// TIA Portal V17 export
// export: Created 2025-03-14T10:45:43.7128547Z, ExportSetting WithDefaults, DisplayName Totally Integrated Automation Portal, DisplayVersion V17 Update 8, DisplayName TIA Portal Openness, DisplayVersion V17 Update 8, DisplayName TIA Portal Version Control Interface, DisplayVersion V17, DisplayName SINAMICS Startdrive Advanced, DisplayVersion V17 SP2, DisplayName SINAMICS Startdrive G110M, G120, G120C, G120D, G120P, G115D, DisplayVersion V17 SP2, DisplayName SINAMICS Startdrive G130, G150, S120, S150, SINAMICS MV, S210, DisplayVersion V17 SP2, DisplayName STEP 7 Professional, DisplayVersion V17 Update 8, DisplayName SINUMERIK ONE STEP 7 Toolbox, DisplayVersion V17 Update 12, DisplayName SINUMERIK 840D sl STEP 7 Toolbox, DisplayVersion V17 Update 12, DisplayName STEP 7 Safety, DisplayVersion V17 Update 6, DisplayName WinCC Advanced, DisplayVersion V17 Update 8
FUNCTION "FC2036_MANUAL_LOAD_CYCLE" : Void   // FC2036, LAD
{ S7_Optimized_Access := 'FALSE' }
AUTHOR : ETXETAR
VERSION : 1.0
// stored: AutoNumber false, IsIECCheckEnabled false, SetENOAutomatically false, UDAEnableTagReadback false
   VAR_TEMP
      O_BYTE_0 : Struct   // OPTIONS BYTE 0
         MANUAL_LOAD_SELECTOR : Bool;   // MANUAL LOAD SELECTOR OPTION
      END_STRUCT;
   END_VAR
   VAR CONSTANT
      FC_NUMBER : Int := 2036;
      ZERO : Char := '0';
   END_VAR
   VAR_TEMP   // added for the SCL form of the ladder/FBD networks
      _w1 : Bool;
      _w2 : Bool;
      _w3 : Bool;
      _w4 : Bool;
      _w5 : Bool;
      _w6 : Bool;
      _w7 : Bool;
      _w8 : Bool;
      _w9 : Bool;
      _w10 : Bool;
      _w11 : Bool;
      _w12 : Bool;
      _w13 : Bool;
      _w14 : Bool;
      _w15 : Bool;
      _w16 : Bool;
      _w17 : Bool;
      _w18 : Bool;
      _w19 : Bool;
      _w20 : Bool;
      _w21 : Bool;
      _w22 : Bool;
      _w23 : Bool;
      _w24 : Bool;
      _w25 : Bool;
      _w26 : Bool;
   END_VAR
BEGIN

REGION Network 1: MANUAL LOAD SELECTOR OPTION
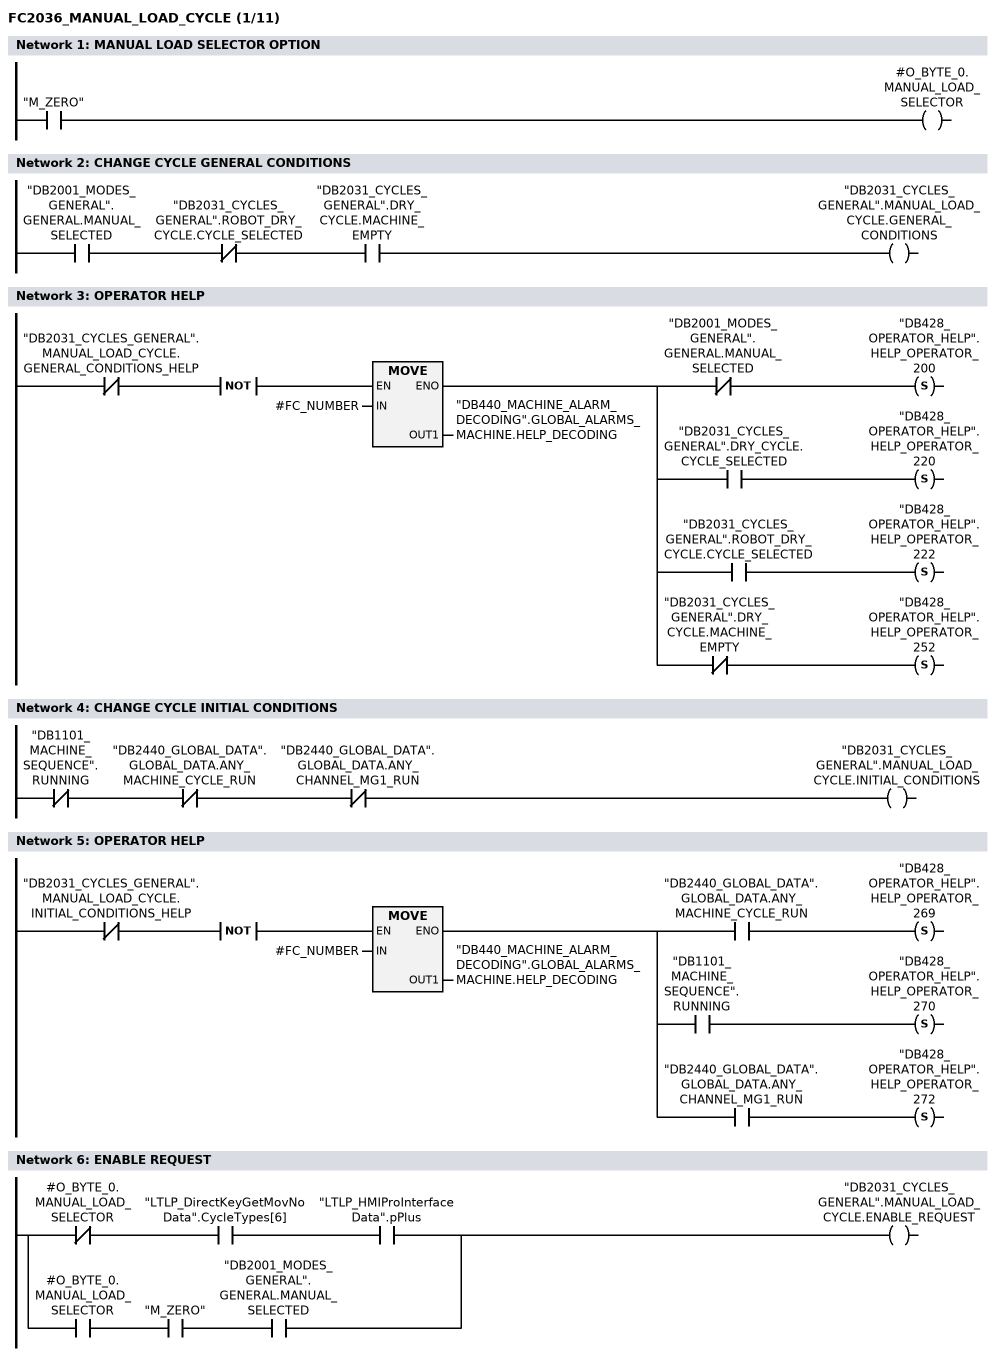
   RUNG wire#powerrail
      Contact( "M_ZERO" )
      Coil( #O_BYTE_0.MANUAL_LOAD_SELECTOR )
   END_RUNG
   // the same network as SCL:
   #O_BYTE_0.MANUAL_LOAD_SELECTOR := "M_ZERO";
END_REGION

REGION Network 2: CHANGE CYCLE GENERAL CONDITIONS
   RUNG wire#powerrail
      Contact( "DB2001_MODES_GENERAL".GENERAL.MANUAL_SELECTED )
      I_Contact( "DB2031_CYCLES_GENERAL".ROBOT_DRY_CYCLE.CYCLE_SELECTED )
      Contact( "DB2031_CYCLES_GENERAL".DRY_CYCLE.MACHINE_EMPTY )
      Coil( "DB2031_CYCLES_GENERAL".MANUAL_LOAD_CYCLE.GENERAL_CONDITIONS )
   END_RUNG
   // the same network as SCL:
   "DB2031_CYCLES_GENERAL".MANUAL_LOAD_CYCLE.GENERAL_CONDITIONS := "DB2001_MODES_GENERAL".GENERAL.MANUAL_SELECTED AND NOT "DB2031_CYCLES_GENERAL".ROBOT_DRY_CYCLE.CYCLE_SELECTED AND "DB2031_CYCLES_GENERAL".DRY_CYCLE.MACHINE_EMPTY;
END_REGION

REGION Network 3: OPERATOR HELP
   RUNG wire#powerrail
      I_Contact( "DB2031_CYCLES_GENERAL".MANUAL_LOAD_CYCLE.GENERAL_CONDITIONS_HELP )
      Not()
      { S7_GenerateENO := "TRUE" } Move(in := #FC_NUMBER, out1 => "DB440_MACHINE_ALARM_DECODING".GLOBAL_ALARMS_MACHINE.HELP_DECODING)
      wire#w1
      I_Contact( "DB2001_MODES_GENERAL".GENERAL.MANUAL_SELECTED )
      S_Coil( "DB428_OPERATOR_HELP".HELP_OPERATOR_200 )
   END_RUNG
   RUNG wire#w1
      Contact( "DB2031_CYCLES_GENERAL".DRY_CYCLE.CYCLE_SELECTED )
      S_Coil( "DB428_OPERATOR_HELP".HELP_OPERATOR_220 )
   END_RUNG
   RUNG wire#w1
      Contact( "DB2031_CYCLES_GENERAL".ROBOT_DRY_CYCLE.CYCLE_SELECTED )
      S_Coil( "DB428_OPERATOR_HELP".HELP_OPERATOR_222 )
   END_RUNG
   RUNG wire#w1
      I_Contact( "DB2031_CYCLES_GENERAL".DRY_CYCLE.MACHINE_EMPTY )
      S_Coil( "DB428_OPERATOR_HELP".HELP_OPERATOR_252 )
   END_RUNG
   // the same network as SCL:
   // ENO of a box is taken as its EN; it also drops when the box reports an error
   #_w1 := NOT (NOT "DB2031_CYCLES_GENERAL".MANUAL_LOAD_CYCLE.GENERAL_CONDITIONS_HELP);
   IF #_w1 THEN "DB440_MACHINE_ALARM_DECODING".GLOBAL_ALARMS_MACHINE.HELP_DECODING := #FC_NUMBER; END_IF;
   IF #_w1 AND NOT "DB2001_MODES_GENERAL".GENERAL.MANUAL_SELECTED THEN
       "DB428_OPERATOR_HELP".HELP_OPERATOR_200 := TRUE;
   END_IF;
   IF #_w1 AND "DB2031_CYCLES_GENERAL".DRY_CYCLE.CYCLE_SELECTED THEN
       "DB428_OPERATOR_HELP".HELP_OPERATOR_220 := TRUE;
   END_IF;
   IF #_w1 AND "DB2031_CYCLES_GENERAL".ROBOT_DRY_CYCLE.CYCLE_SELECTED THEN
       "DB428_OPERATOR_HELP".HELP_OPERATOR_222 := TRUE;
   END_IF;
   IF #_w1 AND NOT "DB2031_CYCLES_GENERAL".DRY_CYCLE.MACHINE_EMPTY THEN
       "DB428_OPERATOR_HELP".HELP_OPERATOR_252 := TRUE;
   END_IF;
END_REGION

REGION Network 4: CHANGE CYCLE INITIAL CONDITIONS
   RUNG wire#powerrail
      I_Contact( "DB1101_MACHINE_SEQUENCE".RUNNING )
      I_Contact( "DB2440_GLOBAL_DATA".GLOBAL_DATA.ANY_MACHINE_CYCLE_RUN )
      I_Contact( "DB2440_GLOBAL_DATA".GLOBAL_DATA.ANY_CHANNEL_MG1_RUN )
      Coil( "DB2031_CYCLES_GENERAL".MANUAL_LOAD_CYCLE.INITIAL_CONDITIONS )
   END_RUNG
   // the same network as SCL:
   "DB2031_CYCLES_GENERAL".MANUAL_LOAD_CYCLE.INITIAL_CONDITIONS := NOT "DB1101_MACHINE_SEQUENCE".RUNNING AND NOT "DB2440_GLOBAL_DATA".GLOBAL_DATA.ANY_MACHINE_CYCLE_RUN AND NOT "DB2440_GLOBAL_DATA".GLOBAL_DATA.ANY_CHANNEL_MG1_RUN;
END_REGION

REGION Network 5: OPERATOR HELP
   RUNG wire#powerrail
      I_Contact( "DB2031_CYCLES_GENERAL".MANUAL_LOAD_CYCLE.INITIAL_CONDITIONS_HELP )
      Not()
      { S7_GenerateENO := "TRUE" } Move(in := #FC_NUMBER, out1 => "DB440_MACHINE_ALARM_DECODING".GLOBAL_ALARMS_MACHINE.HELP_DECODING)
      wire#w1
      Contact( "DB2440_GLOBAL_DATA".GLOBAL_DATA.ANY_MACHINE_CYCLE_RUN )
      S_Coil( "DB428_OPERATOR_HELP".HELP_OPERATOR_269 )
   END_RUNG
   RUNG wire#w1
      Contact( "DB1101_MACHINE_SEQUENCE".RUNNING )
      S_Coil( "DB428_OPERATOR_HELP".HELP_OPERATOR_270 )
   END_RUNG
   RUNG wire#w1
      Contact( "DB2440_GLOBAL_DATA".GLOBAL_DATA.ANY_CHANNEL_MG1_RUN )
      S_Coil( "DB428_OPERATOR_HELP".HELP_OPERATOR_272 )
   END_RUNG
   // the same network as SCL:
   // ENO of a box is taken as its EN; it also drops when the box reports an error
   #_w1 := NOT (NOT "DB2031_CYCLES_GENERAL".MANUAL_LOAD_CYCLE.INITIAL_CONDITIONS_HELP);
   IF #_w1 THEN "DB440_MACHINE_ALARM_DECODING".GLOBAL_ALARMS_MACHINE.HELP_DECODING := #FC_NUMBER; END_IF;
   IF #_w1 AND "DB2440_GLOBAL_DATA".GLOBAL_DATA.ANY_MACHINE_CYCLE_RUN THEN
       "DB428_OPERATOR_HELP".HELP_OPERATOR_269 := TRUE;
   END_IF;
   IF #_w1 AND "DB1101_MACHINE_SEQUENCE".RUNNING THEN
       "DB428_OPERATOR_HELP".HELP_OPERATOR_270 := TRUE;
   END_IF;
   IF #_w1 AND "DB2440_GLOBAL_DATA".GLOBAL_DATA.ANY_CHANNEL_MG1_RUN THEN
       "DB428_OPERATOR_HELP".HELP_OPERATOR_272 := TRUE;
   END_IF;
END_REGION

REGION Network 6: ENABLE REQUEST
   RUNG wire#powerrail
      I_Contact( #O_BYTE_0.MANUAL_LOAD_SELECTOR )
      Contact( "LTLP_DirectKeyGetMovNoData".CycleTypes[6] )
      Contact( "LTLP_HMIProInterfaceData".pPlus )
      wire#w1
      Coil( "DB2031_CYCLES_GENERAL".MANUAL_LOAD_CYCLE.ENABLE_REQUEST )
   END_RUNG
   RUNG wire#powerrail
      Contact( #O_BYTE_0.MANUAL_LOAD_SELECTOR )
      Contact( "M_ZERO" )
      Contact( "DB2001_MODES_GENERAL".GENERAL.MANUAL_SELECTED )
   END_RUNG wire#w1
   // the same network as SCL:
   "DB2031_CYCLES_GENERAL".MANUAL_LOAD_CYCLE.ENABLE_REQUEST := (NOT #O_BYTE_0.MANUAL_LOAD_SELECTOR AND "LTLP_DirectKeyGetMovNoData".CycleTypes[6] AND "LTLP_HMIProInterfaceData".pPlus) OR (#O_BYTE_0.MANUAL_LOAD_SELECTOR AND "M_ZERO" AND "DB2001_MODES_GENERAL".GENERAL.MANUAL_SELECTED);
END_REGION

REGION Network 7: DISABLE REQUEST
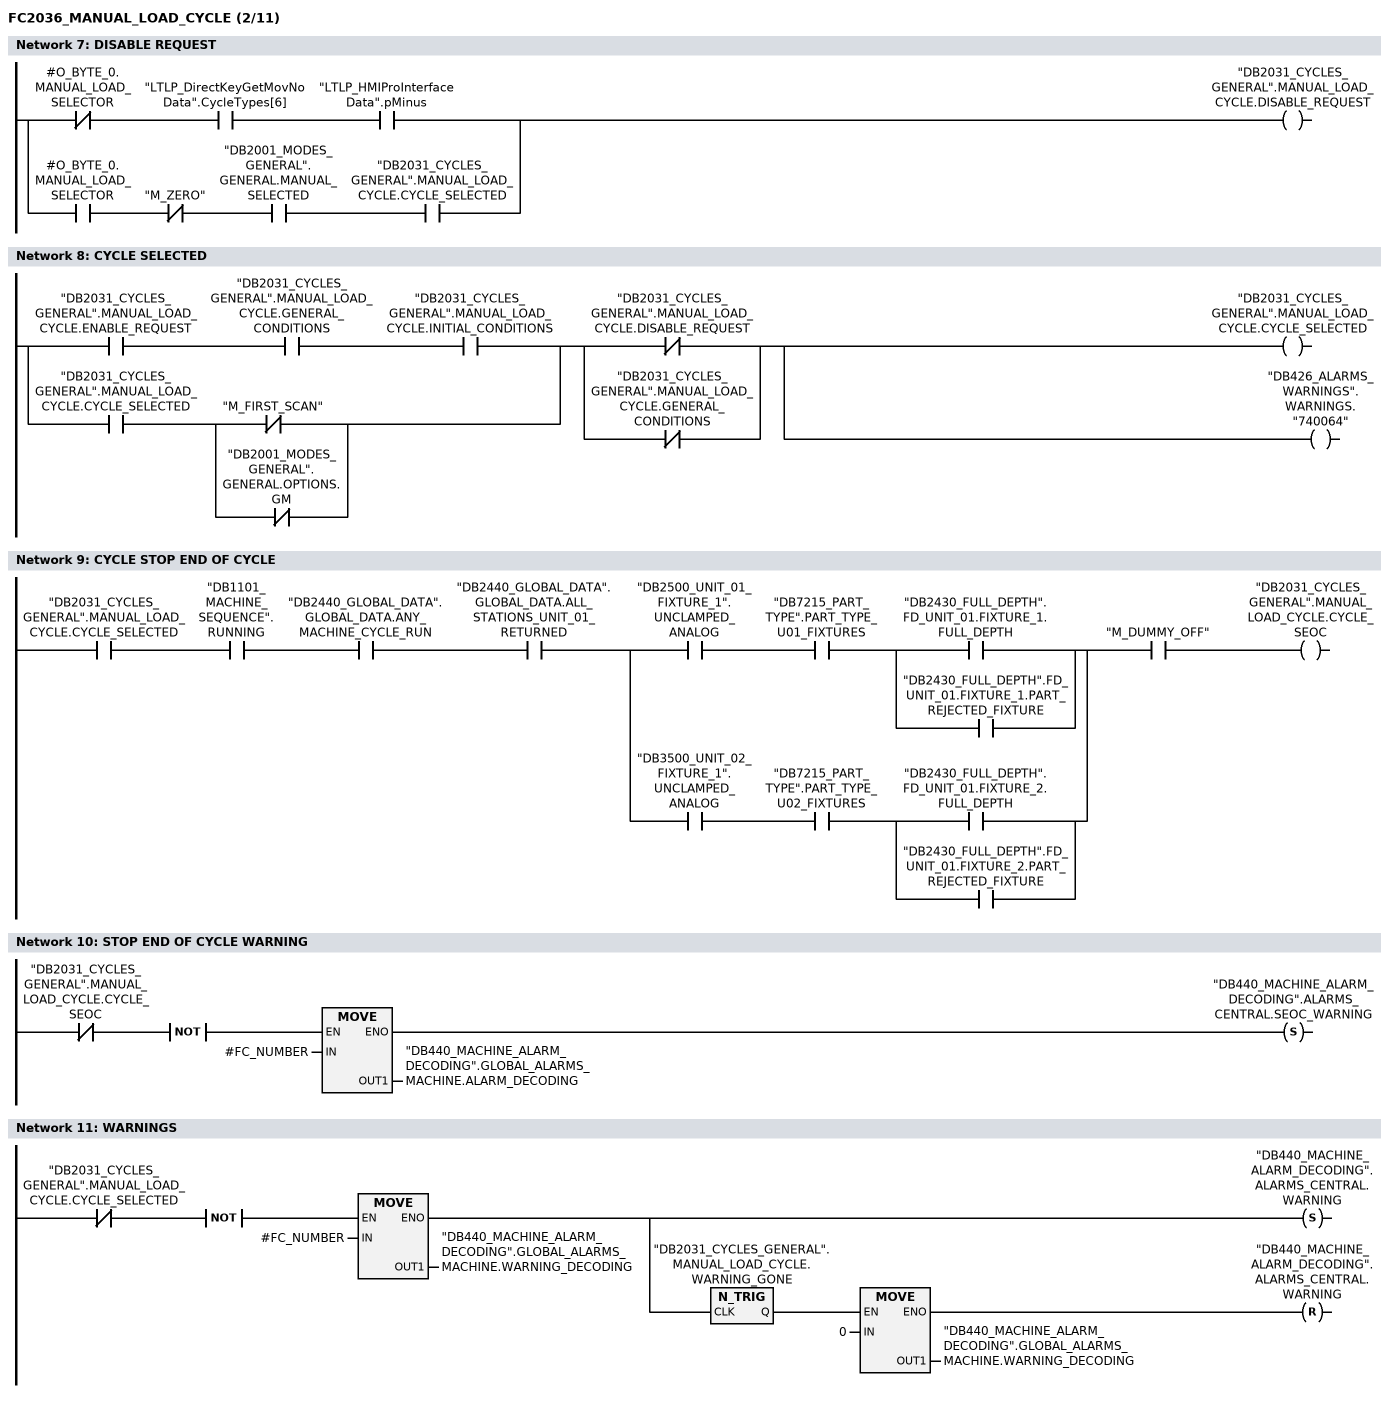
   RUNG wire#powerrail
      I_Contact( #O_BYTE_0.MANUAL_LOAD_SELECTOR )
      Contact( "LTLP_DirectKeyGetMovNoData".CycleTypes[6] )
      Contact( "LTLP_HMIProInterfaceData".pMinus )
      wire#w1
      Coil( "DB2031_CYCLES_GENERAL".MANUAL_LOAD_CYCLE.DISABLE_REQUEST )
   END_RUNG
   RUNG wire#powerrail
      Contact( #O_BYTE_0.MANUAL_LOAD_SELECTOR )
      I_Contact( "M_ZERO" )
      Contact( "DB2001_MODES_GENERAL".GENERAL.MANUAL_SELECTED )
      Contact( "DB2031_CYCLES_GENERAL".MANUAL_LOAD_CYCLE.CYCLE_SELECTED )
   END_RUNG wire#w1
   // the same network as SCL:
   "DB2031_CYCLES_GENERAL".MANUAL_LOAD_CYCLE.DISABLE_REQUEST := (NOT #O_BYTE_0.MANUAL_LOAD_SELECTOR AND "LTLP_DirectKeyGetMovNoData".CycleTypes[6] AND "LTLP_HMIProInterfaceData".pMinus) OR (#O_BYTE_0.MANUAL_LOAD_SELECTOR AND NOT "M_ZERO" AND "DB2001_MODES_GENERAL".GENERAL.MANUAL_SELECTED AND "DB2031_CYCLES_GENERAL".MANUAL_LOAD_CYCLE.CYCLE_SELECTED);
END_REGION

REGION Network 8: CYCLE SELECTED
   RUNG wire#powerrail
      Contact( "DB2031_CYCLES_GENERAL".MANUAL_LOAD_CYCLE.ENABLE_REQUEST )
      Contact( "DB2031_CYCLES_GENERAL".MANUAL_LOAD_CYCLE.GENERAL_CONDITIONS )
      Contact( "DB2031_CYCLES_GENERAL".MANUAL_LOAD_CYCLE.INITIAL_CONDITIONS )
      wire#w1
      I_Contact( "DB2031_CYCLES_GENERAL".MANUAL_LOAD_CYCLE.DISABLE_REQUEST )
      wire#w3
      Coil( "DB2031_CYCLES_GENERAL".MANUAL_LOAD_CYCLE.CYCLE_SELECTED )
   END_RUNG
   RUNG wire#powerrail
      Contact( "DB2031_CYCLES_GENERAL".MANUAL_LOAD_CYCLE.CYCLE_SELECTED )
      wire#w2
      I_Contact( "M_FIRST_SCAN" )
   END_RUNG wire#w1
   RUNG wire#w2
      I_Contact( "DB2001_MODES_GENERAL".GENERAL.OPTIONS.GM )
   END_RUNG wire#w1
   RUNG wire#w1
      I_Contact( "DB2031_CYCLES_GENERAL".MANUAL_LOAD_CYCLE.GENERAL_CONDITIONS )
   END_RUNG wire#w3
   RUNG wire#w3
      Coil( "DB426_ALARMS_WARNINGS".WARNINGS."740064" )
   END_RUNG
   // the same network as SCL:
   "DB2031_CYCLES_GENERAL".MANUAL_LOAD_CYCLE.CYCLE_SELECTED := (("DB2031_CYCLES_GENERAL".MANUAL_LOAD_CYCLE.ENABLE_REQUEST AND "DB2031_CYCLES_GENERAL".MANUAL_LOAD_CYCLE.GENERAL_CONDITIONS AND "DB2031_CYCLES_GENERAL".MANUAL_LOAD_CYCLE.INITIAL_CONDITIONS) OR ("DB2031_CYCLES_GENERAL".MANUAL_LOAD_CYCLE.CYCLE_SELECTED AND (NOT "M_FIRST_SCAN" OR NOT "DB2001_MODES_GENERAL".GENERAL.OPTIONS.GM))) AND (NOT "DB2031_CYCLES_GENERAL".MANUAL_LOAD_CYCLE.DISABLE_REQUEST OR NOT "DB2031_CYCLES_GENERAL".MANUAL_LOAD_CYCLE.GENERAL_CONDITIONS);
   "DB426_ALARMS_WARNINGS".WARNINGS."740064" := "DB2031_CYCLES_GENERAL".MANUAL_LOAD_CYCLE.CYCLE_SELECTED;
END_REGION

REGION Network 9: CYCLE STOP END OF CYCLE
   RUNG wire#powerrail
      Contact( "DB2031_CYCLES_GENERAL".MANUAL_LOAD_CYCLE.CYCLE_SELECTED )
      Contact( "DB1101_MACHINE_SEQUENCE".RUNNING )
      Contact( "DB2440_GLOBAL_DATA".GLOBAL_DATA.ANY_MACHINE_CYCLE_RUN )
      Contact( "DB2440_GLOBAL_DATA".GLOBAL_DATA.ALL_STATIONS_UNIT_01_RETURNED )
      wire#w1
      Contact( "DB2500_UNIT_01_FIXTURE_1".UNCLAMPED_ANALOG )
      Contact( "DB7215_PART_TYPE".PART_TYPE_U01_FIXTURES )
      wire#w2
      Contact( "DB2430_FULL_DEPTH".FD_UNIT_01.FIXTURE_1.FULL_DEPTH )
      wire#w3
      Contact( "M_DUMMY_OFF" )
      Coil( "DB2031_CYCLES_GENERAL".MANUAL_LOAD_CYCLE.CYCLE_SEOC )
   END_RUNG
   RUNG wire#w2
      Contact( "DB2430_FULL_DEPTH".FD_UNIT_01.FIXTURE_1.PART_REJECTED_FIXTURE )
   END_RUNG wire#w3
   RUNG wire#w1
      Contact( "DB3500_UNIT_02_FIXTURE_1".UNCLAMPED_ANALOG )
      Contact( "DB7215_PART_TYPE".PART_TYPE_U02_FIXTURES )
      wire#w4
      Contact( "DB2430_FULL_DEPTH".FD_UNIT_01.FIXTURE_2.FULL_DEPTH )
   END_RUNG wire#w3
   RUNG wire#w4
      Contact( "DB2430_FULL_DEPTH".FD_UNIT_01.FIXTURE_2.PART_REJECTED_FIXTURE )
   END_RUNG wire#w3
   // the same network as SCL:
   "DB2031_CYCLES_GENERAL".MANUAL_LOAD_CYCLE.CYCLE_SEOC := "DB2031_CYCLES_GENERAL".MANUAL_LOAD_CYCLE.CYCLE_SELECTED AND "DB1101_MACHINE_SEQUENCE".RUNNING AND "DB2440_GLOBAL_DATA".GLOBAL_DATA.ANY_MACHINE_CYCLE_RUN AND "DB2440_GLOBAL_DATA".GLOBAL_DATA.ALL_STATIONS_UNIT_01_RETURNED AND (("DB2500_UNIT_01_FIXTURE_1".UNCLAMPED_ANALOG AND "DB7215_PART_TYPE".PART_TYPE_U01_FIXTURES AND ("DB2430_FULL_DEPTH".FD_UNIT_01.FIXTURE_1.FULL_DEPTH OR "DB2430_FULL_DEPTH".FD_UNIT_01.FIXTURE_1.PART_REJECTED_FIXTURE)) OR ("DB3500_UNIT_02_FIXTURE_1".UNCLAMPED_ANALOG AND "DB7215_PART_TYPE".PART_TYPE_U02_FIXTURES AND ("DB2430_FULL_DEPTH".FD_UNIT_01.FIXTURE_2.FULL_DEPTH OR "DB2430_FULL_DEPTH".FD_UNIT_01.FIXTURE_2.PART_REJECTED_FIXTURE))) AND "M_DUMMY_OFF";
END_REGION

REGION Network 10: STOP END OF CYCLE WARNING
   RUNG wire#powerrail
      I_Contact( "DB2031_CYCLES_GENERAL".MANUAL_LOAD_CYCLE.CYCLE_SEOC )
      Not()
      { S7_GenerateENO := "TRUE" } Move(in := #FC_NUMBER, out1 => "DB440_MACHINE_ALARM_DECODING".GLOBAL_ALARMS_MACHINE.ALARM_DECODING)
      S_Coil( "DB440_MACHINE_ALARM_DECODING".ALARMS_CENTRAL.SEOC_WARNING )
   END_RUNG
   // the same network as SCL:
   // ENO of a box is taken as its EN; it also drops when the box reports an error
   IF NOT (NOT "DB2031_CYCLES_GENERAL".MANUAL_LOAD_CYCLE.CYCLE_SEOC) THEN
       "DB440_MACHINE_ALARM_DECODING".GLOBAL_ALARMS_MACHINE.ALARM_DECODING := #FC_NUMBER;
       "DB440_MACHINE_ALARM_DECODING".ALARMS_CENTRAL.SEOC_WARNING := TRUE;
   END_IF;
END_REGION

REGION Network 11: WARNINGS
   RUNG wire#powerrail
      I_Contact( "DB2031_CYCLES_GENERAL".MANUAL_LOAD_CYCLE.CYCLE_SELECTED )
      Not()
      Move(in := #FC_NUMBER, out1 => "DB440_MACHINE_ALARM_DECODING".GLOBAL_ALARMS_MACHINE.WARNING_DECODING)
      wire#w1
      S_Coil( "DB440_MACHINE_ALARM_DECODING".ALARMS_CENTRAL.WARNING )
   END_RUNG
   RUNG wire#w1
      N_Trig( "DB2031_CYCLES_GENERAL".MANUAL_LOAD_CYCLE.WARNING_GONE )
      Move(in := 0, out1 => "DB440_MACHINE_ALARM_DECODING".GLOBAL_ALARMS_MACHINE.WARNING_DECODING)
      R_Coil( "DB440_MACHINE_ALARM_DECODING".ALARMS_CENTRAL.WARNING )
   END_RUNG
   // the same network as SCL:
   #_w1 := NOT (NOT "DB2031_CYCLES_GENERAL".MANUAL_LOAD_CYCLE.CYCLE_SELECTED);
   IF #_w1 THEN
       "DB440_MACHINE_ALARM_DECODING".GLOBAL_ALARMS_MACHINE.WARNING_DECODING := #FC_NUMBER;
       "DB440_MACHINE_ALARM_DECODING".ALARMS_CENTRAL.WARNING := TRUE;
   END_IF;
   #_w2 := NOT #_w1 AND "DB2031_CYCLES_GENERAL".MANUAL_LOAD_CYCLE.WARNING_GONE;   // falling edge
   "DB2031_CYCLES_GENERAL".MANUAL_LOAD_CYCLE.WARNING_GONE := #_w1;
   IF #_w2 THEN
       "DB440_MACHINE_ALARM_DECODING".GLOBAL_ALARMS_MACHINE.WARNING_DECODING := 0;
       "DB440_MACHINE_ALARM_DECODING".ALARMS_CENTRAL.WARNING := FALSE;
   END_IF;
END_REGION

REGION Network 12: CHANGE CYCLE GENERAL CONDITIONS HELP
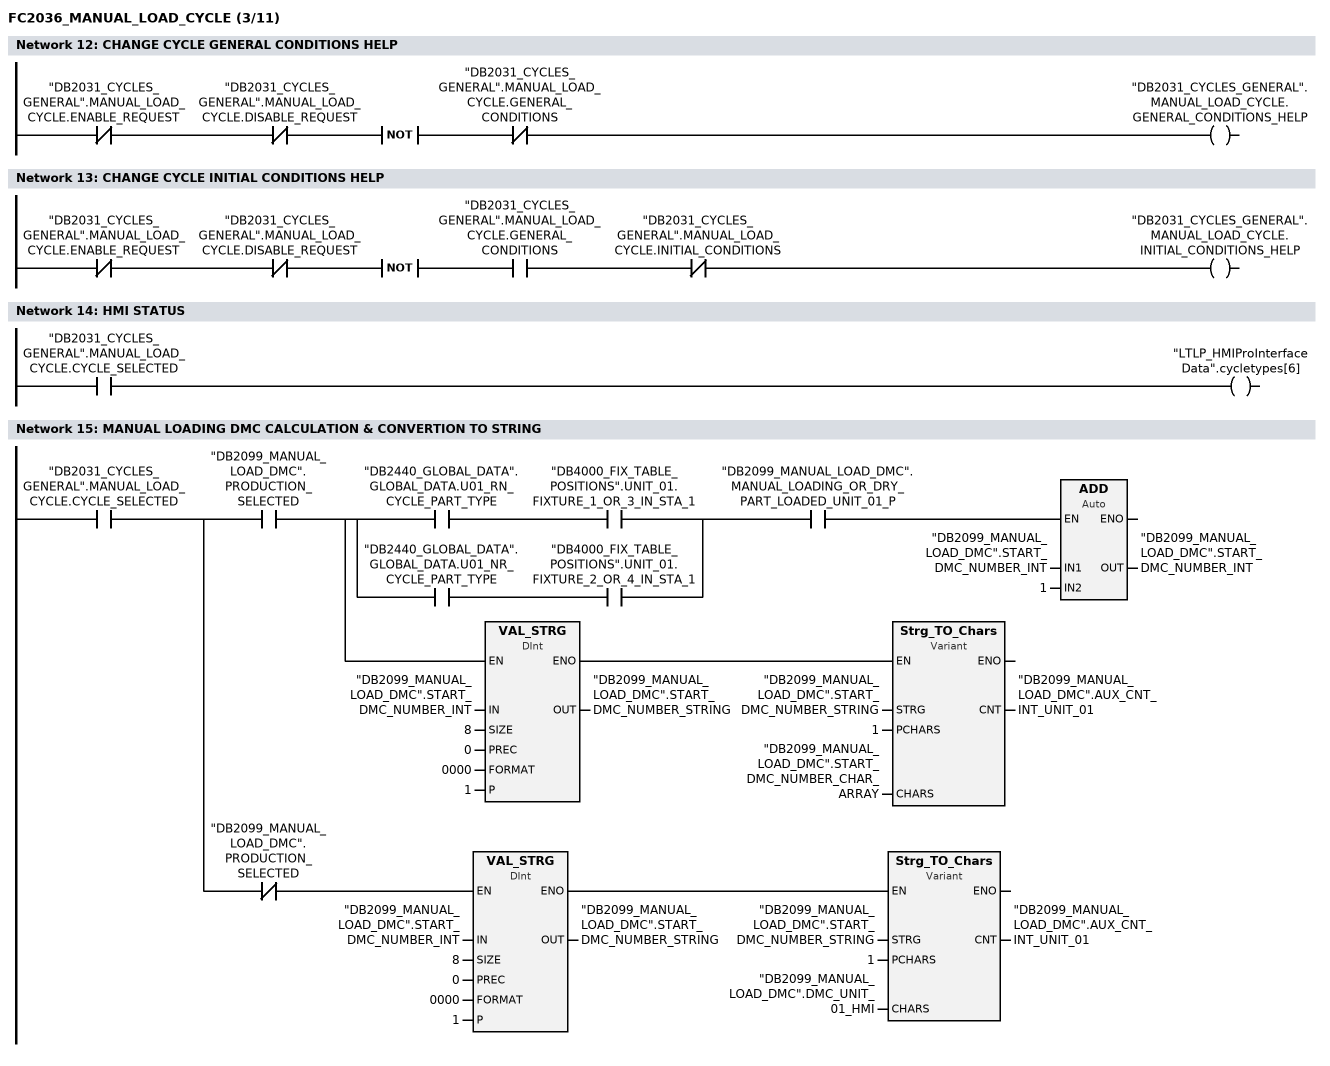
   RUNG wire#powerrail
      I_Contact( "DB2031_CYCLES_GENERAL".MANUAL_LOAD_CYCLE.ENABLE_REQUEST )
      I_Contact( "DB2031_CYCLES_GENERAL".MANUAL_LOAD_CYCLE.DISABLE_REQUEST )
      Not()
      I_Contact( "DB2031_CYCLES_GENERAL".MANUAL_LOAD_CYCLE.GENERAL_CONDITIONS )
      Coil( "DB2031_CYCLES_GENERAL".MANUAL_LOAD_CYCLE.GENERAL_CONDITIONS_HELP )
   END_RUNG
   // the same network as SCL:
   "DB2031_CYCLES_GENERAL".MANUAL_LOAD_CYCLE.GENERAL_CONDITIONS_HELP := NOT (NOT "DB2031_CYCLES_GENERAL".MANUAL_LOAD_CYCLE.ENABLE_REQUEST AND NOT "DB2031_CYCLES_GENERAL".MANUAL_LOAD_CYCLE.DISABLE_REQUEST) AND NOT "DB2031_CYCLES_GENERAL".MANUAL_LOAD_CYCLE.GENERAL_CONDITIONS;
END_REGION

REGION Network 13: CHANGE CYCLE INITIAL CONDITIONS HELP
   RUNG wire#powerrail
      I_Contact( "DB2031_CYCLES_GENERAL".MANUAL_LOAD_CYCLE.ENABLE_REQUEST )
      I_Contact( "DB2031_CYCLES_GENERAL".MANUAL_LOAD_CYCLE.DISABLE_REQUEST )
      Not()
      Contact( "DB2031_CYCLES_GENERAL".MANUAL_LOAD_CYCLE.GENERAL_CONDITIONS )
      I_Contact( "DB2031_CYCLES_GENERAL".MANUAL_LOAD_CYCLE.INITIAL_CONDITIONS )
      Coil( "DB2031_CYCLES_GENERAL".MANUAL_LOAD_CYCLE.INITIAL_CONDITIONS_HELP )
   END_RUNG
   // the same network as SCL:
   "DB2031_CYCLES_GENERAL".MANUAL_LOAD_CYCLE.INITIAL_CONDITIONS_HELP := NOT (NOT "DB2031_CYCLES_GENERAL".MANUAL_LOAD_CYCLE.ENABLE_REQUEST AND NOT "DB2031_CYCLES_GENERAL".MANUAL_LOAD_CYCLE.DISABLE_REQUEST) AND "DB2031_CYCLES_GENERAL".MANUAL_LOAD_CYCLE.GENERAL_CONDITIONS AND NOT "DB2031_CYCLES_GENERAL".MANUAL_LOAD_CYCLE.INITIAL_CONDITIONS;
END_REGION

REGION Network 14: HMI STATUS
   RUNG wire#powerrail
      Contact( "DB2031_CYCLES_GENERAL".MANUAL_LOAD_CYCLE.CYCLE_SELECTED )
      Coil( "LTLP_HMIProInterfaceData".cycletypes[6] )
   END_RUNG
   // the same network as SCL:
   "LTLP_HMIProInterfaceData".cycletypes[6] := "DB2031_CYCLES_GENERAL".MANUAL_LOAD_CYCLE.CYCLE_SELECTED;
END_REGION

REGION Network 15: MANUAL LOADING DMC CALCULATION & CONVERTION TO STRING
   RUNG wire#powerrail
      Contact( "DB2031_CYCLES_GENERAL".MANUAL_LOAD_CYCLE.CYCLE_SELECTED )
      wire#w1
      Contact( "DB2099_MANUAL_LOAD_DMC".PRODUCTION_SELECTED )
      wire#w2
      Contact( "DB2440_GLOBAL_DATA".GLOBAL_DATA.U01_RN_CYCLE_PART_TYPE )
      Contact( "DB4000_FIX_TABLE_POSITIONS".UNIT_01.FIXTURE_1_OR_3_IN_STA_1 )
      wire#w3
      Contact( "DB2099_MANUAL_LOAD_DMC".MANUAL_LOADING_OR_DRY_PART_LOADED_UNIT_01_P )
      Add(in1 := "DB2099_MANUAL_LOAD_DMC".START_DMC_NUMBER_INT, in2 := 1, out => "DB2099_MANUAL_LOAD_DMC".START_DMC_NUMBER_INT)
   END_RUNG
   RUNG wire#w2
      Contact( "DB2440_GLOBAL_DATA".GLOBAL_DATA.U01_NR_CYCLE_PART_TYPE )
      Contact( "DB4000_FIX_TABLE_POSITIONS".UNIT_01.FIXTURE_2_OR_4_IN_STA_1 )
   END_RUNG wire#w3
   RUNG wire#w2
      { S7_Templates := "[value_type := DInt, str_type := String]" } VAL_STRG(IN := "DB2099_MANUAL_LOAD_DMC".START_DMC_NUMBER_INT, SIZE := 8, PREC := 0, FORMAT := 0000, P := 1, OUT => "DB2099_MANUAL_LOAD_DMC".START_DMC_NUMBER_STRING)
      { S7_Templates := "[ptr_type := Variant, strg_type := String]" } Strg_TO_Chars(Strg := "DB2099_MANUAL_LOAD_DMC".START_DMC_NUMBER_STRING, pChars := 1, Chars := "DB2099_MANUAL_LOAD_DMC".START_DMC_NUMBER_CHAR_ARRAY, Cnt => "DB2099_MANUAL_LOAD_DMC".AUX_CNT_INT_UNIT_01)
   END_RUNG
   RUNG wire#w1
      I_Contact( "DB2099_MANUAL_LOAD_DMC".PRODUCTION_SELECTED )
      { S7_Templates := "[value_type := DInt, str_type := String]" } VAL_STRG(IN := "DB2099_MANUAL_LOAD_DMC".START_DMC_NUMBER_INT, SIZE := 8, PREC := 0, FORMAT := 0000, P := 1, OUT => "DB2099_MANUAL_LOAD_DMC".START_DMC_NUMBER_STRING)
      { S7_Templates := "[ptr_type := Variant, strg_type := String]" } Strg_TO_Chars(Strg := "DB2099_MANUAL_LOAD_DMC".START_DMC_NUMBER_STRING, pChars := 1, Chars := "DB2099_MANUAL_LOAD_DMC".DMC_UNIT_01_HMI, Cnt => "DB2099_MANUAL_LOAD_DMC".AUX_CNT_INT_UNIT_01)
   END_RUNG
   // the same network as SCL:
   #_w1 := "DB2031_CYCLES_GENERAL".MANUAL_LOAD_CYCLE.CYCLE_SELECTED AND "DB2099_MANUAL_LOAD_DMC".PRODUCTION_SELECTED;
   IF #_w1 AND (("DB2440_GLOBAL_DATA".GLOBAL_DATA.U01_RN_CYCLE_PART_TYPE AND "DB4000_FIX_TABLE_POSITIONS".UNIT_01.FIXTURE_1_OR_3_IN_STA_1) OR ("DB2440_GLOBAL_DATA".GLOBAL_DATA.U01_NR_CYCLE_PART_TYPE AND "DB4000_FIX_TABLE_POSITIONS".UNIT_01.FIXTURE_2_OR_4_IN_STA_1)) AND "DB2099_MANUAL_LOAD_DMC".MANUAL_LOADING_OR_DRY_PART_LOADED_UNIT_01_P THEN
       "DB2099_MANUAL_LOAD_DMC".START_DMC_NUMBER_INT := "DB2099_MANUAL_LOAD_DMC".START_DMC_NUMBER_INT + 1;
   END_IF;
   #_w3 := "DB2031_CYCLES_GENERAL".MANUAL_LOAD_CYCLE.CYCLE_SELECTED;
   VAL_STRG(EN := #_w1,
            IN := "DB2099_MANUAL_LOAD_DMC".START_DMC_NUMBER_INT,
            SIZE := 8,
            PREC := 0,
            FORMAT := 0000,
            P := 1,
            OUT => "DB2099_MANUAL_LOAD_DMC".START_DMC_NUMBER_STRING,
            ENO => #_w2);
   IF #_w2 THEN
       Strg_TO_Chars(Strg := "DB2099_MANUAL_LOAD_DMC".START_DMC_NUMBER_STRING,
                     pChars := 1,
                     Chars := "DB2099_MANUAL_LOAD_DMC".START_DMC_NUMBER_CHAR_ARRAY,
                     Cnt => "DB2099_MANUAL_LOAD_DMC".AUX_CNT_INT_UNIT_01);
   END_IF;
   VAL_STRG(EN := #_w3 AND NOT "DB2099_MANUAL_LOAD_DMC".PRODUCTION_SELECTED,
            IN := "DB2099_MANUAL_LOAD_DMC".START_DMC_NUMBER_INT,
            SIZE := 8,
            PREC := 0,
            FORMAT := 0000,
            P := 1,
            OUT => "DB2099_MANUAL_LOAD_DMC".START_DMC_NUMBER_STRING,
            ENO => #_w4);
   IF #_w4 THEN
       Strg_TO_Chars(Strg := "DB2099_MANUAL_LOAD_DMC".START_DMC_NUMBER_STRING,
                     pChars := 1,
                     Chars := "DB2099_MANUAL_LOAD_DMC".DMC_UNIT_01_HMI,
                     Cnt => "DB2099_MANUAL_LOAD_DMC".AUX_CNT_INT_UNIT_01);
   END_IF;
END_REGION

REGION Network 16: PART DMC UNIT 01 WRITING FOR MANUAL LOADING & NOT PRODUCTION SELECTED
   // M0.2 CUANDO SE DECIDA CON LEON CAMBIAR LA ESTRUCTURA DEL DMC SOLO HARA FALTA BORRAR LO QUE ESTÁ TRAS M0.2 Y BORRAR EL M0.3 PARA QUE SE EJECUTE EL NUEVO CODIGO. DE LO CONTRARIO SUSTITUIR M0.2 POR M0.3 Y VICEVERSA
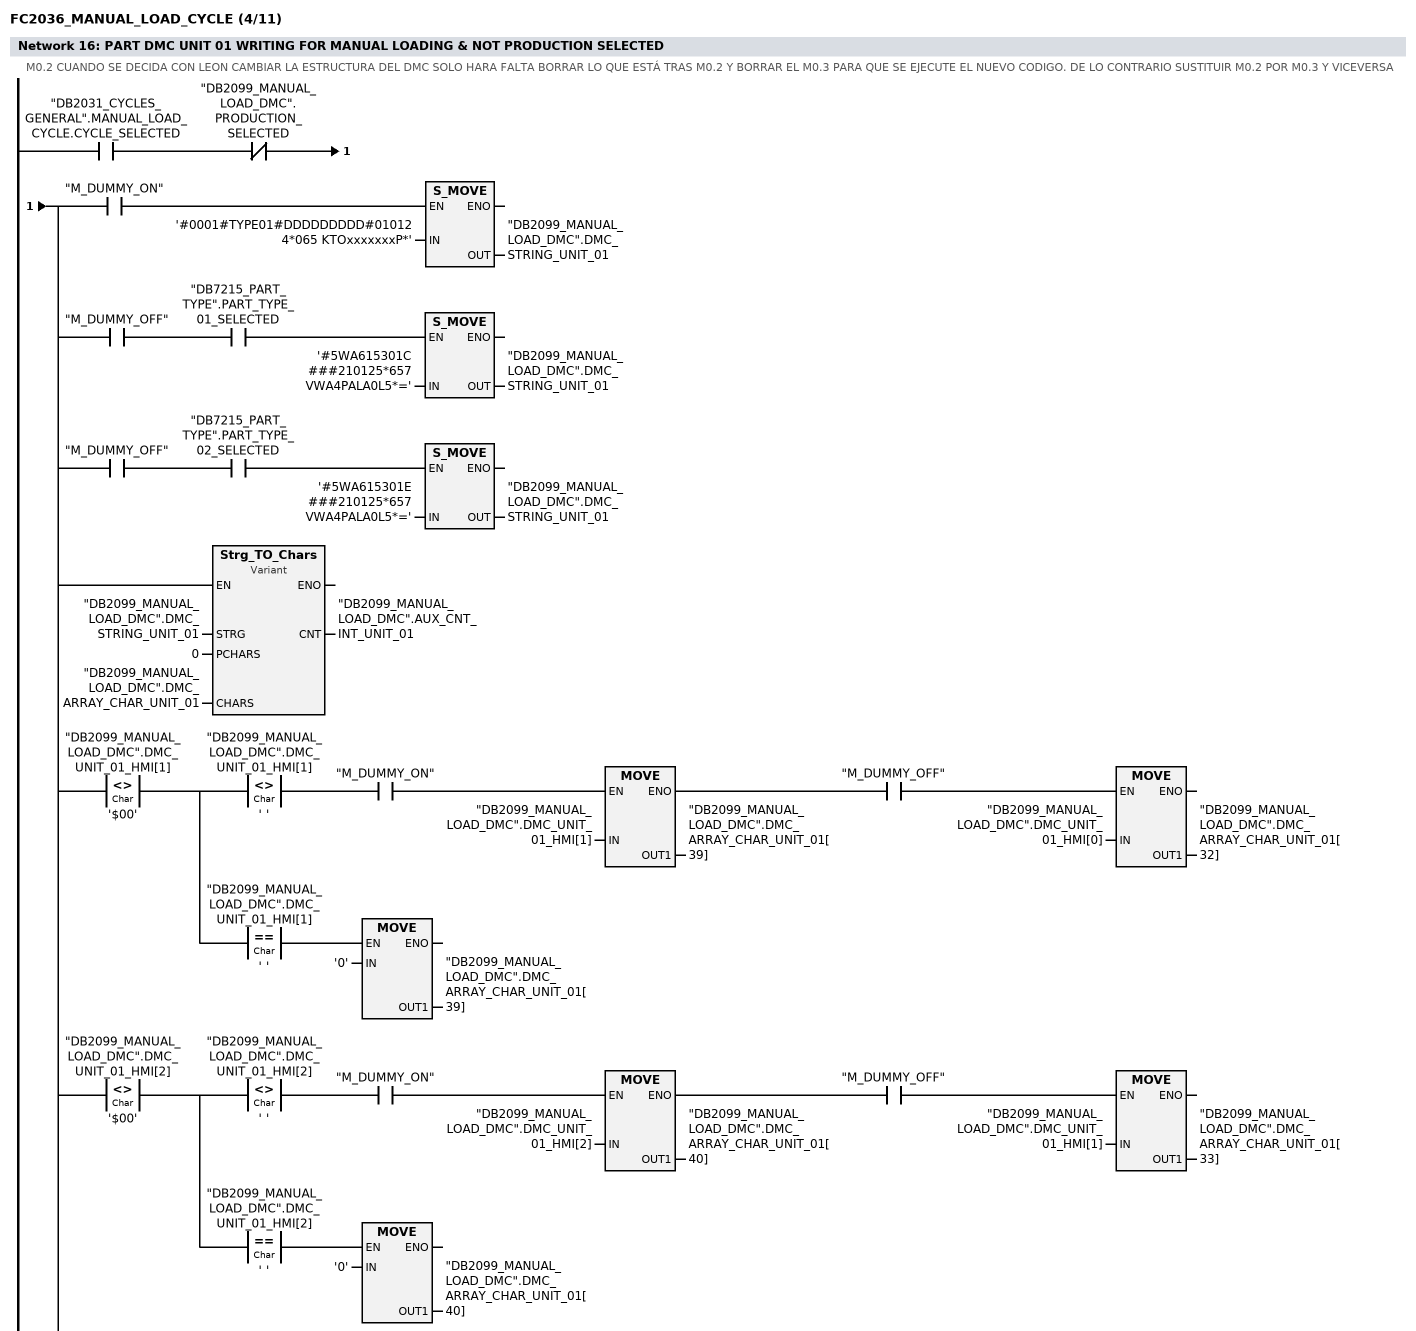
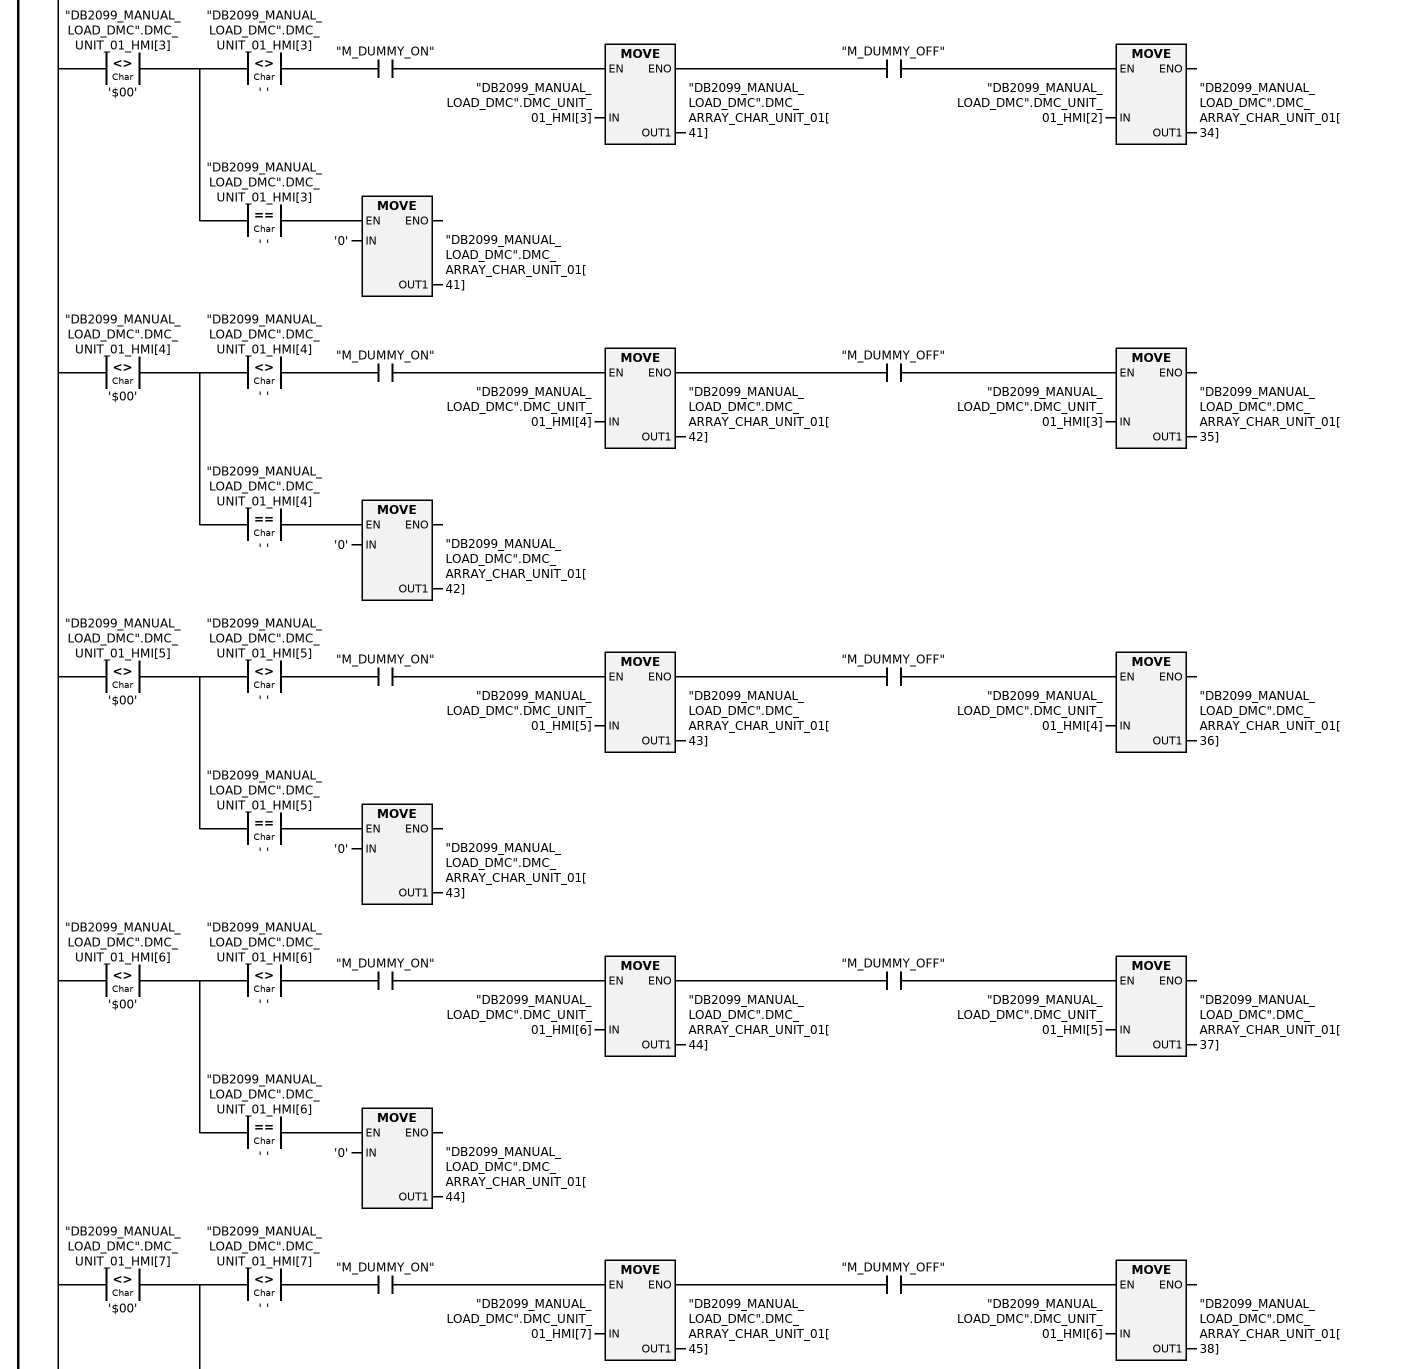
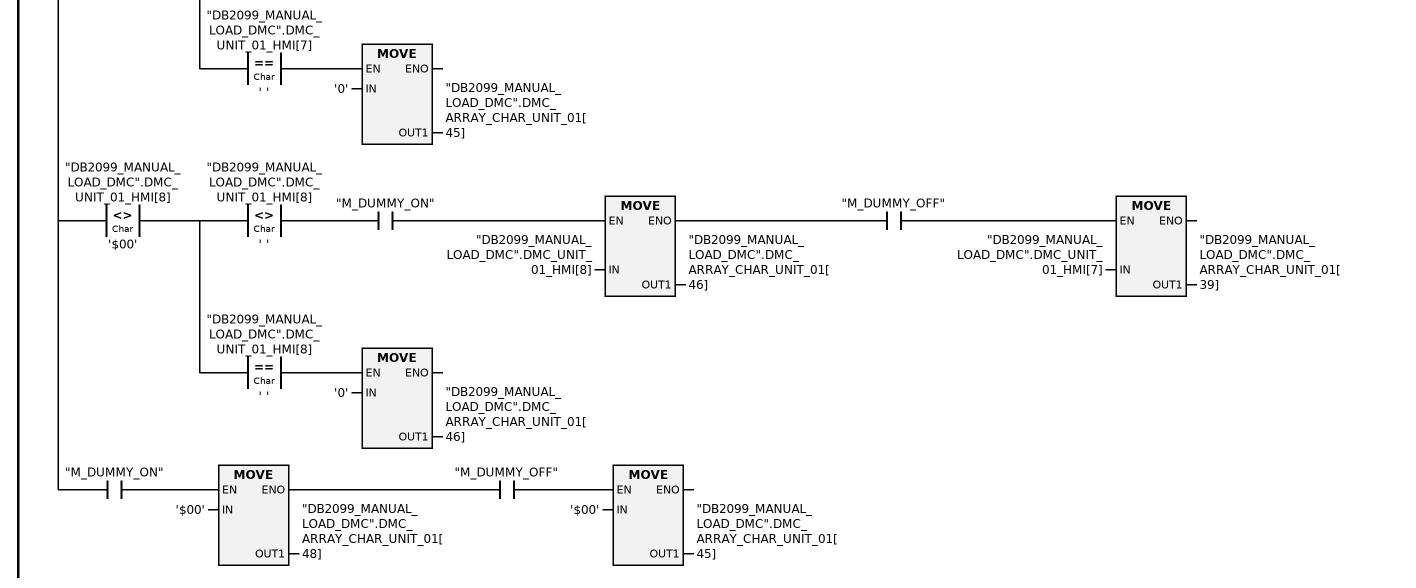
   RUNG wire#powerrail
      Contact( "DB2031_CYCLES_GENERAL".MANUAL_LOAD_CYCLE.CYCLE_SELECTED )
      I_Contact( "DB2099_MANUAL_LOAD_DMC".PRODUCTION_SELECTED )
      wire#w1
      Contact( "M_DUMMY_ON" )
      S_Move(in := '#0001#TYPE01#DDDDDDDDD#010124*065 KTOxxxxxxxP*', out => "DB2099_MANUAL_LOAD_DMC".DMC_STRING_UNIT_01)
   END_RUNG
   RUNG wire#w1
      Contact( "M_DUMMY_OFF" )
      Contact( "DB7215_PART_TYPE".PART_TYPE_01_SELECTED )
      S_Move(in := '#5WA615301C    ###210125*657 VWA4PALA0L5*=', out => "DB2099_MANUAL_LOAD_DMC".DMC_STRING_UNIT_01)
   END_RUNG
   RUNG wire#w1
      Contact( "M_DUMMY_OFF" )
      Contact( "DB7215_PART_TYPE".PART_TYPE_02_SELECTED )
      S_Move(in := '#5WA615301E    ###210125*657 VWA4PALA0L5*=', out => "DB2099_MANUAL_LOAD_DMC".DMC_STRING_UNIT_01)
   END_RUNG
   RUNG wire#w1
      { S7_Templates := "[ptr_type := Variant, strg_type := String]" } Strg_TO_Chars(Strg := "DB2099_MANUAL_LOAD_DMC".DMC_STRING_UNIT_01, pChars := 0, Chars := "DB2099_MANUAL_LOAD_DMC".DMC_ARRAY_CHAR_UNIT_01, Cnt => "DB2099_MANUAL_LOAD_DMC".AUX_CNT_INT_UNIT_01)
   END_RUNG
   RUNG wire#w1
      { S7_Templates := "SrcType := Char" } NE_Contact(in1 := "DB2099_MANUAL_LOAD_DMC".DMC_UNIT_01_HMI[1], in2 := '$00')
      wire#w2
      { S7_Templates := "SrcType := Char" } NE_Contact(in1 := "DB2099_MANUAL_LOAD_DMC".DMC_UNIT_01_HMI[1], in2 := ' ')
      Contact( "M_DUMMY_ON" )
      Move(in := "DB2099_MANUAL_LOAD_DMC".DMC_UNIT_01_HMI[1], out1 => "DB2099_MANUAL_LOAD_DMC".DMC_ARRAY_CHAR_UNIT_01[39])
      Contact( "M_DUMMY_OFF" )
      Move(in := "DB2099_MANUAL_LOAD_DMC".DMC_UNIT_01_HMI[0], out1 => "DB2099_MANUAL_LOAD_DMC".DMC_ARRAY_CHAR_UNIT_01[32])
   END_RUNG
   RUNG wire#w2
      { S7_Templates := "SrcType := Char" } EQ_Contact(in1 := "DB2099_MANUAL_LOAD_DMC".DMC_UNIT_01_HMI[1], in2 := ' ')
      Move(in := '0', out1 => "DB2099_MANUAL_LOAD_DMC".DMC_ARRAY_CHAR_UNIT_01[39])
   END_RUNG
   RUNG wire#w1
      { S7_Templates := "SrcType := Char" } NE_Contact(in1 := "DB2099_MANUAL_LOAD_DMC".DMC_UNIT_01_HMI[2], in2 := '$00')
      wire#w3
      { S7_Templates := "SrcType := Char" } NE_Contact(in1 := "DB2099_MANUAL_LOAD_DMC".DMC_UNIT_01_HMI[2], in2 := ' ')
      Contact( "M_DUMMY_ON" )
      Move(in := "DB2099_MANUAL_LOAD_DMC".DMC_UNIT_01_HMI[2], out1 => "DB2099_MANUAL_LOAD_DMC".DMC_ARRAY_CHAR_UNIT_01[40])
      Contact( "M_DUMMY_OFF" )
      Move(in := "DB2099_MANUAL_LOAD_DMC".DMC_UNIT_01_HMI[1], out1 => "DB2099_MANUAL_LOAD_DMC".DMC_ARRAY_CHAR_UNIT_01[33])
   END_RUNG
   RUNG wire#w3
      { S7_Templates := "SrcType := Char" } EQ_Contact(in1 := "DB2099_MANUAL_LOAD_DMC".DMC_UNIT_01_HMI[2], in2 := ' ')
      Move(in := '0', out1 => "DB2099_MANUAL_LOAD_DMC".DMC_ARRAY_CHAR_UNIT_01[40])
   END_RUNG
   RUNG wire#w1
      { S7_Templates := "SrcType := Char" } NE_Contact(in1 := "DB2099_MANUAL_LOAD_DMC".DMC_UNIT_01_HMI[3], in2 := '$00')
      wire#w4
      { S7_Templates := "SrcType := Char" } NE_Contact(in1 := "DB2099_MANUAL_LOAD_DMC".DMC_UNIT_01_HMI[3], in2 := ' ')
      Contact( "M_DUMMY_ON" )
      Move(in := "DB2099_MANUAL_LOAD_DMC".DMC_UNIT_01_HMI[3], out1 => "DB2099_MANUAL_LOAD_DMC".DMC_ARRAY_CHAR_UNIT_01[41])
      Contact( "M_DUMMY_OFF" )
      Move(in := "DB2099_MANUAL_LOAD_DMC".DMC_UNIT_01_HMI[2], out1 => "DB2099_MANUAL_LOAD_DMC".DMC_ARRAY_CHAR_UNIT_01[34])
   END_RUNG
   RUNG wire#w4
      { S7_Templates := "SrcType := Char" } EQ_Contact(in1 := "DB2099_MANUAL_LOAD_DMC".DMC_UNIT_01_HMI[3], in2 := ' ')
      Move(in := '0', out1 => "DB2099_MANUAL_LOAD_DMC".DMC_ARRAY_CHAR_UNIT_01[41])
   END_RUNG
   RUNG wire#w1
      { S7_Templates := "SrcType := Char" } NE_Contact(in1 := "DB2099_MANUAL_LOAD_DMC".DMC_UNIT_01_HMI[4], in2 := '$00')
      wire#w5
      { S7_Templates := "SrcType := Char" } NE_Contact(in1 := "DB2099_MANUAL_LOAD_DMC".DMC_UNIT_01_HMI[4], in2 := ' ')
      Contact( "M_DUMMY_ON" )
      Move(in := "DB2099_MANUAL_LOAD_DMC".DMC_UNIT_01_HMI[4], out1 => "DB2099_MANUAL_LOAD_DMC".DMC_ARRAY_CHAR_UNIT_01[42])
      Contact( "M_DUMMY_OFF" )
      Move(in := "DB2099_MANUAL_LOAD_DMC".DMC_UNIT_01_HMI[3], out1 => "DB2099_MANUAL_LOAD_DMC".DMC_ARRAY_CHAR_UNIT_01[35])
   END_RUNG
   RUNG wire#w5
      { S7_Templates := "SrcType := Char" } EQ_Contact(in1 := "DB2099_MANUAL_LOAD_DMC".DMC_UNIT_01_HMI[4], in2 := ' ')
      Move(in := '0', out1 => "DB2099_MANUAL_LOAD_DMC".DMC_ARRAY_CHAR_UNIT_01[42])
   END_RUNG
   RUNG wire#w1
      { S7_Templates := "SrcType := Char" } NE_Contact(in1 := "DB2099_MANUAL_LOAD_DMC".DMC_UNIT_01_HMI[5], in2 := '$00')
      wire#w6
      { S7_Templates := "SrcType := Char" } NE_Contact(in1 := "DB2099_MANUAL_LOAD_DMC".DMC_UNIT_01_HMI[5], in2 := ' ')
      Contact( "M_DUMMY_ON" )
      Move(in := "DB2099_MANUAL_LOAD_DMC".DMC_UNIT_01_HMI[5], out1 => "DB2099_MANUAL_LOAD_DMC".DMC_ARRAY_CHAR_UNIT_01[43])
      Contact( "M_DUMMY_OFF" )
      Move(in := "DB2099_MANUAL_LOAD_DMC".DMC_UNIT_01_HMI[4], out1 => "DB2099_MANUAL_LOAD_DMC".DMC_ARRAY_CHAR_UNIT_01[36])
   END_RUNG
   RUNG wire#w6
      { S7_Templates := "SrcType := Char" } EQ_Contact(in1 := "DB2099_MANUAL_LOAD_DMC".DMC_UNIT_01_HMI[5], in2 := ' ')
      Move(in := '0', out1 => "DB2099_MANUAL_LOAD_DMC".DMC_ARRAY_CHAR_UNIT_01[43])
   END_RUNG
   RUNG wire#w1
      { S7_Templates := "SrcType := Char" } NE_Contact(in1 := "DB2099_MANUAL_LOAD_DMC".DMC_UNIT_01_HMI[6], in2 := '$00')
      wire#w7
      { S7_Templates := "SrcType := Char" } NE_Contact(in1 := "DB2099_MANUAL_LOAD_DMC".DMC_UNIT_01_HMI[6], in2 := ' ')
      Contact( "M_DUMMY_ON" )
      Move(in := "DB2099_MANUAL_LOAD_DMC".DMC_UNIT_01_HMI[6], out1 => "DB2099_MANUAL_LOAD_DMC".DMC_ARRAY_CHAR_UNIT_01[44])
      Contact( "M_DUMMY_OFF" )
      Move(in := "DB2099_MANUAL_LOAD_DMC".DMC_UNIT_01_HMI[5], out1 => "DB2099_MANUAL_LOAD_DMC".DMC_ARRAY_CHAR_UNIT_01[37])
   END_RUNG
   RUNG wire#w7
      { S7_Templates := "SrcType := Char" } EQ_Contact(in1 := "DB2099_MANUAL_LOAD_DMC".DMC_UNIT_01_HMI[6], in2 := ' ')
      Move(in := '0', out1 => "DB2099_MANUAL_LOAD_DMC".DMC_ARRAY_CHAR_UNIT_01[44])
   END_RUNG
   RUNG wire#w1
      { S7_Templates := "SrcType := Char" } NE_Contact(in1 := "DB2099_MANUAL_LOAD_DMC".DMC_UNIT_01_HMI[7], in2 := '$00')
      wire#w8
      { S7_Templates := "SrcType := Char" } NE_Contact(in1 := "DB2099_MANUAL_LOAD_DMC".DMC_UNIT_01_HMI[7], in2 := ' ')
      Contact( "M_DUMMY_ON" )
      Move(in := "DB2099_MANUAL_LOAD_DMC".DMC_UNIT_01_HMI[7], out1 => "DB2099_MANUAL_LOAD_DMC".DMC_ARRAY_CHAR_UNIT_01[45])
      Contact( "M_DUMMY_OFF" )
      Move(in := "DB2099_MANUAL_LOAD_DMC".DMC_UNIT_01_HMI[6], out1 => "DB2099_MANUAL_LOAD_DMC".DMC_ARRAY_CHAR_UNIT_01[38])
   END_RUNG
   RUNG wire#w8
      { S7_Templates := "SrcType := Char" } EQ_Contact(in1 := "DB2099_MANUAL_LOAD_DMC".DMC_UNIT_01_HMI[7], in2 := ' ')
      Move(in := '0', out1 => "DB2099_MANUAL_LOAD_DMC".DMC_ARRAY_CHAR_UNIT_01[45])
   END_RUNG
   RUNG wire#w1
      { S7_Templates := "SrcType := Char" } NE_Contact(in1 := "DB2099_MANUAL_LOAD_DMC".DMC_UNIT_01_HMI[8], in2 := '$00')
      wire#w9
      { S7_Templates := "SrcType := Char" } NE_Contact(in1 := "DB2099_MANUAL_LOAD_DMC".DMC_UNIT_01_HMI[8], in2 := ' ')
      Contact( "M_DUMMY_ON" )
      Move(in := "DB2099_MANUAL_LOAD_DMC".DMC_UNIT_01_HMI[8], out1 => "DB2099_MANUAL_LOAD_DMC".DMC_ARRAY_CHAR_UNIT_01[46])
      Contact( "M_DUMMY_OFF" )
      Move(in := "DB2099_MANUAL_LOAD_DMC".DMC_UNIT_01_HMI[7], out1 => "DB2099_MANUAL_LOAD_DMC".DMC_ARRAY_CHAR_UNIT_01[39])
   END_RUNG
   RUNG wire#w9
      { S7_Templates := "SrcType := Char" } EQ_Contact(in1 := "DB2099_MANUAL_LOAD_DMC".DMC_UNIT_01_HMI[8], in2 := ' ')
      Move(in := '0', out1 => "DB2099_MANUAL_LOAD_DMC".DMC_ARRAY_CHAR_UNIT_01[46])
   END_RUNG
   RUNG wire#w1
      Contact( "M_DUMMY_ON" )
      Move(in := '$00', out1 => "DB2099_MANUAL_LOAD_DMC".DMC_ARRAY_CHAR_UNIT_01[48])
      Contact( "M_DUMMY_OFF" )
      Move(in := '$00', out1 => "DB2099_MANUAL_LOAD_DMC".DMC_ARRAY_CHAR_UNIT_01[45])
   END_RUNG
   // the same network as SCL:
   #_w1 := "DB2031_CYCLES_GENERAL".MANUAL_LOAD_CYCLE.CYCLE_SELECTED AND NOT "DB2099_MANUAL_LOAD_DMC".PRODUCTION_SELECTED;
   IF #_w1 AND "M_DUMMY_ON" THEN
       "DB2099_MANUAL_LOAD_DMC".DMC_STRING_UNIT_01 := '#0001#TYPE01#DDDDDDDDD#010124*065 KTOxxxxxxxP*';
   END_IF;
   IF #_w1 AND "M_DUMMY_OFF" AND "DB7215_PART_TYPE".PART_TYPE_01_SELECTED THEN
       "DB2099_MANUAL_LOAD_DMC".DMC_STRING_UNIT_01 := '#5WA615301C    ###210125*657 VWA4PALA0L5*=';
   END_IF;
   IF #_w1 AND "M_DUMMY_OFF" AND "DB7215_PART_TYPE".PART_TYPE_02_SELECTED THEN
       "DB2099_MANUAL_LOAD_DMC".DMC_STRING_UNIT_01 := '#5WA615301E    ###210125*657 VWA4PALA0L5*=';
   END_IF;
   IF #_w1 THEN
       Strg_TO_Chars(Strg := "DB2099_MANUAL_LOAD_DMC".DMC_STRING_UNIT_01,
                     pChars := 0,
                     Chars := "DB2099_MANUAL_LOAD_DMC".DMC_ARRAY_CHAR_UNIT_01,
                     Cnt => "DB2099_MANUAL_LOAD_DMC".AUX_CNT_INT_UNIT_01);
   END_IF;
   #_w2 := #_w1 AND ("DB2099_MANUAL_LOAD_DMC".DMC_UNIT_01_HMI[1] <> '$00');
   #_w3 := #_w2 AND ("DB2099_MANUAL_LOAD_DMC".DMC_UNIT_01_HMI[1] <> ' ') AND "M_DUMMY_ON";
   IF #_w3 THEN
       "DB2099_MANUAL_LOAD_DMC".DMC_ARRAY_CHAR_UNIT_01[39] := "DB2099_MANUAL_LOAD_DMC".DMC_UNIT_01_HMI[1];
   END_IF;
   IF #_w3 AND "M_DUMMY_OFF" THEN
       "DB2099_MANUAL_LOAD_DMC".DMC_ARRAY_CHAR_UNIT_01[32] := "DB2099_MANUAL_LOAD_DMC".DMC_UNIT_01_HMI[0];
   END_IF;
   IF #_w2 AND ("DB2099_MANUAL_LOAD_DMC".DMC_UNIT_01_HMI[1] = ' ') THEN
       "DB2099_MANUAL_LOAD_DMC".DMC_ARRAY_CHAR_UNIT_01[39] := '0';
   END_IF;
   #_w4 := #_w1 AND ("DB2099_MANUAL_LOAD_DMC".DMC_UNIT_01_HMI[2] <> '$00');
   #_w5 := #_w4 AND ("DB2099_MANUAL_LOAD_DMC".DMC_UNIT_01_HMI[2] <> ' ') AND "M_DUMMY_ON";
   IF #_w5 THEN
       "DB2099_MANUAL_LOAD_DMC".DMC_ARRAY_CHAR_UNIT_01[40] := "DB2099_MANUAL_LOAD_DMC".DMC_UNIT_01_HMI[2];
   END_IF;
   IF #_w5 AND "M_DUMMY_OFF" THEN
       "DB2099_MANUAL_LOAD_DMC".DMC_ARRAY_CHAR_UNIT_01[33] := "DB2099_MANUAL_LOAD_DMC".DMC_UNIT_01_HMI[1];
   END_IF;
   IF #_w4 AND ("DB2099_MANUAL_LOAD_DMC".DMC_UNIT_01_HMI[2] = ' ') THEN
       "DB2099_MANUAL_LOAD_DMC".DMC_ARRAY_CHAR_UNIT_01[40] := '0';
   END_IF;
   #_w6 := #_w1 AND ("DB2099_MANUAL_LOAD_DMC".DMC_UNIT_01_HMI[3] <> '$00');
   #_w7 := #_w6 AND ("DB2099_MANUAL_LOAD_DMC".DMC_UNIT_01_HMI[3] <> ' ') AND "M_DUMMY_ON";
   IF #_w7 THEN
       "DB2099_MANUAL_LOAD_DMC".DMC_ARRAY_CHAR_UNIT_01[41] := "DB2099_MANUAL_LOAD_DMC".DMC_UNIT_01_HMI[3];
   END_IF;
   IF #_w7 AND "M_DUMMY_OFF" THEN
       "DB2099_MANUAL_LOAD_DMC".DMC_ARRAY_CHAR_UNIT_01[34] := "DB2099_MANUAL_LOAD_DMC".DMC_UNIT_01_HMI[2];
   END_IF;
   IF #_w6 AND ("DB2099_MANUAL_LOAD_DMC".DMC_UNIT_01_HMI[3] = ' ') THEN
       "DB2099_MANUAL_LOAD_DMC".DMC_ARRAY_CHAR_UNIT_01[41] := '0';
   END_IF;
   #_w8 := #_w1 AND ("DB2099_MANUAL_LOAD_DMC".DMC_UNIT_01_HMI[4] <> '$00');
   #_w9 := #_w8 AND ("DB2099_MANUAL_LOAD_DMC".DMC_UNIT_01_HMI[4] <> ' ') AND "M_DUMMY_ON";
   IF #_w9 THEN
       "DB2099_MANUAL_LOAD_DMC".DMC_ARRAY_CHAR_UNIT_01[42] := "DB2099_MANUAL_LOAD_DMC".DMC_UNIT_01_HMI[4];
   END_IF;
   IF #_w9 AND "M_DUMMY_OFF" THEN
       "DB2099_MANUAL_LOAD_DMC".DMC_ARRAY_CHAR_UNIT_01[35] := "DB2099_MANUAL_LOAD_DMC".DMC_UNIT_01_HMI[3];
   END_IF;
   IF #_w8 AND ("DB2099_MANUAL_LOAD_DMC".DMC_UNIT_01_HMI[4] = ' ') THEN
       "DB2099_MANUAL_LOAD_DMC".DMC_ARRAY_CHAR_UNIT_01[42] := '0';
   END_IF;
   #_w10 := #_w1 AND ("DB2099_MANUAL_LOAD_DMC".DMC_UNIT_01_HMI[5] <> '$00');
   #_w11 := #_w10 AND ("DB2099_MANUAL_LOAD_DMC".DMC_UNIT_01_HMI[5] <> ' ') AND "M_DUMMY_ON";
   IF #_w11 THEN
       "DB2099_MANUAL_LOAD_DMC".DMC_ARRAY_CHAR_UNIT_01[43] := "DB2099_MANUAL_LOAD_DMC".DMC_UNIT_01_HMI[5];
   END_IF;
   IF #_w11 AND "M_DUMMY_OFF" THEN
       "DB2099_MANUAL_LOAD_DMC".DMC_ARRAY_CHAR_UNIT_01[36] := "DB2099_MANUAL_LOAD_DMC".DMC_UNIT_01_HMI[4];
   END_IF;
   IF #_w10 AND ("DB2099_MANUAL_LOAD_DMC".DMC_UNIT_01_HMI[5] = ' ') THEN
       "DB2099_MANUAL_LOAD_DMC".DMC_ARRAY_CHAR_UNIT_01[43] := '0';
   END_IF;
   #_w12 := #_w1 AND ("DB2099_MANUAL_LOAD_DMC".DMC_UNIT_01_HMI[6] <> '$00');
   #_w13 := #_w12 AND ("DB2099_MANUAL_LOAD_DMC".DMC_UNIT_01_HMI[6] <> ' ') AND "M_DUMMY_ON";
   IF #_w13 THEN
       "DB2099_MANUAL_LOAD_DMC".DMC_ARRAY_CHAR_UNIT_01[44] := "DB2099_MANUAL_LOAD_DMC".DMC_UNIT_01_HMI[6];
   END_IF;
   IF #_w13 AND "M_DUMMY_OFF" THEN
       "DB2099_MANUAL_LOAD_DMC".DMC_ARRAY_CHAR_UNIT_01[37] := "DB2099_MANUAL_LOAD_DMC".DMC_UNIT_01_HMI[5];
   END_IF;
   IF #_w12 AND ("DB2099_MANUAL_LOAD_DMC".DMC_UNIT_01_HMI[6] = ' ') THEN
       "DB2099_MANUAL_LOAD_DMC".DMC_ARRAY_CHAR_UNIT_01[44] := '0';
   END_IF;
   #_w14 := #_w1 AND ("DB2099_MANUAL_LOAD_DMC".DMC_UNIT_01_HMI[7] <> '$00');
   #_w15 := #_w14 AND ("DB2099_MANUAL_LOAD_DMC".DMC_UNIT_01_HMI[7] <> ' ') AND "M_DUMMY_ON";
   IF #_w15 THEN
       "DB2099_MANUAL_LOAD_DMC".DMC_ARRAY_CHAR_UNIT_01[45] := "DB2099_MANUAL_LOAD_DMC".DMC_UNIT_01_HMI[7];
   END_IF;
   IF #_w15 AND "M_DUMMY_OFF" THEN
       "DB2099_MANUAL_LOAD_DMC".DMC_ARRAY_CHAR_UNIT_01[38] := "DB2099_MANUAL_LOAD_DMC".DMC_UNIT_01_HMI[6];
   END_IF;
   IF #_w14 AND ("DB2099_MANUAL_LOAD_DMC".DMC_UNIT_01_HMI[7] = ' ') THEN
       "DB2099_MANUAL_LOAD_DMC".DMC_ARRAY_CHAR_UNIT_01[45] := '0';
   END_IF;
   #_w16 := #_w1 AND ("DB2099_MANUAL_LOAD_DMC".DMC_UNIT_01_HMI[8] <> '$00');
   #_w17 := #_w16 AND ("DB2099_MANUAL_LOAD_DMC".DMC_UNIT_01_HMI[8] <> ' ') AND "M_DUMMY_ON";
   IF #_w17 THEN
       "DB2099_MANUAL_LOAD_DMC".DMC_ARRAY_CHAR_UNIT_01[46] := "DB2099_MANUAL_LOAD_DMC".DMC_UNIT_01_HMI[8];
   END_IF;
   IF #_w17 AND "M_DUMMY_OFF" THEN
       "DB2099_MANUAL_LOAD_DMC".DMC_ARRAY_CHAR_UNIT_01[39] := "DB2099_MANUAL_LOAD_DMC".DMC_UNIT_01_HMI[7];
   END_IF;
   IF #_w16 AND ("DB2099_MANUAL_LOAD_DMC".DMC_UNIT_01_HMI[8] = ' ') THEN
       "DB2099_MANUAL_LOAD_DMC".DMC_ARRAY_CHAR_UNIT_01[46] := '0';
   END_IF;
   #_w18 := #_w1 AND "M_DUMMY_ON";
   IF #_w18 THEN "DB2099_MANUAL_LOAD_DMC".DMC_ARRAY_CHAR_UNIT_01[48] := '$00'; END_IF;
   IF #_w18 AND "M_DUMMY_OFF" THEN "DB2099_MANUAL_LOAD_DMC".DMC_ARRAY_CHAR_UNIT_01[45] := '$00'; END_IF;
END_REGION

REGION Network 17: PART DMC UNIT 02 WRITING FOR MANUAL LOADING & NOT PRODUCTION SELECTED
   // M0.2 CUANDO SE DECIDA CON LEON CAMBIAR LA ESTRUCTURA DEL DMC SOLO HARA FALTA BORRAR LO QUE ESTÁ TRAS M0.2 Y BORRAR EL M0.3 PARA QUE SE EJECUTE EL NUEVO CODIGO. DE LO CONTRARIO SUSTITUIR M0.2 POR M0.3 Y VICEVERSA
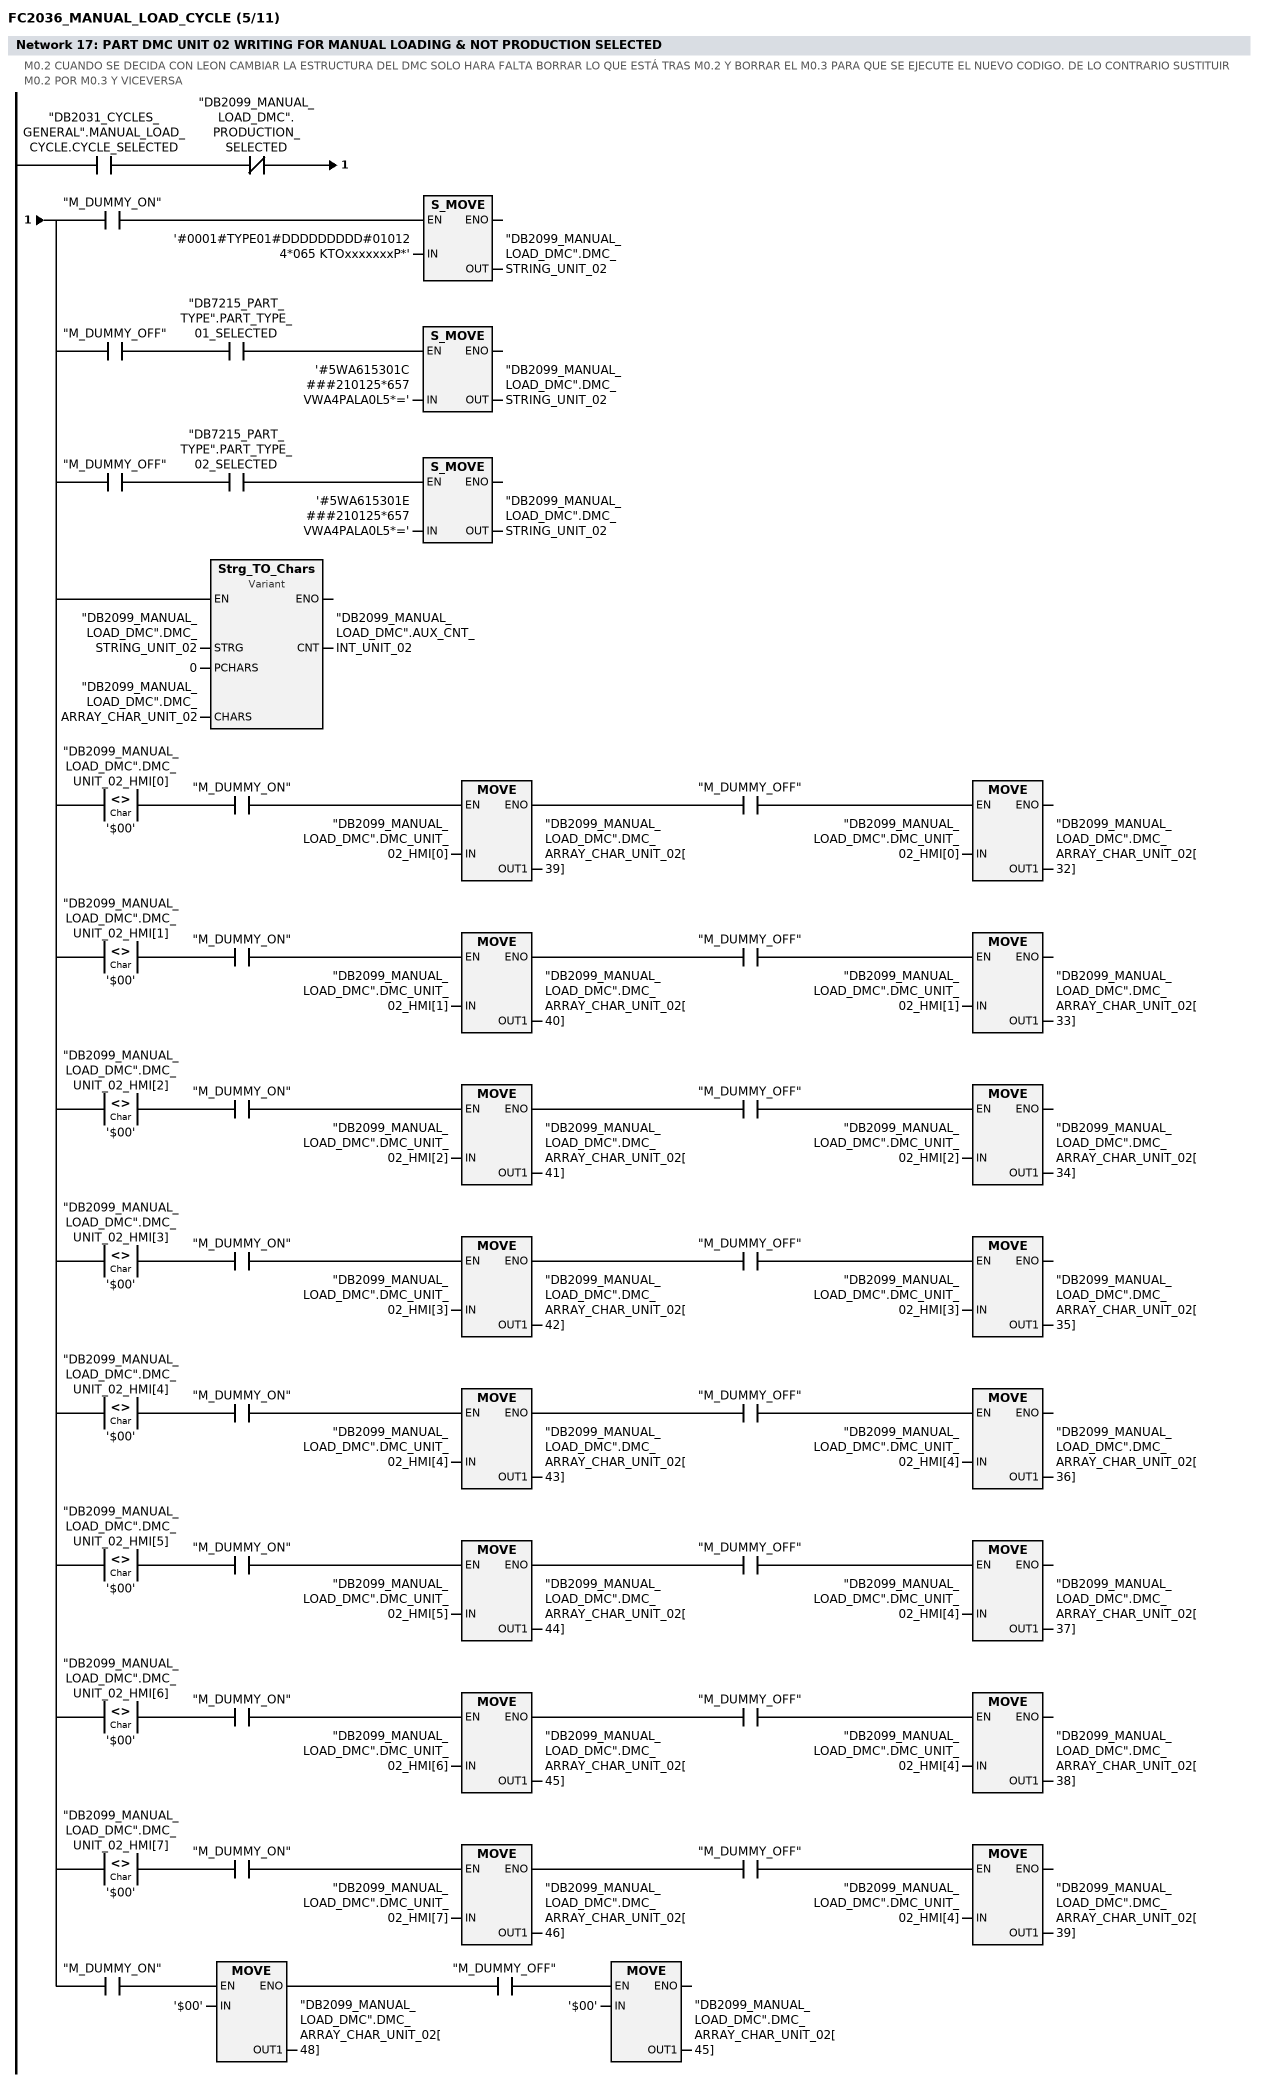
   RUNG wire#powerrail
      Contact( "DB2031_CYCLES_GENERAL".MANUAL_LOAD_CYCLE.CYCLE_SELECTED )
      I_Contact( "DB2099_MANUAL_LOAD_DMC".PRODUCTION_SELECTED )
      wire#w1
      Contact( "M_DUMMY_ON" )
      S_Move(in := '#0001#TYPE01#DDDDDDDDD#010124*065 KTOxxxxxxxP*', out => "DB2099_MANUAL_LOAD_DMC".DMC_STRING_UNIT_02)
   END_RUNG
   RUNG wire#w1
      Contact( "M_DUMMY_OFF" )
      Contact( "DB7215_PART_TYPE".PART_TYPE_01_SELECTED )
      S_Move(in := '#5WA615301C    ###210125*657 VWA4PALA0L5*=', out => "DB2099_MANUAL_LOAD_DMC".DMC_STRING_UNIT_02)
   END_RUNG
   RUNG wire#w1
      Contact( "M_DUMMY_OFF" )
      Contact( "DB7215_PART_TYPE".PART_TYPE_02_SELECTED )
      S_Move(in := '#5WA615301E    ###210125*657 VWA4PALA0L5*=', out => "DB2099_MANUAL_LOAD_DMC".DMC_STRING_UNIT_02)
   END_RUNG
   RUNG wire#w1
      { S7_Templates := "[ptr_type := Variant, strg_type := String]" } Strg_TO_Chars(Strg := "DB2099_MANUAL_LOAD_DMC".DMC_STRING_UNIT_02, pChars := 0, Chars := "DB2099_MANUAL_LOAD_DMC".DMC_ARRAY_CHAR_UNIT_02, Cnt => "DB2099_MANUAL_LOAD_DMC".AUX_CNT_INT_UNIT_02)
   END_RUNG
   RUNG wire#w1
      { S7_Templates := "SrcType := Char" } NE_Contact(in1 := "DB2099_MANUAL_LOAD_DMC".DMC_UNIT_02_HMI[0], in2 := '$00')
      Contact( "M_DUMMY_ON" )
      Move(in := "DB2099_MANUAL_LOAD_DMC".DMC_UNIT_02_HMI[0], out1 => "DB2099_MANUAL_LOAD_DMC".DMC_ARRAY_CHAR_UNIT_02[39])
      Contact( "M_DUMMY_OFF" )
      Move(in := "DB2099_MANUAL_LOAD_DMC".DMC_UNIT_02_HMI[0], out1 => "DB2099_MANUAL_LOAD_DMC".DMC_ARRAY_CHAR_UNIT_02[32])
   END_RUNG
   RUNG wire#w1
      { S7_Templates := "SrcType := Char" } NE_Contact(in1 := "DB2099_MANUAL_LOAD_DMC".DMC_UNIT_02_HMI[1], in2 := '$00')
      Contact( "M_DUMMY_ON" )
      Move(in := "DB2099_MANUAL_LOAD_DMC".DMC_UNIT_02_HMI[1], out1 => "DB2099_MANUAL_LOAD_DMC".DMC_ARRAY_CHAR_UNIT_02[40])
      Contact( "M_DUMMY_OFF" )
      Move(in := "DB2099_MANUAL_LOAD_DMC".DMC_UNIT_02_HMI[1], out1 => "DB2099_MANUAL_LOAD_DMC".DMC_ARRAY_CHAR_UNIT_02[33])
   END_RUNG
   RUNG wire#w1
      { S7_Templates := "SrcType := Char" } NE_Contact(in1 := "DB2099_MANUAL_LOAD_DMC".DMC_UNIT_02_HMI[2], in2 := '$00')
      Contact( "M_DUMMY_ON" )
      Move(in := "DB2099_MANUAL_LOAD_DMC".DMC_UNIT_02_HMI[2], out1 => "DB2099_MANUAL_LOAD_DMC".DMC_ARRAY_CHAR_UNIT_02[41])
      Contact( "M_DUMMY_OFF" )
      Move(in := "DB2099_MANUAL_LOAD_DMC".DMC_UNIT_02_HMI[2], out1 => "DB2099_MANUAL_LOAD_DMC".DMC_ARRAY_CHAR_UNIT_02[34])
   END_RUNG
   RUNG wire#w1
      { S7_Templates := "SrcType := Char" } NE_Contact(in1 := "DB2099_MANUAL_LOAD_DMC".DMC_UNIT_02_HMI[3], in2 := '$00')
      Contact( "M_DUMMY_ON" )
      Move(in := "DB2099_MANUAL_LOAD_DMC".DMC_UNIT_02_HMI[3], out1 => "DB2099_MANUAL_LOAD_DMC".DMC_ARRAY_CHAR_UNIT_02[42])
      Contact( "M_DUMMY_OFF" )
      Move(in := "DB2099_MANUAL_LOAD_DMC".DMC_UNIT_02_HMI[3], out1 => "DB2099_MANUAL_LOAD_DMC".DMC_ARRAY_CHAR_UNIT_02[35])
   END_RUNG
   RUNG wire#w1
      { S7_Templates := "SrcType := Char" } NE_Contact(in1 := "DB2099_MANUAL_LOAD_DMC".DMC_UNIT_02_HMI[4], in2 := '$00')
      Contact( "M_DUMMY_ON" )
      Move(in := "DB2099_MANUAL_LOAD_DMC".DMC_UNIT_02_HMI[4], out1 => "DB2099_MANUAL_LOAD_DMC".DMC_ARRAY_CHAR_UNIT_02[43])
      Contact( "M_DUMMY_OFF" )
      Move(in := "DB2099_MANUAL_LOAD_DMC".DMC_UNIT_02_HMI[4], out1 => "DB2099_MANUAL_LOAD_DMC".DMC_ARRAY_CHAR_UNIT_02[36])
   END_RUNG
   RUNG wire#w1
      { S7_Templates := "SrcType := Char" } NE_Contact(in1 := "DB2099_MANUAL_LOAD_DMC".DMC_UNIT_02_HMI[5], in2 := '$00')
      Contact( "M_DUMMY_ON" )
      Move(in := "DB2099_MANUAL_LOAD_DMC".DMC_UNIT_02_HMI[5], out1 => "DB2099_MANUAL_LOAD_DMC".DMC_ARRAY_CHAR_UNIT_02[44])
      Contact( "M_DUMMY_OFF" )
      Move(in := "DB2099_MANUAL_LOAD_DMC".DMC_UNIT_02_HMI[4], out1 => "DB2099_MANUAL_LOAD_DMC".DMC_ARRAY_CHAR_UNIT_02[37])
   END_RUNG
   RUNG wire#w1
      { S7_Templates := "SrcType := Char" } NE_Contact(in1 := "DB2099_MANUAL_LOAD_DMC".DMC_UNIT_02_HMI[6], in2 := '$00')
      Contact( "M_DUMMY_ON" )
      Move(in := "DB2099_MANUAL_LOAD_DMC".DMC_UNIT_02_HMI[6], out1 => "DB2099_MANUAL_LOAD_DMC".DMC_ARRAY_CHAR_UNIT_02[45])
      Contact( "M_DUMMY_OFF" )
      Move(in := "DB2099_MANUAL_LOAD_DMC".DMC_UNIT_02_HMI[4], out1 => "DB2099_MANUAL_LOAD_DMC".DMC_ARRAY_CHAR_UNIT_02[38])
   END_RUNG
   RUNG wire#w1
      { S7_Templates := "SrcType := Char" } NE_Contact(in1 := "DB2099_MANUAL_LOAD_DMC".DMC_UNIT_02_HMI[7], in2 := '$00')
      Contact( "M_DUMMY_ON" )
      Move(in := "DB2099_MANUAL_LOAD_DMC".DMC_UNIT_02_HMI[7], out1 => "DB2099_MANUAL_LOAD_DMC".DMC_ARRAY_CHAR_UNIT_02[46])
      Contact( "M_DUMMY_OFF" )
      Move(in := "DB2099_MANUAL_LOAD_DMC".DMC_UNIT_02_HMI[4], out1 => "DB2099_MANUAL_LOAD_DMC".DMC_ARRAY_CHAR_UNIT_02[39])
   END_RUNG
   RUNG wire#w1
      Contact( "M_DUMMY_ON" )
      Move(in := '$00', out1 => "DB2099_MANUAL_LOAD_DMC".DMC_ARRAY_CHAR_UNIT_02[48])
      Contact( "M_DUMMY_OFF" )
      Move(in := '$00', out1 => "DB2099_MANUAL_LOAD_DMC".DMC_ARRAY_CHAR_UNIT_02[45])
   END_RUNG
   // the same network as SCL:
   #_w1 := "DB2031_CYCLES_GENERAL".MANUAL_LOAD_CYCLE.CYCLE_SELECTED AND NOT "DB2099_MANUAL_LOAD_DMC".PRODUCTION_SELECTED;
   IF #_w1 AND "M_DUMMY_ON" THEN
       "DB2099_MANUAL_LOAD_DMC".DMC_STRING_UNIT_02 := '#0001#TYPE01#DDDDDDDDD#010124*065 KTOxxxxxxxP*';
   END_IF;
   IF #_w1 AND "M_DUMMY_OFF" AND "DB7215_PART_TYPE".PART_TYPE_01_SELECTED THEN
       "DB2099_MANUAL_LOAD_DMC".DMC_STRING_UNIT_02 := '#5WA615301C    ###210125*657 VWA4PALA0L5*=';
   END_IF;
   IF #_w1 AND "M_DUMMY_OFF" AND "DB7215_PART_TYPE".PART_TYPE_02_SELECTED THEN
       "DB2099_MANUAL_LOAD_DMC".DMC_STRING_UNIT_02 := '#5WA615301E    ###210125*657 VWA4PALA0L5*=';
   END_IF;
   IF #_w1 THEN
       Strg_TO_Chars(Strg := "DB2099_MANUAL_LOAD_DMC".DMC_STRING_UNIT_02,
                     pChars := 0,
                     Chars := "DB2099_MANUAL_LOAD_DMC".DMC_ARRAY_CHAR_UNIT_02,
                     Cnt => "DB2099_MANUAL_LOAD_DMC".AUX_CNT_INT_UNIT_02);
   END_IF;
   #_w2 := #_w1 AND ("DB2099_MANUAL_LOAD_DMC".DMC_UNIT_02_HMI[0] <> '$00') AND "M_DUMMY_ON";
   IF #_w2 THEN
       "DB2099_MANUAL_LOAD_DMC".DMC_ARRAY_CHAR_UNIT_02[39] := "DB2099_MANUAL_LOAD_DMC".DMC_UNIT_02_HMI[0];
   END_IF;
   IF #_w2 AND "M_DUMMY_OFF" THEN
       "DB2099_MANUAL_LOAD_DMC".DMC_ARRAY_CHAR_UNIT_02[32] := "DB2099_MANUAL_LOAD_DMC".DMC_UNIT_02_HMI[0];
   END_IF;
   #_w3 := #_w1 AND ("DB2099_MANUAL_LOAD_DMC".DMC_UNIT_02_HMI[1] <> '$00') AND "M_DUMMY_ON";
   IF #_w3 THEN
       "DB2099_MANUAL_LOAD_DMC".DMC_ARRAY_CHAR_UNIT_02[40] := "DB2099_MANUAL_LOAD_DMC".DMC_UNIT_02_HMI[1];
   END_IF;
   IF #_w3 AND "M_DUMMY_OFF" THEN
       "DB2099_MANUAL_LOAD_DMC".DMC_ARRAY_CHAR_UNIT_02[33] := "DB2099_MANUAL_LOAD_DMC".DMC_UNIT_02_HMI[1];
   END_IF;
   #_w4 := #_w1 AND ("DB2099_MANUAL_LOAD_DMC".DMC_UNIT_02_HMI[2] <> '$00') AND "M_DUMMY_ON";
   IF #_w4 THEN
       "DB2099_MANUAL_LOAD_DMC".DMC_ARRAY_CHAR_UNIT_02[41] := "DB2099_MANUAL_LOAD_DMC".DMC_UNIT_02_HMI[2];
   END_IF;
   IF #_w4 AND "M_DUMMY_OFF" THEN
       "DB2099_MANUAL_LOAD_DMC".DMC_ARRAY_CHAR_UNIT_02[34] := "DB2099_MANUAL_LOAD_DMC".DMC_UNIT_02_HMI[2];
   END_IF;
   #_w5 := #_w1 AND ("DB2099_MANUAL_LOAD_DMC".DMC_UNIT_02_HMI[3] <> '$00') AND "M_DUMMY_ON";
   IF #_w5 THEN
       "DB2099_MANUAL_LOAD_DMC".DMC_ARRAY_CHAR_UNIT_02[42] := "DB2099_MANUAL_LOAD_DMC".DMC_UNIT_02_HMI[3];
   END_IF;
   IF #_w5 AND "M_DUMMY_OFF" THEN
       "DB2099_MANUAL_LOAD_DMC".DMC_ARRAY_CHAR_UNIT_02[35] := "DB2099_MANUAL_LOAD_DMC".DMC_UNIT_02_HMI[3];
   END_IF;
   #_w6 := #_w1 AND ("DB2099_MANUAL_LOAD_DMC".DMC_UNIT_02_HMI[4] <> '$00') AND "M_DUMMY_ON";
   IF #_w6 THEN
       "DB2099_MANUAL_LOAD_DMC".DMC_ARRAY_CHAR_UNIT_02[43] := "DB2099_MANUAL_LOAD_DMC".DMC_UNIT_02_HMI[4];
   END_IF;
   IF #_w6 AND "M_DUMMY_OFF" THEN
       "DB2099_MANUAL_LOAD_DMC".DMC_ARRAY_CHAR_UNIT_02[36] := "DB2099_MANUAL_LOAD_DMC".DMC_UNIT_02_HMI[4];
   END_IF;
   #_w7 := #_w1 AND ("DB2099_MANUAL_LOAD_DMC".DMC_UNIT_02_HMI[5] <> '$00') AND "M_DUMMY_ON";
   IF #_w7 THEN
       "DB2099_MANUAL_LOAD_DMC".DMC_ARRAY_CHAR_UNIT_02[44] := "DB2099_MANUAL_LOAD_DMC".DMC_UNIT_02_HMI[5];
   END_IF;
   IF #_w7 AND "M_DUMMY_OFF" THEN
       "DB2099_MANUAL_LOAD_DMC".DMC_ARRAY_CHAR_UNIT_02[37] := "DB2099_MANUAL_LOAD_DMC".DMC_UNIT_02_HMI[4];
   END_IF;
   #_w8 := #_w1 AND ("DB2099_MANUAL_LOAD_DMC".DMC_UNIT_02_HMI[6] <> '$00') AND "M_DUMMY_ON";
   IF #_w8 THEN
       "DB2099_MANUAL_LOAD_DMC".DMC_ARRAY_CHAR_UNIT_02[45] := "DB2099_MANUAL_LOAD_DMC".DMC_UNIT_02_HMI[6];
   END_IF;
   IF #_w8 AND "M_DUMMY_OFF" THEN
       "DB2099_MANUAL_LOAD_DMC".DMC_ARRAY_CHAR_UNIT_02[38] := "DB2099_MANUAL_LOAD_DMC".DMC_UNIT_02_HMI[4];
   END_IF;
   #_w9 := #_w1 AND ("DB2099_MANUAL_LOAD_DMC".DMC_UNIT_02_HMI[7] <> '$00') AND "M_DUMMY_ON";
   IF #_w9 THEN
       "DB2099_MANUAL_LOAD_DMC".DMC_ARRAY_CHAR_UNIT_02[46] := "DB2099_MANUAL_LOAD_DMC".DMC_UNIT_02_HMI[7];
   END_IF;
   IF #_w9 AND "M_DUMMY_OFF" THEN
       "DB2099_MANUAL_LOAD_DMC".DMC_ARRAY_CHAR_UNIT_02[39] := "DB2099_MANUAL_LOAD_DMC".DMC_UNIT_02_HMI[4];
   END_IF;
   #_w10 := #_w1 AND "M_DUMMY_ON";
   IF #_w10 THEN "DB2099_MANUAL_LOAD_DMC".DMC_ARRAY_CHAR_UNIT_02[48] := '$00'; END_IF;
   IF #_w10 AND "M_DUMMY_OFF" THEN "DB2099_MANUAL_LOAD_DMC".DMC_ARRAY_CHAR_UNIT_02[45] := '$00'; END_IF;
END_REGION

REGION Network 18: PART DMC UNIT 01 WRITING FOR MANUAL LOADING & PRODUCTION SELECTED
   // M0.2 CUANDO SE DECIDA CON LEON CAMBIAR LA ESTRUCTURA DEL DMC SOLO HARA FALTA BORRAR LO QUE ESTÁ TRAS M0.2 Y BORRAR EL M0.3 PARA QUE SE EJECUTE EL NUEVO CODIGO. DE LO CONTRARIO SUSTITUIR M0.2 POR M0.3 Y VICEVERSA
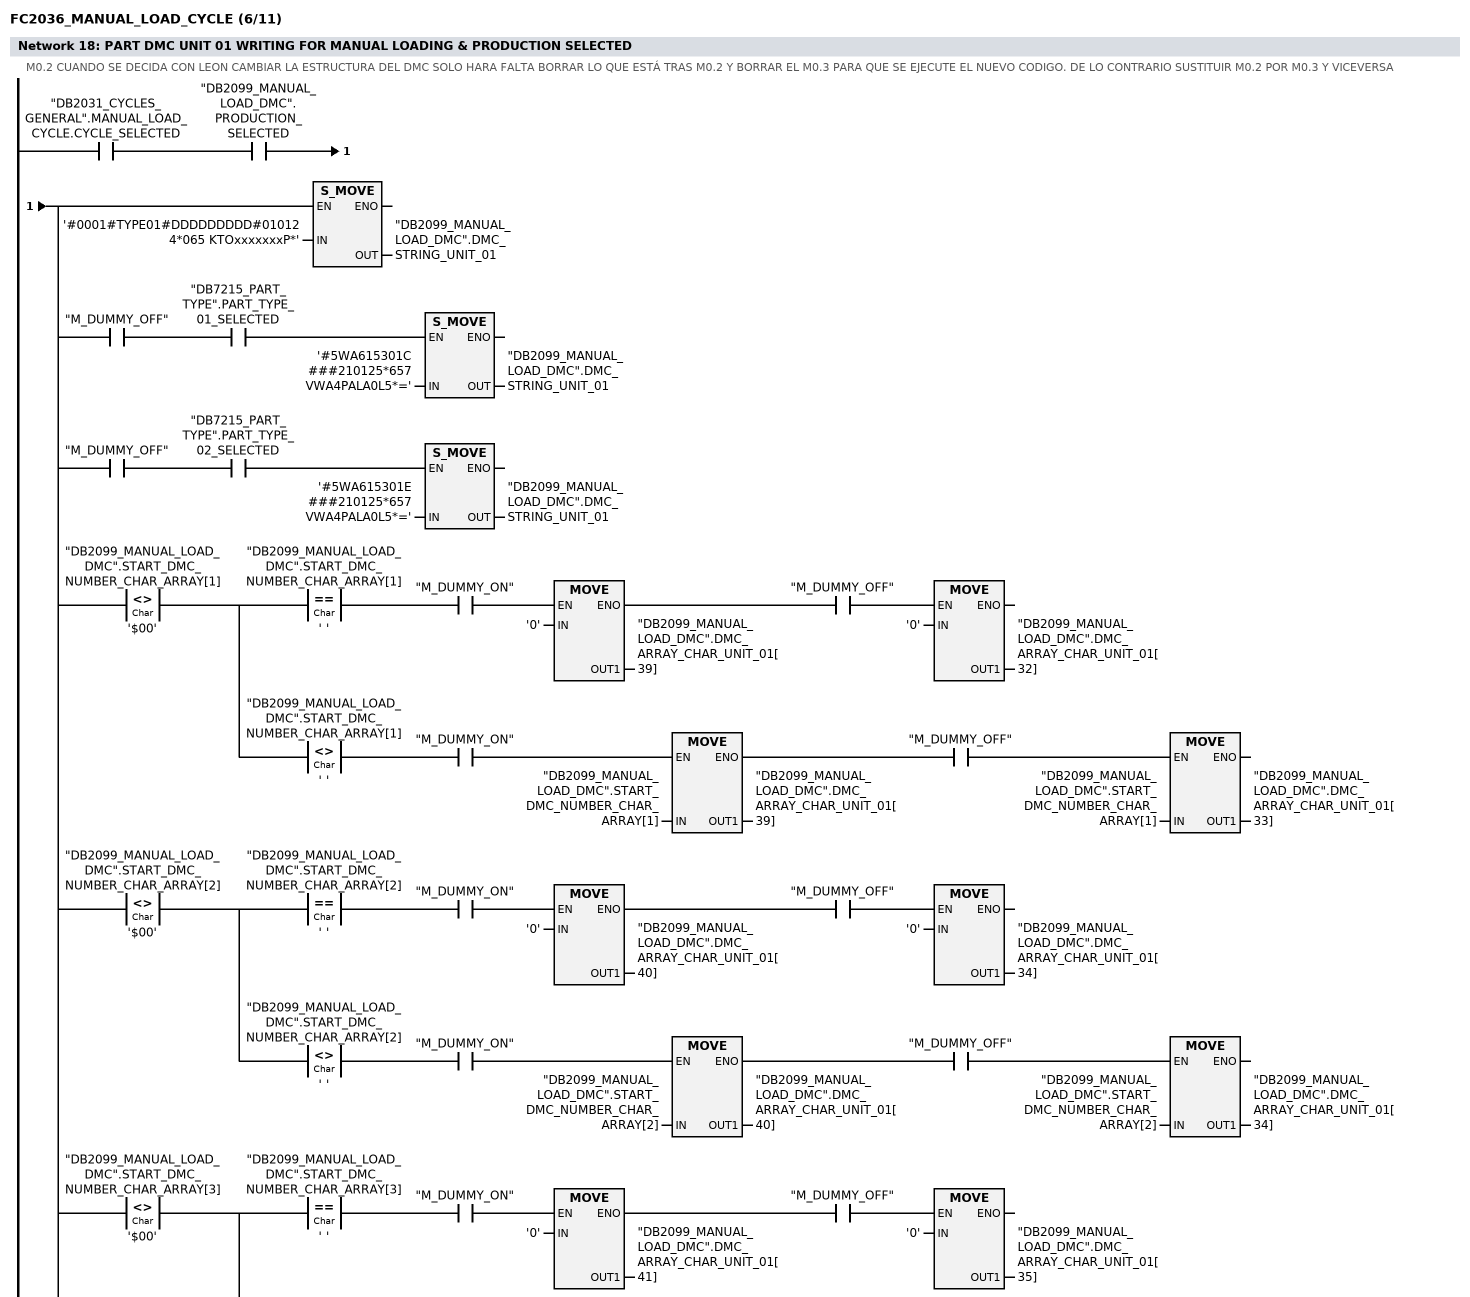
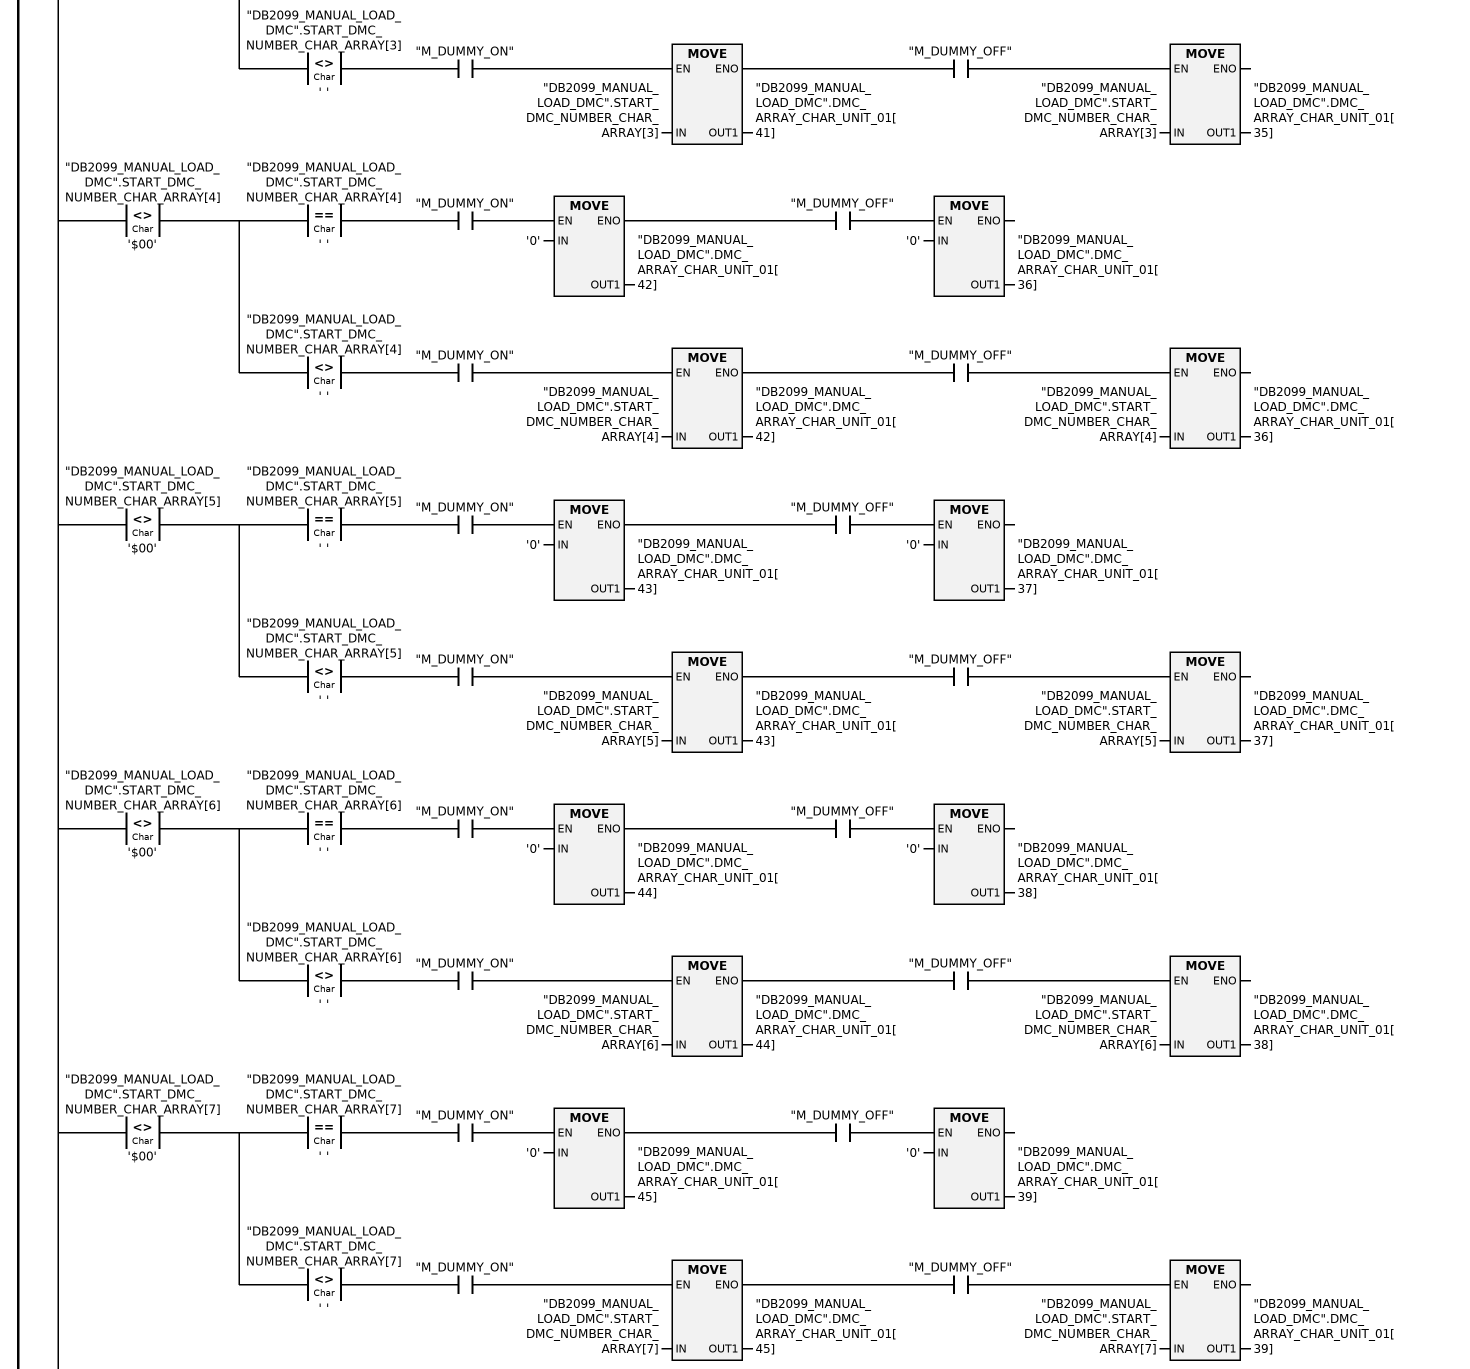
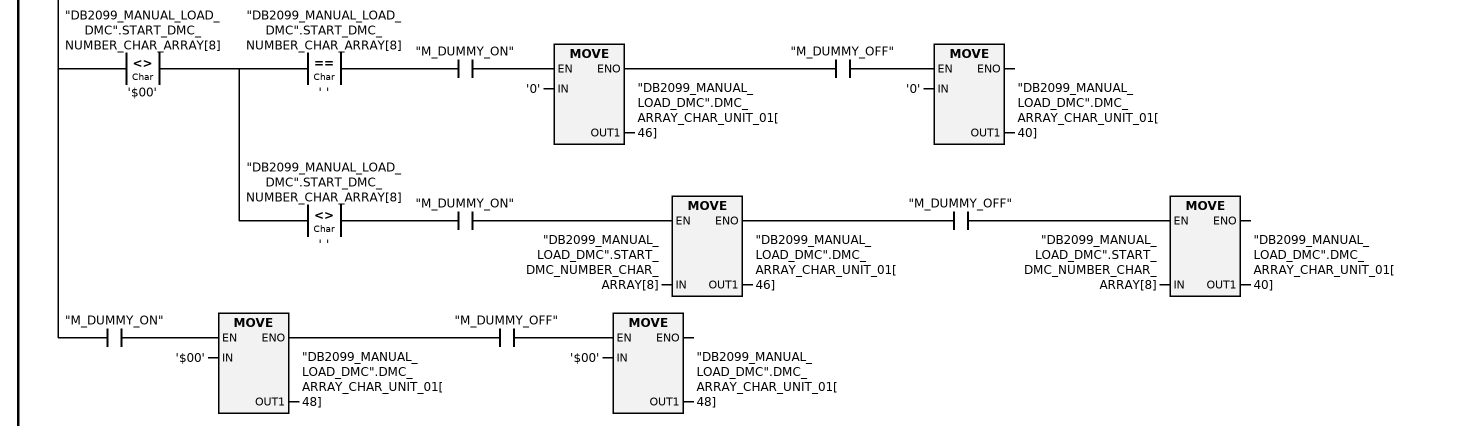
   RUNG wire#powerrail
      Contact( "DB2031_CYCLES_GENERAL".MANUAL_LOAD_CYCLE.CYCLE_SELECTED )
      Contact( "DB2099_MANUAL_LOAD_DMC".PRODUCTION_SELECTED )
      wire#w1
      S_Move(in := '#0001#TYPE01#DDDDDDDDD#010124*065 KTOxxxxxxxP*', out => "DB2099_MANUAL_LOAD_DMC".DMC_STRING_UNIT_01)
   END_RUNG
   RUNG wire#w1
      Contact( "M_DUMMY_OFF" )
      Contact( "DB7215_PART_TYPE".PART_TYPE_01_SELECTED )
      S_Move(in := '#5WA615301C    ###210125*657 VWA4PALA0L5*=', out => "DB2099_MANUAL_LOAD_DMC".DMC_STRING_UNIT_01)
   END_RUNG
   RUNG wire#w1
      Contact( "M_DUMMY_OFF" )
      Contact( "DB7215_PART_TYPE".PART_TYPE_02_SELECTED )
      S_Move(in := '#5WA615301E    ###210125*657 VWA4PALA0L5*=', out => "DB2099_MANUAL_LOAD_DMC".DMC_STRING_UNIT_01)
   END_RUNG
   RUNG wire#w1
      { S7_Templates := "SrcType := Char" } NE_Contact(in1 := "DB2099_MANUAL_LOAD_DMC".START_DMC_NUMBER_CHAR_ARRAY[1], in2 := '$00')
      wire#w2
      { S7_Templates := "SrcType := Char" } EQ_Contact(in1 := "DB2099_MANUAL_LOAD_DMC".START_DMC_NUMBER_CHAR_ARRAY[1], in2 := ' ')
      Contact( "M_DUMMY_ON" )
      Move(in := '0', out1 => "DB2099_MANUAL_LOAD_DMC".DMC_ARRAY_CHAR_UNIT_01[39])
      Contact( "M_DUMMY_OFF" )
      Move(in := '0', out1 => "DB2099_MANUAL_LOAD_DMC".DMC_ARRAY_CHAR_UNIT_01[32])
   END_RUNG
   RUNG wire#w2
      { S7_Templates := "SrcType := Char" } NE_Contact(in1 := "DB2099_MANUAL_LOAD_DMC".START_DMC_NUMBER_CHAR_ARRAY[1], in2 := ' ')
      Contact( "M_DUMMY_ON" )
      Move(in := "DB2099_MANUAL_LOAD_DMC".START_DMC_NUMBER_CHAR_ARRAY[1], out1 => "DB2099_MANUAL_LOAD_DMC".DMC_ARRAY_CHAR_UNIT_01[39])
      Contact( "M_DUMMY_OFF" )
      Move(in := "DB2099_MANUAL_LOAD_DMC".START_DMC_NUMBER_CHAR_ARRAY[1], out1 => "DB2099_MANUAL_LOAD_DMC".DMC_ARRAY_CHAR_UNIT_01[33])
   END_RUNG
   RUNG wire#w1
      { S7_Templates := "SrcType := Char" } NE_Contact(in1 := "DB2099_MANUAL_LOAD_DMC".START_DMC_NUMBER_CHAR_ARRAY[2], in2 := '$00')
      wire#w3
      { S7_Templates := "SrcType := Char" } EQ_Contact(in1 := "DB2099_MANUAL_LOAD_DMC".START_DMC_NUMBER_CHAR_ARRAY[2], in2 := ' ')
      Contact( "M_DUMMY_ON" )
      Move(in := '0', out1 => "DB2099_MANUAL_LOAD_DMC".DMC_ARRAY_CHAR_UNIT_01[40])
      Contact( "M_DUMMY_OFF" )
      Move(in := '0', out1 => "DB2099_MANUAL_LOAD_DMC".DMC_ARRAY_CHAR_UNIT_01[34])
   END_RUNG
   RUNG wire#w3
      { S7_Templates := "SrcType := Char" } NE_Contact(in1 := "DB2099_MANUAL_LOAD_DMC".START_DMC_NUMBER_CHAR_ARRAY[2], in2 := ' ')
      Contact( "M_DUMMY_ON" )
      Move(in := "DB2099_MANUAL_LOAD_DMC".START_DMC_NUMBER_CHAR_ARRAY[2], out1 => "DB2099_MANUAL_LOAD_DMC".DMC_ARRAY_CHAR_UNIT_01[40])
      Contact( "M_DUMMY_OFF" )
      Move(in := "DB2099_MANUAL_LOAD_DMC".START_DMC_NUMBER_CHAR_ARRAY[2], out1 => "DB2099_MANUAL_LOAD_DMC".DMC_ARRAY_CHAR_UNIT_01[34])
   END_RUNG
   RUNG wire#w1
      { S7_Templates := "SrcType := Char" } NE_Contact(in1 := "DB2099_MANUAL_LOAD_DMC".START_DMC_NUMBER_CHAR_ARRAY[3], in2 := '$00')
      wire#w4
      { S7_Templates := "SrcType := Char" } EQ_Contact(in1 := "DB2099_MANUAL_LOAD_DMC".START_DMC_NUMBER_CHAR_ARRAY[3], in2 := ' ')
      Contact( "M_DUMMY_ON" )
      Move(in := '0', out1 => "DB2099_MANUAL_LOAD_DMC".DMC_ARRAY_CHAR_UNIT_01[41])
      Contact( "M_DUMMY_OFF" )
      Move(in := '0', out1 => "DB2099_MANUAL_LOAD_DMC".DMC_ARRAY_CHAR_UNIT_01[35])
   END_RUNG
   RUNG wire#w4
      { S7_Templates := "SrcType := Char" } NE_Contact(in1 := "DB2099_MANUAL_LOAD_DMC".START_DMC_NUMBER_CHAR_ARRAY[3], in2 := ' ')
      Contact( "M_DUMMY_ON" )
      Move(in := "DB2099_MANUAL_LOAD_DMC".START_DMC_NUMBER_CHAR_ARRAY[3], out1 => "DB2099_MANUAL_LOAD_DMC".DMC_ARRAY_CHAR_UNIT_01[41])
      Contact( "M_DUMMY_OFF" )
      Move(in := "DB2099_MANUAL_LOAD_DMC".START_DMC_NUMBER_CHAR_ARRAY[3], out1 => "DB2099_MANUAL_LOAD_DMC".DMC_ARRAY_CHAR_UNIT_01[35])
   END_RUNG
   RUNG wire#w1
      { S7_Templates := "SrcType := Char" } NE_Contact(in1 := "DB2099_MANUAL_LOAD_DMC".START_DMC_NUMBER_CHAR_ARRAY[4], in2 := '$00')
      wire#w5
      { S7_Templates := "SrcType := Char" } EQ_Contact(in1 := "DB2099_MANUAL_LOAD_DMC".START_DMC_NUMBER_CHAR_ARRAY[4], in2 := ' ')
      Contact( "M_DUMMY_ON" )
      Move(in := '0', out1 => "DB2099_MANUAL_LOAD_DMC".DMC_ARRAY_CHAR_UNIT_01[42])
      Contact( "M_DUMMY_OFF" )
      Move(in := '0', out1 => "DB2099_MANUAL_LOAD_DMC".DMC_ARRAY_CHAR_UNIT_01[36])
   END_RUNG
   RUNG wire#w5
      { S7_Templates := "SrcType := Char" } NE_Contact(in1 := "DB2099_MANUAL_LOAD_DMC".START_DMC_NUMBER_CHAR_ARRAY[4], in2 := ' ')
      Contact( "M_DUMMY_ON" )
      Move(in := "DB2099_MANUAL_LOAD_DMC".START_DMC_NUMBER_CHAR_ARRAY[4], out1 => "DB2099_MANUAL_LOAD_DMC".DMC_ARRAY_CHAR_UNIT_01[42])
      Contact( "M_DUMMY_OFF" )
      Move(in := "DB2099_MANUAL_LOAD_DMC".START_DMC_NUMBER_CHAR_ARRAY[4], out1 => "DB2099_MANUAL_LOAD_DMC".DMC_ARRAY_CHAR_UNIT_01[36])
   END_RUNG
   RUNG wire#w1
      { S7_Templates := "SrcType := Char" } NE_Contact(in1 := "DB2099_MANUAL_LOAD_DMC".START_DMC_NUMBER_CHAR_ARRAY[5], in2 := '$00')
      wire#w6
      { S7_Templates := "SrcType := Char" } EQ_Contact(in1 := "DB2099_MANUAL_LOAD_DMC".START_DMC_NUMBER_CHAR_ARRAY[5], in2 := ' ')
      Contact( "M_DUMMY_ON" )
      Move(in := '0', out1 => "DB2099_MANUAL_LOAD_DMC".DMC_ARRAY_CHAR_UNIT_01[43])
      Contact( "M_DUMMY_OFF" )
      Move(in := '0', out1 => "DB2099_MANUAL_LOAD_DMC".DMC_ARRAY_CHAR_UNIT_01[37])
   END_RUNG
   RUNG wire#w6
      { S7_Templates := "SrcType := Char" } NE_Contact(in1 := "DB2099_MANUAL_LOAD_DMC".START_DMC_NUMBER_CHAR_ARRAY[5], in2 := ' ')
      Contact( "M_DUMMY_ON" )
      Move(in := "DB2099_MANUAL_LOAD_DMC".START_DMC_NUMBER_CHAR_ARRAY[5], out1 => "DB2099_MANUAL_LOAD_DMC".DMC_ARRAY_CHAR_UNIT_01[43])
      Contact( "M_DUMMY_OFF" )
      Move(in := "DB2099_MANUAL_LOAD_DMC".START_DMC_NUMBER_CHAR_ARRAY[5], out1 => "DB2099_MANUAL_LOAD_DMC".DMC_ARRAY_CHAR_UNIT_01[37])
   END_RUNG
   RUNG wire#w1
      { S7_Templates := "SrcType := Char" } NE_Contact(in1 := "DB2099_MANUAL_LOAD_DMC".START_DMC_NUMBER_CHAR_ARRAY[6], in2 := '$00')
      wire#w7
      { S7_Templates := "SrcType := Char" } EQ_Contact(in1 := "DB2099_MANUAL_LOAD_DMC".START_DMC_NUMBER_CHAR_ARRAY[6], in2 := ' ')
      Contact( "M_DUMMY_ON" )
      Move(in := '0', out1 => "DB2099_MANUAL_LOAD_DMC".DMC_ARRAY_CHAR_UNIT_01[44])
      Contact( "M_DUMMY_OFF" )
      Move(in := '0', out1 => "DB2099_MANUAL_LOAD_DMC".DMC_ARRAY_CHAR_UNIT_01[38])
   END_RUNG
   RUNG wire#w7
      { S7_Templates := "SrcType := Char" } NE_Contact(in1 := "DB2099_MANUAL_LOAD_DMC".START_DMC_NUMBER_CHAR_ARRAY[6], in2 := ' ')
      Contact( "M_DUMMY_ON" )
      Move(in := "DB2099_MANUAL_LOAD_DMC".START_DMC_NUMBER_CHAR_ARRAY[6], out1 => "DB2099_MANUAL_LOAD_DMC".DMC_ARRAY_CHAR_UNIT_01[44])
      Contact( "M_DUMMY_OFF" )
      Move(in := "DB2099_MANUAL_LOAD_DMC".START_DMC_NUMBER_CHAR_ARRAY[6], out1 => "DB2099_MANUAL_LOAD_DMC".DMC_ARRAY_CHAR_UNIT_01[38])
   END_RUNG
   RUNG wire#w1
      { S7_Templates := "SrcType := Char" } NE_Contact(in1 := "DB2099_MANUAL_LOAD_DMC".START_DMC_NUMBER_CHAR_ARRAY[7], in2 := '$00')
      wire#w8
      { S7_Templates := "SrcType := Char" } EQ_Contact(in1 := "DB2099_MANUAL_LOAD_DMC".START_DMC_NUMBER_CHAR_ARRAY[7], in2 := ' ')
      Contact( "M_DUMMY_ON" )
      Move(in := '0', out1 => "DB2099_MANUAL_LOAD_DMC".DMC_ARRAY_CHAR_UNIT_01[45])
      Contact( "M_DUMMY_OFF" )
      Move(in := '0', out1 => "DB2099_MANUAL_LOAD_DMC".DMC_ARRAY_CHAR_UNIT_01[39])
   END_RUNG
   RUNG wire#w8
      { S7_Templates := "SrcType := Char" } NE_Contact(in1 := "DB2099_MANUAL_LOAD_DMC".START_DMC_NUMBER_CHAR_ARRAY[7], in2 := ' ')
      Contact( "M_DUMMY_ON" )
      Move(in := "DB2099_MANUAL_LOAD_DMC".START_DMC_NUMBER_CHAR_ARRAY[7], out1 => "DB2099_MANUAL_LOAD_DMC".DMC_ARRAY_CHAR_UNIT_01[45])
      Contact( "M_DUMMY_OFF" )
      Move(in := "DB2099_MANUAL_LOAD_DMC".START_DMC_NUMBER_CHAR_ARRAY[7], out1 => "DB2099_MANUAL_LOAD_DMC".DMC_ARRAY_CHAR_UNIT_01[39])
   END_RUNG
   RUNG wire#w1
      { S7_Templates := "SrcType := Char" } NE_Contact(in1 := "DB2099_MANUAL_LOAD_DMC".START_DMC_NUMBER_CHAR_ARRAY[8], in2 := '$00')
      wire#w9
      { S7_Templates := "SrcType := Char" } EQ_Contact(in1 := "DB2099_MANUAL_LOAD_DMC".START_DMC_NUMBER_CHAR_ARRAY[8], in2 := ' ')
      Contact( "M_DUMMY_ON" )
      Move(in := '0', out1 => "DB2099_MANUAL_LOAD_DMC".DMC_ARRAY_CHAR_UNIT_01[46])
      Contact( "M_DUMMY_OFF" )
      Move(in := '0', out1 => "DB2099_MANUAL_LOAD_DMC".DMC_ARRAY_CHAR_UNIT_01[40])
   END_RUNG
   RUNG wire#w9
      { S7_Templates := "SrcType := Char" } NE_Contact(in1 := "DB2099_MANUAL_LOAD_DMC".START_DMC_NUMBER_CHAR_ARRAY[8], in2 := ' ')
      Contact( "M_DUMMY_ON" )
      Move(in := "DB2099_MANUAL_LOAD_DMC".START_DMC_NUMBER_CHAR_ARRAY[8], out1 => "DB2099_MANUAL_LOAD_DMC".DMC_ARRAY_CHAR_UNIT_01[46])
      Contact( "M_DUMMY_OFF" )
      Move(in := "DB2099_MANUAL_LOAD_DMC".START_DMC_NUMBER_CHAR_ARRAY[8], out1 => "DB2099_MANUAL_LOAD_DMC".DMC_ARRAY_CHAR_UNIT_01[40])
   END_RUNG
   RUNG wire#w1
      Contact( "M_DUMMY_ON" )
      Move(in := '$00', out1 => "DB2099_MANUAL_LOAD_DMC".DMC_ARRAY_CHAR_UNIT_01[48])
      Contact( "M_DUMMY_OFF" )
      Move(in := '$00', out1 => "DB2099_MANUAL_LOAD_DMC".DMC_ARRAY_CHAR_UNIT_01[48])
   END_RUNG
   // the same network as SCL:
   #_w1 := "DB2031_CYCLES_GENERAL".MANUAL_LOAD_CYCLE.CYCLE_SELECTED AND "DB2099_MANUAL_LOAD_DMC".PRODUCTION_SELECTED;
   IF #_w1 THEN
       "DB2099_MANUAL_LOAD_DMC".DMC_STRING_UNIT_01 := '#0001#TYPE01#DDDDDDDDD#010124*065 KTOxxxxxxxP*';
   END_IF;
   IF #_w1 AND "M_DUMMY_OFF" AND "DB7215_PART_TYPE".PART_TYPE_01_SELECTED THEN
       "DB2099_MANUAL_LOAD_DMC".DMC_STRING_UNIT_01 := '#5WA615301C    ###210125*657 VWA4PALA0L5*=';
   END_IF;
   IF #_w1 AND "M_DUMMY_OFF" AND "DB7215_PART_TYPE".PART_TYPE_02_SELECTED THEN
       "DB2099_MANUAL_LOAD_DMC".DMC_STRING_UNIT_01 := '#5WA615301E    ###210125*657 VWA4PALA0L5*=';
   END_IF;
   #_w2 := #_w1 AND ("DB2099_MANUAL_LOAD_DMC".START_DMC_NUMBER_CHAR_ARRAY[1] <> '$00');
   #_w3 := #_w2 AND ("DB2099_MANUAL_LOAD_DMC".START_DMC_NUMBER_CHAR_ARRAY[1] = ' ') AND "M_DUMMY_ON";
   IF #_w3 THEN "DB2099_MANUAL_LOAD_DMC".DMC_ARRAY_CHAR_UNIT_01[39] := '0'; END_IF;
   IF #_w3 AND "M_DUMMY_OFF" THEN "DB2099_MANUAL_LOAD_DMC".DMC_ARRAY_CHAR_UNIT_01[32] := '0'; END_IF;
   #_w4 := #_w2 AND ("DB2099_MANUAL_LOAD_DMC".START_DMC_NUMBER_CHAR_ARRAY[1] <> ' ') AND "M_DUMMY_ON";
   IF #_w4 THEN
       "DB2099_MANUAL_LOAD_DMC".DMC_ARRAY_CHAR_UNIT_01[39] := "DB2099_MANUAL_LOAD_DMC".START_DMC_NUMBER_CHAR_ARRAY[1];
   END_IF;
   IF #_w4 AND "M_DUMMY_OFF" THEN
       "DB2099_MANUAL_LOAD_DMC".DMC_ARRAY_CHAR_UNIT_01[33] := "DB2099_MANUAL_LOAD_DMC".START_DMC_NUMBER_CHAR_ARRAY[1];
   END_IF;
   #_w5 := #_w1 AND ("DB2099_MANUAL_LOAD_DMC".START_DMC_NUMBER_CHAR_ARRAY[2] <> '$00');
   #_w6 := #_w5 AND ("DB2099_MANUAL_LOAD_DMC".START_DMC_NUMBER_CHAR_ARRAY[2] = ' ') AND "M_DUMMY_ON";
   IF #_w6 THEN "DB2099_MANUAL_LOAD_DMC".DMC_ARRAY_CHAR_UNIT_01[40] := '0'; END_IF;
   IF #_w6 AND "M_DUMMY_OFF" THEN "DB2099_MANUAL_LOAD_DMC".DMC_ARRAY_CHAR_UNIT_01[34] := '0'; END_IF;
   #_w7 := #_w5 AND ("DB2099_MANUAL_LOAD_DMC".START_DMC_NUMBER_CHAR_ARRAY[2] <> ' ') AND "M_DUMMY_ON";
   IF #_w7 THEN
       "DB2099_MANUAL_LOAD_DMC".DMC_ARRAY_CHAR_UNIT_01[40] := "DB2099_MANUAL_LOAD_DMC".START_DMC_NUMBER_CHAR_ARRAY[2];
   END_IF;
   IF #_w7 AND "M_DUMMY_OFF" THEN
       "DB2099_MANUAL_LOAD_DMC".DMC_ARRAY_CHAR_UNIT_01[34] := "DB2099_MANUAL_LOAD_DMC".START_DMC_NUMBER_CHAR_ARRAY[2];
   END_IF;
   #_w8 := #_w1 AND ("DB2099_MANUAL_LOAD_DMC".START_DMC_NUMBER_CHAR_ARRAY[3] <> '$00');
   #_w9 := #_w8 AND ("DB2099_MANUAL_LOAD_DMC".START_DMC_NUMBER_CHAR_ARRAY[3] = ' ') AND "M_DUMMY_ON";
   IF #_w9 THEN "DB2099_MANUAL_LOAD_DMC".DMC_ARRAY_CHAR_UNIT_01[41] := '0'; END_IF;
   IF #_w9 AND "M_DUMMY_OFF" THEN "DB2099_MANUAL_LOAD_DMC".DMC_ARRAY_CHAR_UNIT_01[35] := '0'; END_IF;
   #_w10 := #_w8 AND ("DB2099_MANUAL_LOAD_DMC".START_DMC_NUMBER_CHAR_ARRAY[3] <> ' ') AND "M_DUMMY_ON";
   IF #_w10 THEN
       "DB2099_MANUAL_LOAD_DMC".DMC_ARRAY_CHAR_UNIT_01[41] := "DB2099_MANUAL_LOAD_DMC".START_DMC_NUMBER_CHAR_ARRAY[3];
   END_IF;
   IF #_w10 AND "M_DUMMY_OFF" THEN
       "DB2099_MANUAL_LOAD_DMC".DMC_ARRAY_CHAR_UNIT_01[35] := "DB2099_MANUAL_LOAD_DMC".START_DMC_NUMBER_CHAR_ARRAY[3];
   END_IF;
   #_w11 := #_w1 AND ("DB2099_MANUAL_LOAD_DMC".START_DMC_NUMBER_CHAR_ARRAY[4] <> '$00');
   #_w12 := #_w11 AND ("DB2099_MANUAL_LOAD_DMC".START_DMC_NUMBER_CHAR_ARRAY[4] = ' ') AND "M_DUMMY_ON";
   IF #_w12 THEN "DB2099_MANUAL_LOAD_DMC".DMC_ARRAY_CHAR_UNIT_01[42] := '0'; END_IF;
   IF #_w12 AND "M_DUMMY_OFF" THEN "DB2099_MANUAL_LOAD_DMC".DMC_ARRAY_CHAR_UNIT_01[36] := '0'; END_IF;
   #_w13 := #_w11 AND ("DB2099_MANUAL_LOAD_DMC".START_DMC_NUMBER_CHAR_ARRAY[4] <> ' ') AND "M_DUMMY_ON";
   IF #_w13 THEN
       "DB2099_MANUAL_LOAD_DMC".DMC_ARRAY_CHAR_UNIT_01[42] := "DB2099_MANUAL_LOAD_DMC".START_DMC_NUMBER_CHAR_ARRAY[4];
   END_IF;
   IF #_w13 AND "M_DUMMY_OFF" THEN
       "DB2099_MANUAL_LOAD_DMC".DMC_ARRAY_CHAR_UNIT_01[36] := "DB2099_MANUAL_LOAD_DMC".START_DMC_NUMBER_CHAR_ARRAY[4];
   END_IF;
   #_w14 := #_w1 AND ("DB2099_MANUAL_LOAD_DMC".START_DMC_NUMBER_CHAR_ARRAY[5] <> '$00');
   #_w15 := #_w14 AND ("DB2099_MANUAL_LOAD_DMC".START_DMC_NUMBER_CHAR_ARRAY[5] = ' ') AND "M_DUMMY_ON";
   IF #_w15 THEN "DB2099_MANUAL_LOAD_DMC".DMC_ARRAY_CHAR_UNIT_01[43] := '0'; END_IF;
   IF #_w15 AND "M_DUMMY_OFF" THEN "DB2099_MANUAL_LOAD_DMC".DMC_ARRAY_CHAR_UNIT_01[37] := '0'; END_IF;
   #_w16 := #_w14 AND ("DB2099_MANUAL_LOAD_DMC".START_DMC_NUMBER_CHAR_ARRAY[5] <> ' ') AND "M_DUMMY_ON";
   IF #_w16 THEN
       "DB2099_MANUAL_LOAD_DMC".DMC_ARRAY_CHAR_UNIT_01[43] := "DB2099_MANUAL_LOAD_DMC".START_DMC_NUMBER_CHAR_ARRAY[5];
   END_IF;
   IF #_w16 AND "M_DUMMY_OFF" THEN
       "DB2099_MANUAL_LOAD_DMC".DMC_ARRAY_CHAR_UNIT_01[37] := "DB2099_MANUAL_LOAD_DMC".START_DMC_NUMBER_CHAR_ARRAY[5];
   END_IF;
   #_w17 := #_w1 AND ("DB2099_MANUAL_LOAD_DMC".START_DMC_NUMBER_CHAR_ARRAY[6] <> '$00');
   #_w18 := #_w17 AND ("DB2099_MANUAL_LOAD_DMC".START_DMC_NUMBER_CHAR_ARRAY[6] = ' ') AND "M_DUMMY_ON";
   IF #_w18 THEN "DB2099_MANUAL_LOAD_DMC".DMC_ARRAY_CHAR_UNIT_01[44] := '0'; END_IF;
   IF #_w18 AND "M_DUMMY_OFF" THEN "DB2099_MANUAL_LOAD_DMC".DMC_ARRAY_CHAR_UNIT_01[38] := '0'; END_IF;
   #_w19 := #_w17 AND ("DB2099_MANUAL_LOAD_DMC".START_DMC_NUMBER_CHAR_ARRAY[6] <> ' ') AND "M_DUMMY_ON";
   IF #_w19 THEN
       "DB2099_MANUAL_LOAD_DMC".DMC_ARRAY_CHAR_UNIT_01[44] := "DB2099_MANUAL_LOAD_DMC".START_DMC_NUMBER_CHAR_ARRAY[6];
   END_IF;
   IF #_w19 AND "M_DUMMY_OFF" THEN
       "DB2099_MANUAL_LOAD_DMC".DMC_ARRAY_CHAR_UNIT_01[38] := "DB2099_MANUAL_LOAD_DMC".START_DMC_NUMBER_CHAR_ARRAY[6];
   END_IF;
   #_w20 := #_w1 AND ("DB2099_MANUAL_LOAD_DMC".START_DMC_NUMBER_CHAR_ARRAY[7] <> '$00');
   #_w21 := #_w20 AND ("DB2099_MANUAL_LOAD_DMC".START_DMC_NUMBER_CHAR_ARRAY[7] = ' ') AND "M_DUMMY_ON";
   IF #_w21 THEN "DB2099_MANUAL_LOAD_DMC".DMC_ARRAY_CHAR_UNIT_01[45] := '0'; END_IF;
   IF #_w21 AND "M_DUMMY_OFF" THEN "DB2099_MANUAL_LOAD_DMC".DMC_ARRAY_CHAR_UNIT_01[39] := '0'; END_IF;
   #_w22 := #_w20 AND ("DB2099_MANUAL_LOAD_DMC".START_DMC_NUMBER_CHAR_ARRAY[7] <> ' ') AND "M_DUMMY_ON";
   IF #_w22 THEN
       "DB2099_MANUAL_LOAD_DMC".DMC_ARRAY_CHAR_UNIT_01[45] := "DB2099_MANUAL_LOAD_DMC".START_DMC_NUMBER_CHAR_ARRAY[7];
   END_IF;
   IF #_w22 AND "M_DUMMY_OFF" THEN
       "DB2099_MANUAL_LOAD_DMC".DMC_ARRAY_CHAR_UNIT_01[39] := "DB2099_MANUAL_LOAD_DMC".START_DMC_NUMBER_CHAR_ARRAY[7];
   END_IF;
   #_w23 := #_w1 AND ("DB2099_MANUAL_LOAD_DMC".START_DMC_NUMBER_CHAR_ARRAY[8] <> '$00');
   #_w24 := #_w23 AND ("DB2099_MANUAL_LOAD_DMC".START_DMC_NUMBER_CHAR_ARRAY[8] = ' ') AND "M_DUMMY_ON";
   IF #_w24 THEN "DB2099_MANUAL_LOAD_DMC".DMC_ARRAY_CHAR_UNIT_01[46] := '0'; END_IF;
   IF #_w24 AND "M_DUMMY_OFF" THEN "DB2099_MANUAL_LOAD_DMC".DMC_ARRAY_CHAR_UNIT_01[40] := '0'; END_IF;
   #_w25 := #_w23 AND ("DB2099_MANUAL_LOAD_DMC".START_DMC_NUMBER_CHAR_ARRAY[8] <> ' ') AND "M_DUMMY_ON";
   IF #_w25 THEN
       "DB2099_MANUAL_LOAD_DMC".DMC_ARRAY_CHAR_UNIT_01[46] := "DB2099_MANUAL_LOAD_DMC".START_DMC_NUMBER_CHAR_ARRAY[8];
   END_IF;
   IF #_w25 AND "M_DUMMY_OFF" THEN
       "DB2099_MANUAL_LOAD_DMC".DMC_ARRAY_CHAR_UNIT_01[40] := "DB2099_MANUAL_LOAD_DMC".START_DMC_NUMBER_CHAR_ARRAY[8];
   END_IF;
   #_w26 := #_w1 AND "M_DUMMY_ON";
   IF #_w26 THEN "DB2099_MANUAL_LOAD_DMC".DMC_ARRAY_CHAR_UNIT_01[48] := '$00'; END_IF;
   IF #_w26 AND "M_DUMMY_OFF" THEN "DB2099_MANUAL_LOAD_DMC".DMC_ARRAY_CHAR_UNIT_01[48] := '$00'; END_IF;
END_REGION

REGION Network 19: PART DMC TYPE UNIT 01 & UNIT 02 WRITING FOR MANUAL LOADING
   // M0.2 CUANDO SE DECIDA CON LEON CAMBIAR LA ESTRUCTURA DEL DMC SOLO HARA FALTA BORRAR LO QUE ESTÁ TRAS M0.2 Y BORRAR EL M0.3 PARA QUE SE EJECUTE EL NUEVO CODIGO. DE LO CONTRARIO SUSTITUIR M0.2 POR M0.3 Y VICEVERSA
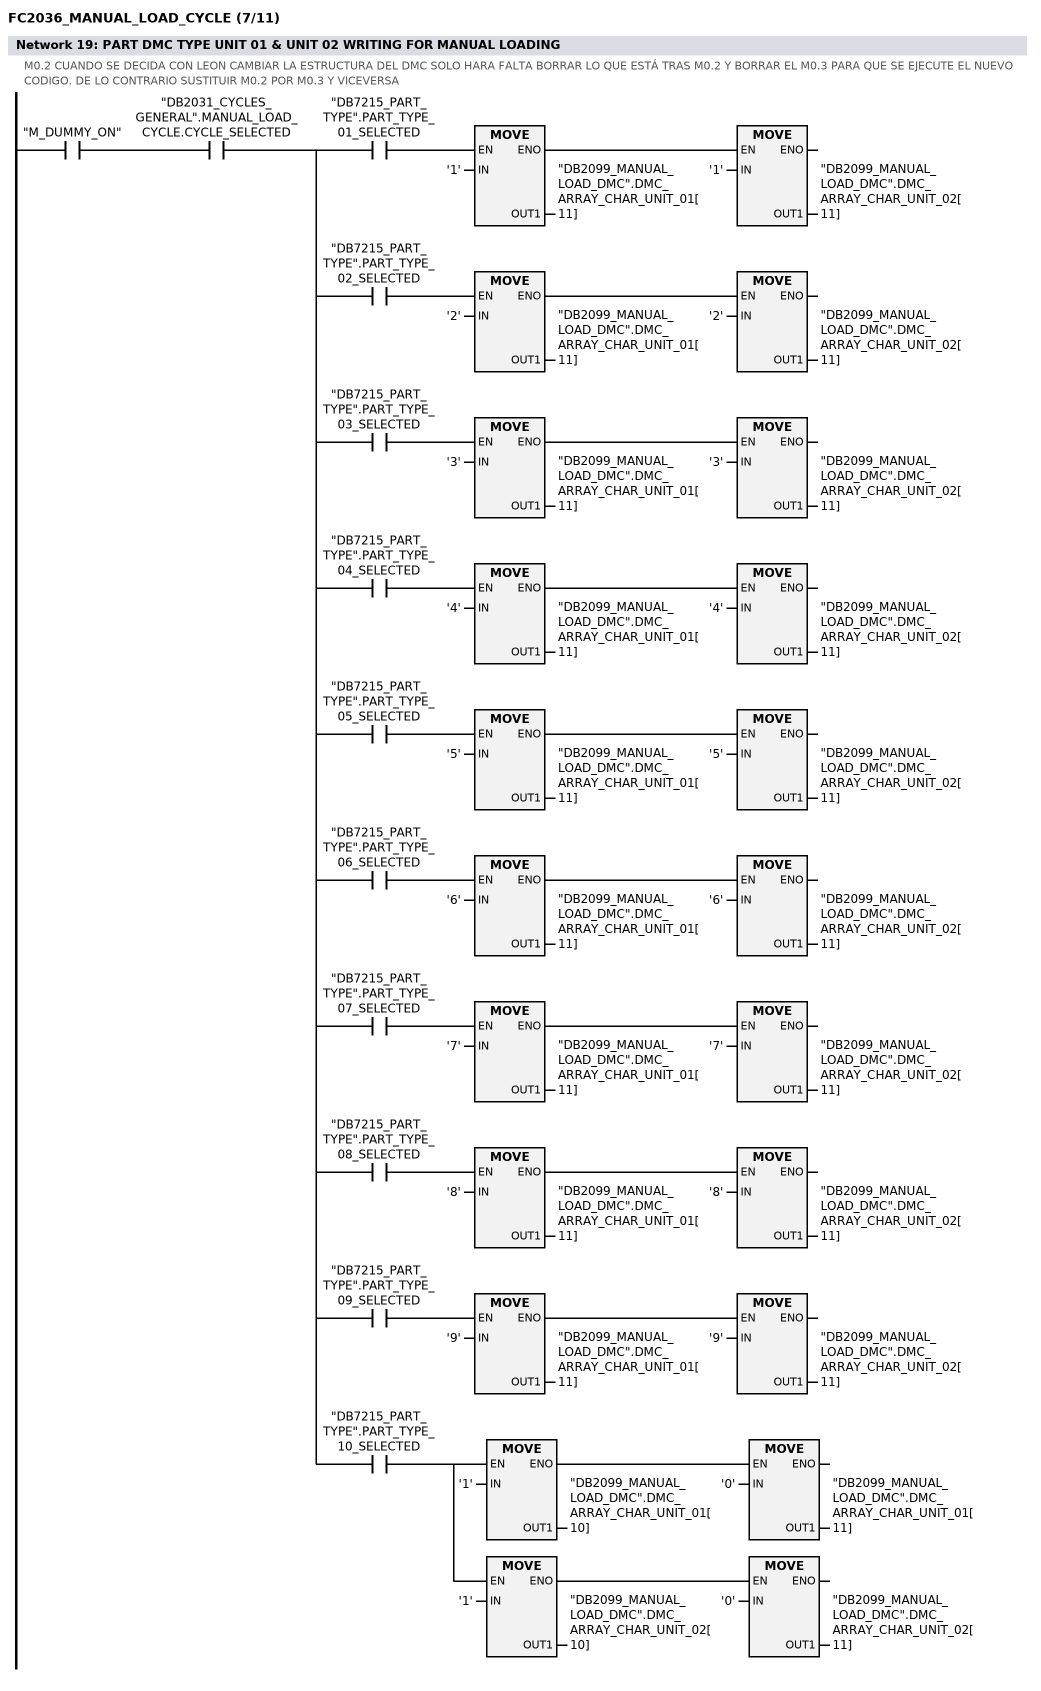
   RUNG wire#powerrail
      Contact( "M_DUMMY_ON" )
      Contact( "DB2031_CYCLES_GENERAL".MANUAL_LOAD_CYCLE.CYCLE_SELECTED )
      wire#w1
      Contact( "DB7215_PART_TYPE".PART_TYPE_01_SELECTED )
      Move(in := '1', out1 => "DB2099_MANUAL_LOAD_DMC".DMC_ARRAY_CHAR_UNIT_01[11])
      Move(in := '1', out1 => "DB2099_MANUAL_LOAD_DMC".DMC_ARRAY_CHAR_UNIT_02[11])
   END_RUNG
   RUNG wire#w1
      Contact( "DB7215_PART_TYPE".PART_TYPE_02_SELECTED )
      Move(in := '2', out1 => "DB2099_MANUAL_LOAD_DMC".DMC_ARRAY_CHAR_UNIT_01[11])
      Move(in := '2', out1 => "DB2099_MANUAL_LOAD_DMC".DMC_ARRAY_CHAR_UNIT_02[11])
   END_RUNG
   RUNG wire#w1
      Contact( "DB7215_PART_TYPE".PART_TYPE_03_SELECTED )
      Move(in := '3', out1 => "DB2099_MANUAL_LOAD_DMC".DMC_ARRAY_CHAR_UNIT_01[11])
      Move(in := '3', out1 => "DB2099_MANUAL_LOAD_DMC".DMC_ARRAY_CHAR_UNIT_02[11])
   END_RUNG
   RUNG wire#w1
      Contact( "DB7215_PART_TYPE".PART_TYPE_04_SELECTED )
      Move(in := '4', out1 => "DB2099_MANUAL_LOAD_DMC".DMC_ARRAY_CHAR_UNIT_01[11])
      Move(in := '4', out1 => "DB2099_MANUAL_LOAD_DMC".DMC_ARRAY_CHAR_UNIT_02[11])
   END_RUNG
   RUNG wire#w1
      Contact( "DB7215_PART_TYPE".PART_TYPE_05_SELECTED )
      Move(in := '5', out1 => "DB2099_MANUAL_LOAD_DMC".DMC_ARRAY_CHAR_UNIT_01[11])
      Move(in := '5', out1 => "DB2099_MANUAL_LOAD_DMC".DMC_ARRAY_CHAR_UNIT_02[11])
   END_RUNG
   RUNG wire#w1
      Contact( "DB7215_PART_TYPE".PART_TYPE_06_SELECTED )
      Move(in := '6', out1 => "DB2099_MANUAL_LOAD_DMC".DMC_ARRAY_CHAR_UNIT_01[11])
      Move(in := '6', out1 => "DB2099_MANUAL_LOAD_DMC".DMC_ARRAY_CHAR_UNIT_02[11])
   END_RUNG
   RUNG wire#w1
      Contact( "DB7215_PART_TYPE".PART_TYPE_07_SELECTED )
      Move(in := '7', out1 => "DB2099_MANUAL_LOAD_DMC".DMC_ARRAY_CHAR_UNIT_01[11])
      Move(in := '7', out1 => "DB2099_MANUAL_LOAD_DMC".DMC_ARRAY_CHAR_UNIT_02[11])
   END_RUNG
   RUNG wire#w1
      Contact( "DB7215_PART_TYPE".PART_TYPE_08_SELECTED )
      Move(in := '8', out1 => "DB2099_MANUAL_LOAD_DMC".DMC_ARRAY_CHAR_UNIT_01[11])
      Move(in := '8', out1 => "DB2099_MANUAL_LOAD_DMC".DMC_ARRAY_CHAR_UNIT_02[11])
   END_RUNG
   RUNG wire#w1
      Contact( "DB7215_PART_TYPE".PART_TYPE_09_SELECTED )
      Move(in := '9', out1 => "DB2099_MANUAL_LOAD_DMC".DMC_ARRAY_CHAR_UNIT_01[11])
      Move(in := '9', out1 => "DB2099_MANUAL_LOAD_DMC".DMC_ARRAY_CHAR_UNIT_02[11])
   END_RUNG
   RUNG wire#w1
      Contact( "DB7215_PART_TYPE".PART_TYPE_10_SELECTED )
      wire#w2
      Move(in := '1', out1 => "DB2099_MANUAL_LOAD_DMC".DMC_ARRAY_CHAR_UNIT_01[10])
      Move(in := '0', out1 => "DB2099_MANUAL_LOAD_DMC".DMC_ARRAY_CHAR_UNIT_01[11])
   END_RUNG
   RUNG wire#w2
      Move(in := '1', out1 => "DB2099_MANUAL_LOAD_DMC".DMC_ARRAY_CHAR_UNIT_02[10])
      Move(in := '0', out1 => "DB2099_MANUAL_LOAD_DMC".DMC_ARRAY_CHAR_UNIT_02[11])
   END_RUNG
   // the same network as SCL:
   #_w1 := "M_DUMMY_ON" AND "DB2031_CYCLES_GENERAL".MANUAL_LOAD_CYCLE.CYCLE_SELECTED;
   IF #_w1 AND "DB7215_PART_TYPE".PART_TYPE_01_SELECTED THEN
       "DB2099_MANUAL_LOAD_DMC".DMC_ARRAY_CHAR_UNIT_01[11] := '1';
       "DB2099_MANUAL_LOAD_DMC".DMC_ARRAY_CHAR_UNIT_02[11] := '1';
   END_IF;
   IF #_w1 AND "DB7215_PART_TYPE".PART_TYPE_02_SELECTED THEN
       "DB2099_MANUAL_LOAD_DMC".DMC_ARRAY_CHAR_UNIT_01[11] := '2';
       "DB2099_MANUAL_LOAD_DMC".DMC_ARRAY_CHAR_UNIT_02[11] := '2';
   END_IF;
   IF #_w1 AND "DB7215_PART_TYPE".PART_TYPE_03_SELECTED THEN
       "DB2099_MANUAL_LOAD_DMC".DMC_ARRAY_CHAR_UNIT_01[11] := '3';
       "DB2099_MANUAL_LOAD_DMC".DMC_ARRAY_CHAR_UNIT_02[11] := '3';
   END_IF;
   IF #_w1 AND "DB7215_PART_TYPE".PART_TYPE_04_SELECTED THEN
       "DB2099_MANUAL_LOAD_DMC".DMC_ARRAY_CHAR_UNIT_01[11] := '4';
       "DB2099_MANUAL_LOAD_DMC".DMC_ARRAY_CHAR_UNIT_02[11] := '4';
   END_IF;
   IF #_w1 AND "DB7215_PART_TYPE".PART_TYPE_05_SELECTED THEN
       "DB2099_MANUAL_LOAD_DMC".DMC_ARRAY_CHAR_UNIT_01[11] := '5';
       "DB2099_MANUAL_LOAD_DMC".DMC_ARRAY_CHAR_UNIT_02[11] := '5';
   END_IF;
   IF #_w1 AND "DB7215_PART_TYPE".PART_TYPE_06_SELECTED THEN
       "DB2099_MANUAL_LOAD_DMC".DMC_ARRAY_CHAR_UNIT_01[11] := '6';
       "DB2099_MANUAL_LOAD_DMC".DMC_ARRAY_CHAR_UNIT_02[11] := '6';
   END_IF;
   IF #_w1 AND "DB7215_PART_TYPE".PART_TYPE_07_SELECTED THEN
       "DB2099_MANUAL_LOAD_DMC".DMC_ARRAY_CHAR_UNIT_01[11] := '7';
       "DB2099_MANUAL_LOAD_DMC".DMC_ARRAY_CHAR_UNIT_02[11] := '7';
   END_IF;
   IF #_w1 AND "DB7215_PART_TYPE".PART_TYPE_08_SELECTED THEN
       "DB2099_MANUAL_LOAD_DMC".DMC_ARRAY_CHAR_UNIT_01[11] := '8';
       "DB2099_MANUAL_LOAD_DMC".DMC_ARRAY_CHAR_UNIT_02[11] := '8';
   END_IF;
   IF #_w1 AND "DB7215_PART_TYPE".PART_TYPE_09_SELECTED THEN
       "DB2099_MANUAL_LOAD_DMC".DMC_ARRAY_CHAR_UNIT_01[11] := '9';
       "DB2099_MANUAL_LOAD_DMC".DMC_ARRAY_CHAR_UNIT_02[11] := '9';
   END_IF;
   IF #_w1 AND "DB7215_PART_TYPE".PART_TYPE_10_SELECTED THEN
       "DB2099_MANUAL_LOAD_DMC".DMC_ARRAY_CHAR_UNIT_01[10] := '1';
       "DB2099_MANUAL_LOAD_DMC".DMC_ARRAY_CHAR_UNIT_01[11] := '0';
       "DB2099_MANUAL_LOAD_DMC".DMC_ARRAY_CHAR_UNIT_02[10] := '1';
       "DB2099_MANUAL_LOAD_DMC".DMC_ARRAY_CHAR_UNIT_02[11] := '0';
   END_IF;
END_REGION

REGION Network 20: PART LOADED UNIT 01 MANUAL LOADING
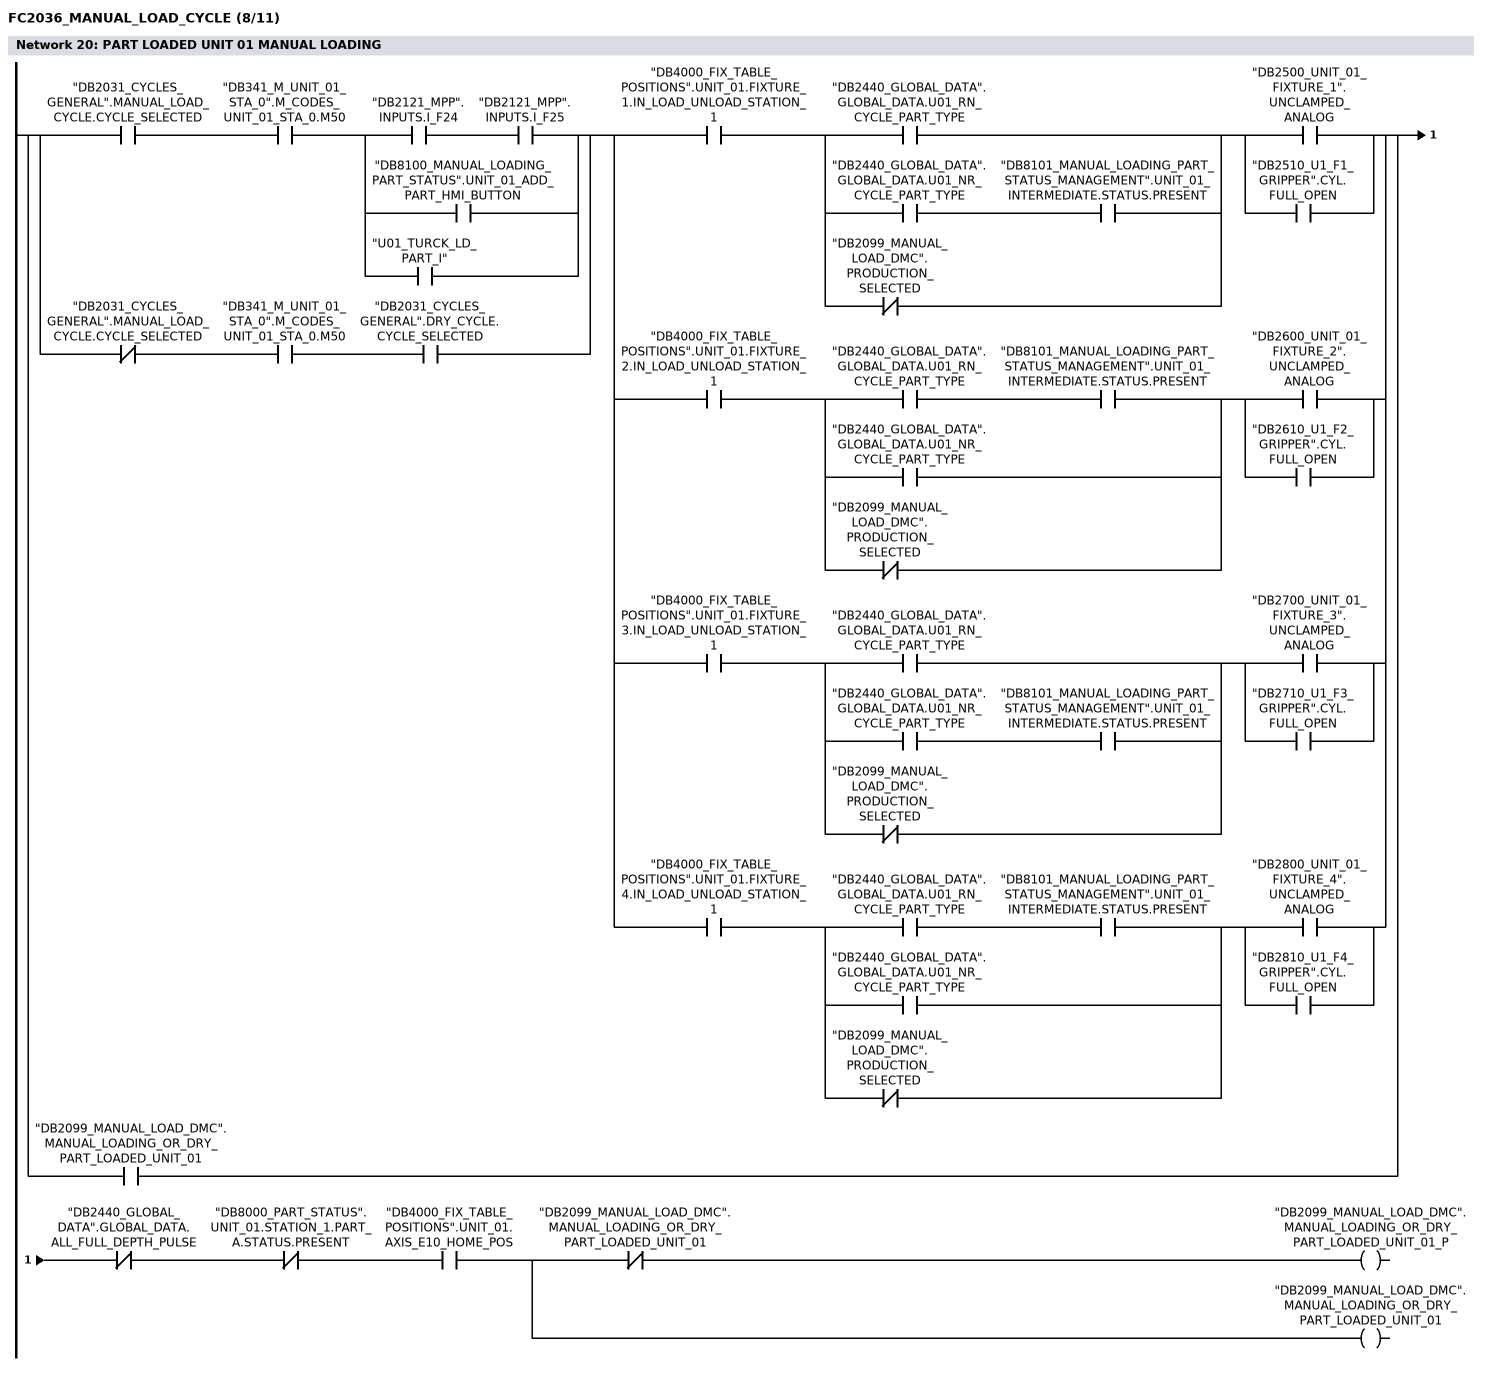
   RUNG wire#powerrail
      Contact( "DB2031_CYCLES_GENERAL".MANUAL_LOAD_CYCLE.CYCLE_SELECTED )
      Contact( "DB341_M_UNIT_01_STA_0".M_CODES_UNIT_01_STA_0.M50 )
      wire#w1
      Contact( "DB2121_MPP".INPUTS.I_F24 )
      Contact( "DB2121_MPP".INPUTS.I_F25 )
      wire#w2
      Contact( "DB4000_FIX_TABLE_POSITIONS".UNIT_01.FIXTURE_1.IN_LOAD_UNLOAD_STATION_1 )
      wire#w3
      Contact( "DB2440_GLOBAL_DATA".GLOBAL_DATA.U01_RN_CYCLE_PART_TYPE )
      wire#w4
      Contact( "DB2500_UNIT_01_FIXTURE_1".UNCLAMPED_ANALOG )
      wire#w5
      I_Contact( "DB2440_GLOBAL_DATA".GLOBAL_DATA.ALL_FULL_DEPTH_PULSE )
      I_Contact( "DB8000_PART_STATUS".UNIT_01.STATION_1.PART_A.STATUS.PRESENT )
      Contact( "DB4000_FIX_TABLE_POSITIONS".UNIT_01.AXIS_E10_HOME_POS )
      wire#w12
      I_Contact( "DB2099_MANUAL_LOAD_DMC".MANUAL_LOADING_OR_DRY_PART_LOADED_UNIT_01 )
      Coil( "DB2099_MANUAL_LOAD_DMC".MANUAL_LOADING_OR_DRY_PART_LOADED_UNIT_01_P )
   END_RUNG
   RUNG wire#w1
      Contact( "DB8100_MANUAL_LOADING_PART_STATUS".UNIT_01_ADD_PART_HMI_BUTTON )
   END_RUNG wire#w2
   RUNG wire#w1
      Contact( "U01_TURCK_LD_PART_I" )
   END_RUNG wire#w2
   RUNG wire#powerrail
      I_Contact( "DB2031_CYCLES_GENERAL".MANUAL_LOAD_CYCLE.CYCLE_SELECTED )
      Contact( "DB341_M_UNIT_01_STA_0".M_CODES_UNIT_01_STA_0.M50 )
      Contact( "DB2031_CYCLES_GENERAL".DRY_CYCLE.CYCLE_SELECTED )
   END_RUNG wire#w2
   RUNG wire#w3
      Contact( "DB2440_GLOBAL_DATA".GLOBAL_DATA.U01_NR_CYCLE_PART_TYPE )
      Contact( "DB8101_MANUAL_LOADING_PART_STATUS_MANAGEMENT".UNIT_01_INTERMEDIATE.STATUS.PRESENT )
   END_RUNG wire#w4
   RUNG wire#w3
      I_Contact( "DB2099_MANUAL_LOAD_DMC".PRODUCTION_SELECTED )
   END_RUNG wire#w4
   RUNG wire#w4
      Contact( "DB2510_U1_F1_GRIPPER".CYL.FULL_OPEN )
   END_RUNG wire#w5
   RUNG wire#w2
      Contact( "DB4000_FIX_TABLE_POSITIONS".UNIT_01.FIXTURE_2.IN_LOAD_UNLOAD_STATION_1 )
      wire#w6
      Contact( "DB2440_GLOBAL_DATA".GLOBAL_DATA.U01_RN_CYCLE_PART_TYPE )
      Contact( "DB8101_MANUAL_LOADING_PART_STATUS_MANAGEMENT".UNIT_01_INTERMEDIATE.STATUS.PRESENT )
      wire#w7
      Contact( "DB2600_UNIT_01_FIXTURE_2".UNCLAMPED_ANALOG )
   END_RUNG wire#w5
   RUNG wire#w6
      Contact( "DB2440_GLOBAL_DATA".GLOBAL_DATA.U01_NR_CYCLE_PART_TYPE )
   END_RUNG wire#w7
   RUNG wire#w6
      I_Contact( "DB2099_MANUAL_LOAD_DMC".PRODUCTION_SELECTED )
   END_RUNG wire#w7
   RUNG wire#w7
      Contact( "DB2610_U1_F2_GRIPPER".CYL.FULL_OPEN )
   END_RUNG wire#w5
   RUNG wire#w2
      Contact( "DB4000_FIX_TABLE_POSITIONS".UNIT_01.FIXTURE_3.IN_LOAD_UNLOAD_STATION_1 )
      wire#w8
      Contact( "DB2440_GLOBAL_DATA".GLOBAL_DATA.U01_RN_CYCLE_PART_TYPE )
      wire#w9
      Contact( "DB2700_UNIT_01_FIXTURE_3".UNCLAMPED_ANALOG )
   END_RUNG wire#w5
   RUNG wire#w8
      Contact( "DB2440_GLOBAL_DATA".GLOBAL_DATA.U01_NR_CYCLE_PART_TYPE )
      Contact( "DB8101_MANUAL_LOADING_PART_STATUS_MANAGEMENT".UNIT_01_INTERMEDIATE.STATUS.PRESENT )
   END_RUNG wire#w9
   RUNG wire#w8
      I_Contact( "DB2099_MANUAL_LOAD_DMC".PRODUCTION_SELECTED )
   END_RUNG wire#w9
   RUNG wire#w9
      Contact( "DB2710_U1_F3_GRIPPER".CYL.FULL_OPEN )
   END_RUNG wire#w5
   RUNG wire#w2
      Contact( "DB4000_FIX_TABLE_POSITIONS".UNIT_01.FIXTURE_4.IN_LOAD_UNLOAD_STATION_1 )
      wire#w10
      Contact( "DB2440_GLOBAL_DATA".GLOBAL_DATA.U01_RN_CYCLE_PART_TYPE )
      Contact( "DB8101_MANUAL_LOADING_PART_STATUS_MANAGEMENT".UNIT_01_INTERMEDIATE.STATUS.PRESENT )
      wire#w11
      Contact( "DB2800_UNIT_01_FIXTURE_4".UNCLAMPED_ANALOG )
   END_RUNG wire#w5
   RUNG wire#w10
      Contact( "DB2440_GLOBAL_DATA".GLOBAL_DATA.U01_NR_CYCLE_PART_TYPE )
   END_RUNG wire#w11
   RUNG wire#w10
      I_Contact( "DB2099_MANUAL_LOAD_DMC".PRODUCTION_SELECTED )
   END_RUNG wire#w11
   RUNG wire#w11
      Contact( "DB2810_U1_F4_GRIPPER".CYL.FULL_OPEN )
   END_RUNG wire#w5
   RUNG wire#powerrail
      Contact( "DB2099_MANUAL_LOAD_DMC".MANUAL_LOADING_OR_DRY_PART_LOADED_UNIT_01 )
   END_RUNG wire#w5
   RUNG wire#w12
      Coil( "DB2099_MANUAL_LOAD_DMC".MANUAL_LOADING_OR_DRY_PART_LOADED_UNIT_01 )
   END_RUNG
   // the same network as SCL:
   #_w1 := (((("DB2031_CYCLES_GENERAL".MANUAL_LOAD_CYCLE.CYCLE_SELECTED AND "DB341_M_UNIT_01_STA_0".M_CODES_UNIT_01_STA_0.M50 AND (("DB2121_MPP".INPUTS.I_F24 AND "DB2121_MPP".INPUTS.I_F25) OR "DB8100_MANUAL_LOADING_PART_STATUS".UNIT_01_ADD_PART_HMI_BUTTON OR "U01_TURCK_LD_PART_I")) OR (NOT "DB2031_CYCLES_GENERAL".MANUAL_LOAD_CYCLE.CYCLE_SELECTED AND "DB341_M_UNIT_01_STA_0".M_CODES_UNIT_01_STA_0.M50 AND "DB2031_CYCLES_GENERAL".DRY_CYCLE.CYCLE_SELECTED)) AND (("DB4000_FIX_TABLE_POSITIONS".UNIT_01.FIXTURE_1.IN_LOAD_UNLOAD_STATION_1 AND ("DB2440_GLOBAL_DATA".GLOBAL_DATA.U01_RN_CYCLE_PART_TYPE OR ("DB2440_GLOBAL_DATA".GLOBAL_DATA.U01_NR_CYCLE_PART_TYPE AND "DB8101_MANUAL_LOADING_PART_STATUS_MANAGEMENT".UNIT_01_INTERMEDIATE.STATUS.PRESENT) OR NOT "DB2099_MANUAL_LOAD_DMC".PRODUCTION_SELECTED) AND ("DB2500_UNIT_01_FIXTURE_1".UNCLAMPED_ANALOG OR "DB2510_U1_F1_GRIPPER".CYL.FULL_OPEN)) OR ("DB4000_FIX_TABLE_POSITIONS".UNIT_01.FIXTURE_2.IN_LOAD_UNLOAD_STATION_1 AND (("DB2440_GLOBAL_DATA".GLOBAL_DATA.U01_RN_CYCLE_PART_TYPE AND "DB8101_MANUAL_LOADING_PART_STATUS_MANAGEMENT".UNIT_01_INTERMEDIATE.STATUS.PRESENT) OR "DB2440_GLOBAL_DATA".GLOBAL_DATA.U01_NR_CYCLE_PART_TYPE OR NOT "DB2099_MANUAL_LOAD_DMC".PRODUCTION_SELECTED) AND ("DB2600_UNIT_01_FIXTURE_2".UNCLAMPED_ANALOG OR "DB2610_U1_F2_GRIPPER".CYL.FULL_OPEN)) OR ("DB4000_FIX_TABLE_POSITIONS".UNIT_01.FIXTURE_3.IN_LOAD_UNLOAD_STATION_1 AND ("DB2440_GLOBAL_DATA".GLOBAL_DATA.U01_RN_CYCLE_PART_TYPE OR ("DB2440_GLOBAL_DATA".GLOBAL_DATA.U01_NR_CYCLE_PART_TYPE AND "DB8101_MANUAL_LOADING_PART_STATUS_MANAGEMENT".UNIT_01_INTERMEDIATE.STATUS.PRESENT) OR NOT "DB2099_MANUAL_LOAD_DMC".PRODUCTION_SELECTED) AND ("DB2700_UNIT_01_FIXTURE_3".UNCLAMPED_ANALOG OR "DB2710_U1_F3_GRIPPER".CYL.FULL_OPEN)) OR ("DB4000_FIX_TABLE_POSITIONS".UNIT_01.FIXTURE_4.IN_LOAD_UNLOAD_STATION_1 AND (("DB2440_GLOBAL_DATA".GLOBAL_DATA.U01_RN_CYCLE_PART_TYPE AND "DB8101_MANUAL_LOADING_PART_STATUS_MANAGEMENT".UNIT_01_INTERMEDIATE.STATUS.PRESENT) OR "DB2440_GLOBAL_DATA".GLOBAL_DATA.U01_NR_CYCLE_PART_TYPE OR NOT "DB2099_MANUAL_LOAD_DMC".PRODUCTION_SELECTED) AND ("DB2800_UNIT_01_FIXTURE_4".UNCLAMPED_ANALOG OR "DB2810_U1_F4_GRIPPER".CYL.FULL_OPEN)))) OR "DB2099_MANUAL_LOAD_DMC".MANUAL_LOADING_OR_DRY_PART_LOADED_UNIT_01) AND NOT "DB2440_GLOBAL_DATA".GLOBAL_DATA.ALL_FULL_DEPTH_PULSE AND NOT "DB8000_PART_STATUS".UNIT_01.STATION_1.PART_A.STATUS.PRESENT AND "DB4000_FIX_TABLE_POSITIONS".UNIT_01.AXIS_E10_HOME_POS;
   "DB2099_MANUAL_LOAD_DMC".MANUAL_LOADING_OR_DRY_PART_LOADED_UNIT_01_P := #_w1 AND NOT "DB2099_MANUAL_LOAD_DMC".MANUAL_LOADING_OR_DRY_PART_LOADED_UNIT_01;
   "DB2099_MANUAL_LOAD_DMC".MANUAL_LOADING_OR_DRY_PART_LOADED_UNIT_01 := #_w1;
END_REGION

REGION Network 21: PART LOADED UNIT 02 MANUAL LOADING
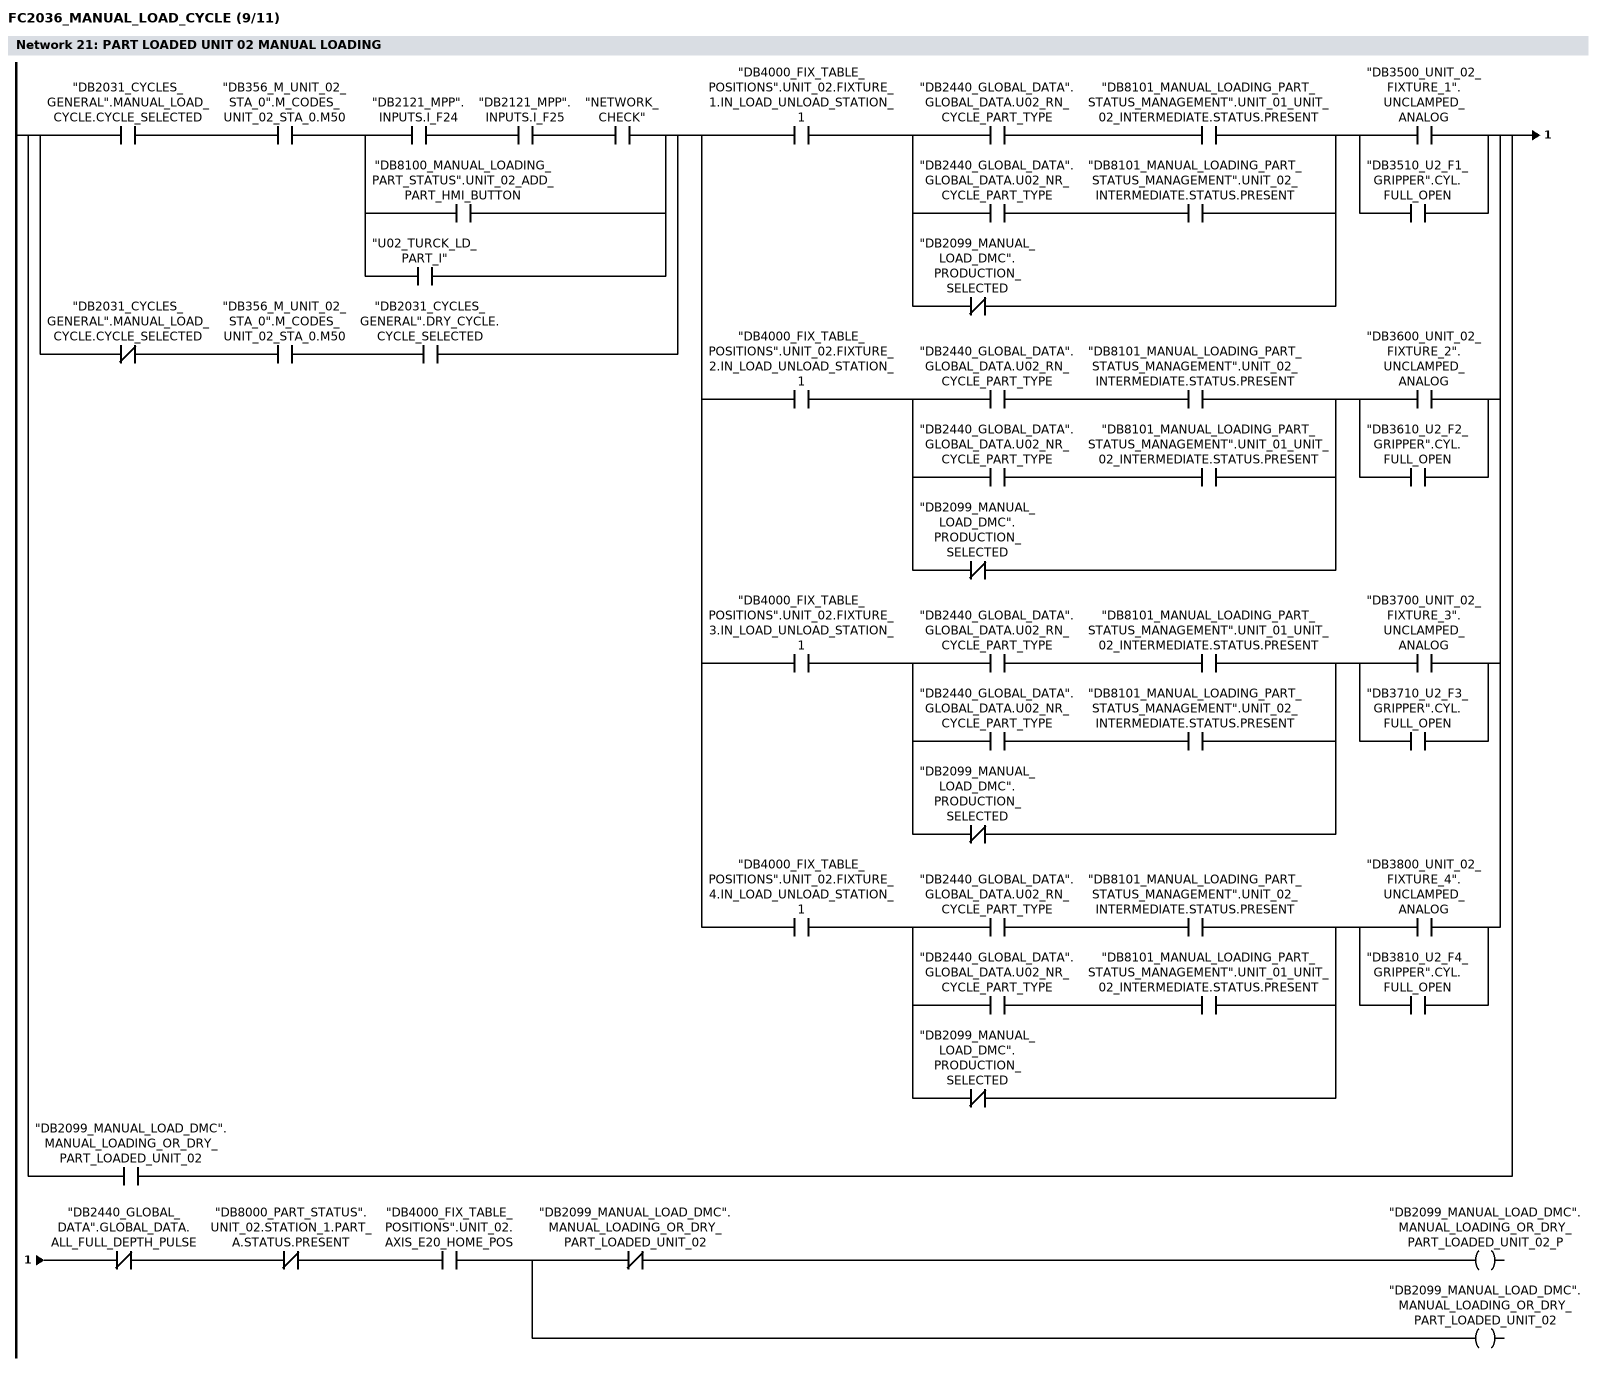
   RUNG wire#powerrail
      Contact( "DB2031_CYCLES_GENERAL".MANUAL_LOAD_CYCLE.CYCLE_SELECTED )
      Contact( "DB356_M_UNIT_02_STA_0".M_CODES_UNIT_02_STA_0.M50 )
      wire#w1
      Contact( "DB2121_MPP".INPUTS.I_F24 )
      Contact( "DB2121_MPP".INPUTS.I_F25 )
      Contact( "NETWORK_CHECK" )
      wire#w2
      Contact( "DB4000_FIX_TABLE_POSITIONS".UNIT_02.FIXTURE_1.IN_LOAD_UNLOAD_STATION_1 )
      wire#w3
      Contact( "DB2440_GLOBAL_DATA".GLOBAL_DATA.U02_RN_CYCLE_PART_TYPE )
      Contact( "DB8101_MANUAL_LOADING_PART_STATUS_MANAGEMENT".UNIT_01_UNIT_02_INTERMEDIATE.STATUS.PRESENT )
      wire#w4
      Contact( "DB3500_UNIT_02_FIXTURE_1".UNCLAMPED_ANALOG )
      wire#w5
      I_Contact( "DB2440_GLOBAL_DATA".GLOBAL_DATA.ALL_FULL_DEPTH_PULSE )
      I_Contact( "DB8000_PART_STATUS".UNIT_02.STATION_1.PART_A.STATUS.PRESENT )
      Contact( "DB4000_FIX_TABLE_POSITIONS".UNIT_02.AXIS_E20_HOME_POS )
      wire#w12
      I_Contact( "DB2099_MANUAL_LOAD_DMC".MANUAL_LOADING_OR_DRY_PART_LOADED_UNIT_02 )
      Coil( "DB2099_MANUAL_LOAD_DMC".MANUAL_LOADING_OR_DRY_PART_LOADED_UNIT_02_P )
   END_RUNG
   RUNG wire#w1
      Contact( "DB8100_MANUAL_LOADING_PART_STATUS".UNIT_02_ADD_PART_HMI_BUTTON )
   END_RUNG wire#w2
   RUNG wire#w1
      Contact( "U02_TURCK_LD_PART_I" )
   END_RUNG wire#w2
   RUNG wire#powerrail
      I_Contact( "DB2031_CYCLES_GENERAL".MANUAL_LOAD_CYCLE.CYCLE_SELECTED )
      Contact( "DB356_M_UNIT_02_STA_0".M_CODES_UNIT_02_STA_0.M50 )
      Contact( "DB2031_CYCLES_GENERAL".DRY_CYCLE.CYCLE_SELECTED )
   END_RUNG wire#w2
   RUNG wire#w3
      Contact( "DB2440_GLOBAL_DATA".GLOBAL_DATA.U02_NR_CYCLE_PART_TYPE )
      Contact( "DB8101_MANUAL_LOADING_PART_STATUS_MANAGEMENT".UNIT_02_INTERMEDIATE.STATUS.PRESENT )
   END_RUNG wire#w4
   RUNG wire#w3
      I_Contact( "DB2099_MANUAL_LOAD_DMC".PRODUCTION_SELECTED )
   END_RUNG wire#w4
   RUNG wire#w4
      Contact( "DB3510_U2_F1_GRIPPER".CYL.FULL_OPEN )
   END_RUNG wire#w5
   RUNG wire#w2
      Contact( "DB4000_FIX_TABLE_POSITIONS".UNIT_02.FIXTURE_2.IN_LOAD_UNLOAD_STATION_1 )
      wire#w6
      Contact( "DB2440_GLOBAL_DATA".GLOBAL_DATA.U02_RN_CYCLE_PART_TYPE )
      Contact( "DB8101_MANUAL_LOADING_PART_STATUS_MANAGEMENT".UNIT_02_INTERMEDIATE.STATUS.PRESENT )
      wire#w7
      Contact( "DB3600_UNIT_02_FIXTURE_2".UNCLAMPED_ANALOG )
   END_RUNG wire#w5
   RUNG wire#w6
      Contact( "DB2440_GLOBAL_DATA".GLOBAL_DATA.U02_NR_CYCLE_PART_TYPE )
      Contact( "DB8101_MANUAL_LOADING_PART_STATUS_MANAGEMENT".UNIT_01_UNIT_02_INTERMEDIATE.STATUS.PRESENT )
   END_RUNG wire#w7
   RUNG wire#w6
      I_Contact( "DB2099_MANUAL_LOAD_DMC".PRODUCTION_SELECTED )
   END_RUNG wire#w7
   RUNG wire#w7
      Contact( "DB3610_U2_F2_GRIPPER".CYL.FULL_OPEN )
   END_RUNG wire#w5
   RUNG wire#w2
      Contact( "DB4000_FIX_TABLE_POSITIONS".UNIT_02.FIXTURE_3.IN_LOAD_UNLOAD_STATION_1 )
      wire#w8
      Contact( "DB2440_GLOBAL_DATA".GLOBAL_DATA.U02_RN_CYCLE_PART_TYPE )
      Contact( "DB8101_MANUAL_LOADING_PART_STATUS_MANAGEMENT".UNIT_01_UNIT_02_INTERMEDIATE.STATUS.PRESENT )
      wire#w9
      Contact( "DB3700_UNIT_02_FIXTURE_3".UNCLAMPED_ANALOG )
   END_RUNG wire#w5
   RUNG wire#w8
      Contact( "DB2440_GLOBAL_DATA".GLOBAL_DATA.U02_NR_CYCLE_PART_TYPE )
      Contact( "DB8101_MANUAL_LOADING_PART_STATUS_MANAGEMENT".UNIT_02_INTERMEDIATE.STATUS.PRESENT )
   END_RUNG wire#w9
   RUNG wire#w8
      I_Contact( "DB2099_MANUAL_LOAD_DMC".PRODUCTION_SELECTED )
   END_RUNG wire#w9
   RUNG wire#w9
      Contact( "DB3710_U2_F3_GRIPPER".CYL.FULL_OPEN )
   END_RUNG wire#w5
   RUNG wire#w2
      Contact( "DB4000_FIX_TABLE_POSITIONS".UNIT_02.FIXTURE_4.IN_LOAD_UNLOAD_STATION_1 )
      wire#w10
      Contact( "DB2440_GLOBAL_DATA".GLOBAL_DATA.U02_RN_CYCLE_PART_TYPE )
      Contact( "DB8101_MANUAL_LOADING_PART_STATUS_MANAGEMENT".UNIT_02_INTERMEDIATE.STATUS.PRESENT )
      wire#w11
      Contact( "DB3800_UNIT_02_FIXTURE_4".UNCLAMPED_ANALOG )
   END_RUNG wire#w5
   RUNG wire#w10
      Contact( "DB2440_GLOBAL_DATA".GLOBAL_DATA.U02_NR_CYCLE_PART_TYPE )
      Contact( "DB8101_MANUAL_LOADING_PART_STATUS_MANAGEMENT".UNIT_01_UNIT_02_INTERMEDIATE.STATUS.PRESENT )
   END_RUNG wire#w11
   RUNG wire#w10
      I_Contact( "DB2099_MANUAL_LOAD_DMC".PRODUCTION_SELECTED )
   END_RUNG wire#w11
   RUNG wire#w11
      Contact( "DB3810_U2_F4_GRIPPER".CYL.FULL_OPEN )
   END_RUNG wire#w5
   RUNG wire#powerrail
      Contact( "DB2099_MANUAL_LOAD_DMC".MANUAL_LOADING_OR_DRY_PART_LOADED_UNIT_02 )
   END_RUNG wire#w5
   RUNG wire#w12
      Coil( "DB2099_MANUAL_LOAD_DMC".MANUAL_LOADING_OR_DRY_PART_LOADED_UNIT_02 )
   END_RUNG
   // the same network as SCL:
   #_w1 := (((("DB2031_CYCLES_GENERAL".MANUAL_LOAD_CYCLE.CYCLE_SELECTED AND "DB356_M_UNIT_02_STA_0".M_CODES_UNIT_02_STA_0.M50 AND (("DB2121_MPP".INPUTS.I_F24 AND "DB2121_MPP".INPUTS.I_F25 AND "NETWORK_CHECK") OR "DB8100_MANUAL_LOADING_PART_STATUS".UNIT_02_ADD_PART_HMI_BUTTON OR "U02_TURCK_LD_PART_I")) OR (NOT "DB2031_CYCLES_GENERAL".MANUAL_LOAD_CYCLE.CYCLE_SELECTED AND "DB356_M_UNIT_02_STA_0".M_CODES_UNIT_02_STA_0.M50 AND "DB2031_CYCLES_GENERAL".DRY_CYCLE.CYCLE_SELECTED)) AND (("DB4000_FIX_TABLE_POSITIONS".UNIT_02.FIXTURE_1.IN_LOAD_UNLOAD_STATION_1 AND (("DB2440_GLOBAL_DATA".GLOBAL_DATA.U02_RN_CYCLE_PART_TYPE AND "DB8101_MANUAL_LOADING_PART_STATUS_MANAGEMENT".UNIT_01_UNIT_02_INTERMEDIATE.STATUS.PRESENT) OR ("DB2440_GLOBAL_DATA".GLOBAL_DATA.U02_NR_CYCLE_PART_TYPE AND "DB8101_MANUAL_LOADING_PART_STATUS_MANAGEMENT".UNIT_02_INTERMEDIATE.STATUS.PRESENT) OR NOT "DB2099_MANUAL_LOAD_DMC".PRODUCTION_SELECTED) AND ("DB3500_UNIT_02_FIXTURE_1".UNCLAMPED_ANALOG OR "DB3510_U2_F1_GRIPPER".CYL.FULL_OPEN)) OR ("DB4000_FIX_TABLE_POSITIONS".UNIT_02.FIXTURE_2.IN_LOAD_UNLOAD_STATION_1 AND (("DB2440_GLOBAL_DATA".GLOBAL_DATA.U02_RN_CYCLE_PART_TYPE AND "DB8101_MANUAL_LOADING_PART_STATUS_MANAGEMENT".UNIT_02_INTERMEDIATE.STATUS.PRESENT) OR ("DB2440_GLOBAL_DATA".GLOBAL_DATA.U02_NR_CYCLE_PART_TYPE AND "DB8101_MANUAL_LOADING_PART_STATUS_MANAGEMENT".UNIT_01_UNIT_02_INTERMEDIATE.STATUS.PRESENT) OR NOT "DB2099_MANUAL_LOAD_DMC".PRODUCTION_SELECTED) AND ("DB3600_UNIT_02_FIXTURE_2".UNCLAMPED_ANALOG OR "DB3610_U2_F2_GRIPPER".CYL.FULL_OPEN)) OR ("DB4000_FIX_TABLE_POSITIONS".UNIT_02.FIXTURE_3.IN_LOAD_UNLOAD_STATION_1 AND (("DB2440_GLOBAL_DATA".GLOBAL_DATA.U02_RN_CYCLE_PART_TYPE AND "DB8101_MANUAL_LOADING_PART_STATUS_MANAGEMENT".UNIT_01_UNIT_02_INTERMEDIATE.STATUS.PRESENT) OR ("DB2440_GLOBAL_DATA".GLOBAL_DATA.U02_NR_CYCLE_PART_TYPE AND "DB8101_MANUAL_LOADING_PART_STATUS_MANAGEMENT".UNIT_02_INTERMEDIATE.STATUS.PRESENT) OR NOT "DB2099_MANUAL_LOAD_DMC".PRODUCTION_SELECTED) AND ("DB3700_UNIT_02_FIXTURE_3".UNCLAMPED_ANALOG OR "DB3710_U2_F3_GRIPPER".CYL.FULL_OPEN)) OR ("DB4000_FIX_TABLE_POSITIONS".UNIT_02.FIXTURE_4.IN_LOAD_UNLOAD_STATION_1 AND (("DB2440_GLOBAL_DATA".GLOBAL_DATA.U02_RN_CYCLE_PART_TYPE AND "DB8101_MANUAL_LOADING_PART_STATUS_MANAGEMENT".UNIT_02_INTERMEDIATE.STATUS.PRESENT) OR ("DB2440_GLOBAL_DATA".GLOBAL_DATA.U02_NR_CYCLE_PART_TYPE AND "DB8101_MANUAL_LOADING_PART_STATUS_MANAGEMENT".UNIT_01_UNIT_02_INTERMEDIATE.STATUS.PRESENT) OR NOT "DB2099_MANUAL_LOAD_DMC".PRODUCTION_SELECTED) AND ("DB3800_UNIT_02_FIXTURE_4".UNCLAMPED_ANALOG OR "DB3810_U2_F4_GRIPPER".CYL.FULL_OPEN)))) OR "DB2099_MANUAL_LOAD_DMC".MANUAL_LOADING_OR_DRY_PART_LOADED_UNIT_02) AND NOT "DB2440_GLOBAL_DATA".GLOBAL_DATA.ALL_FULL_DEPTH_PULSE AND NOT "DB8000_PART_STATUS".UNIT_02.STATION_1.PART_A.STATUS.PRESENT AND "DB4000_FIX_TABLE_POSITIONS".UNIT_02.AXIS_E20_HOME_POS;
   "DB2099_MANUAL_LOAD_DMC".MANUAL_LOADING_OR_DRY_PART_LOADED_UNIT_02_P := #_w1 AND NOT "DB2099_MANUAL_LOAD_DMC".MANUAL_LOADING_OR_DRY_PART_LOADED_UNIT_02;
   "DB2099_MANUAL_LOAD_DMC".MANUAL_LOADING_OR_DRY_PART_LOADED_UNIT_02 := #_w1;
END_REGION

REGION Network 22: PART UNLOADED UNIT 01 MANUAL LOADING
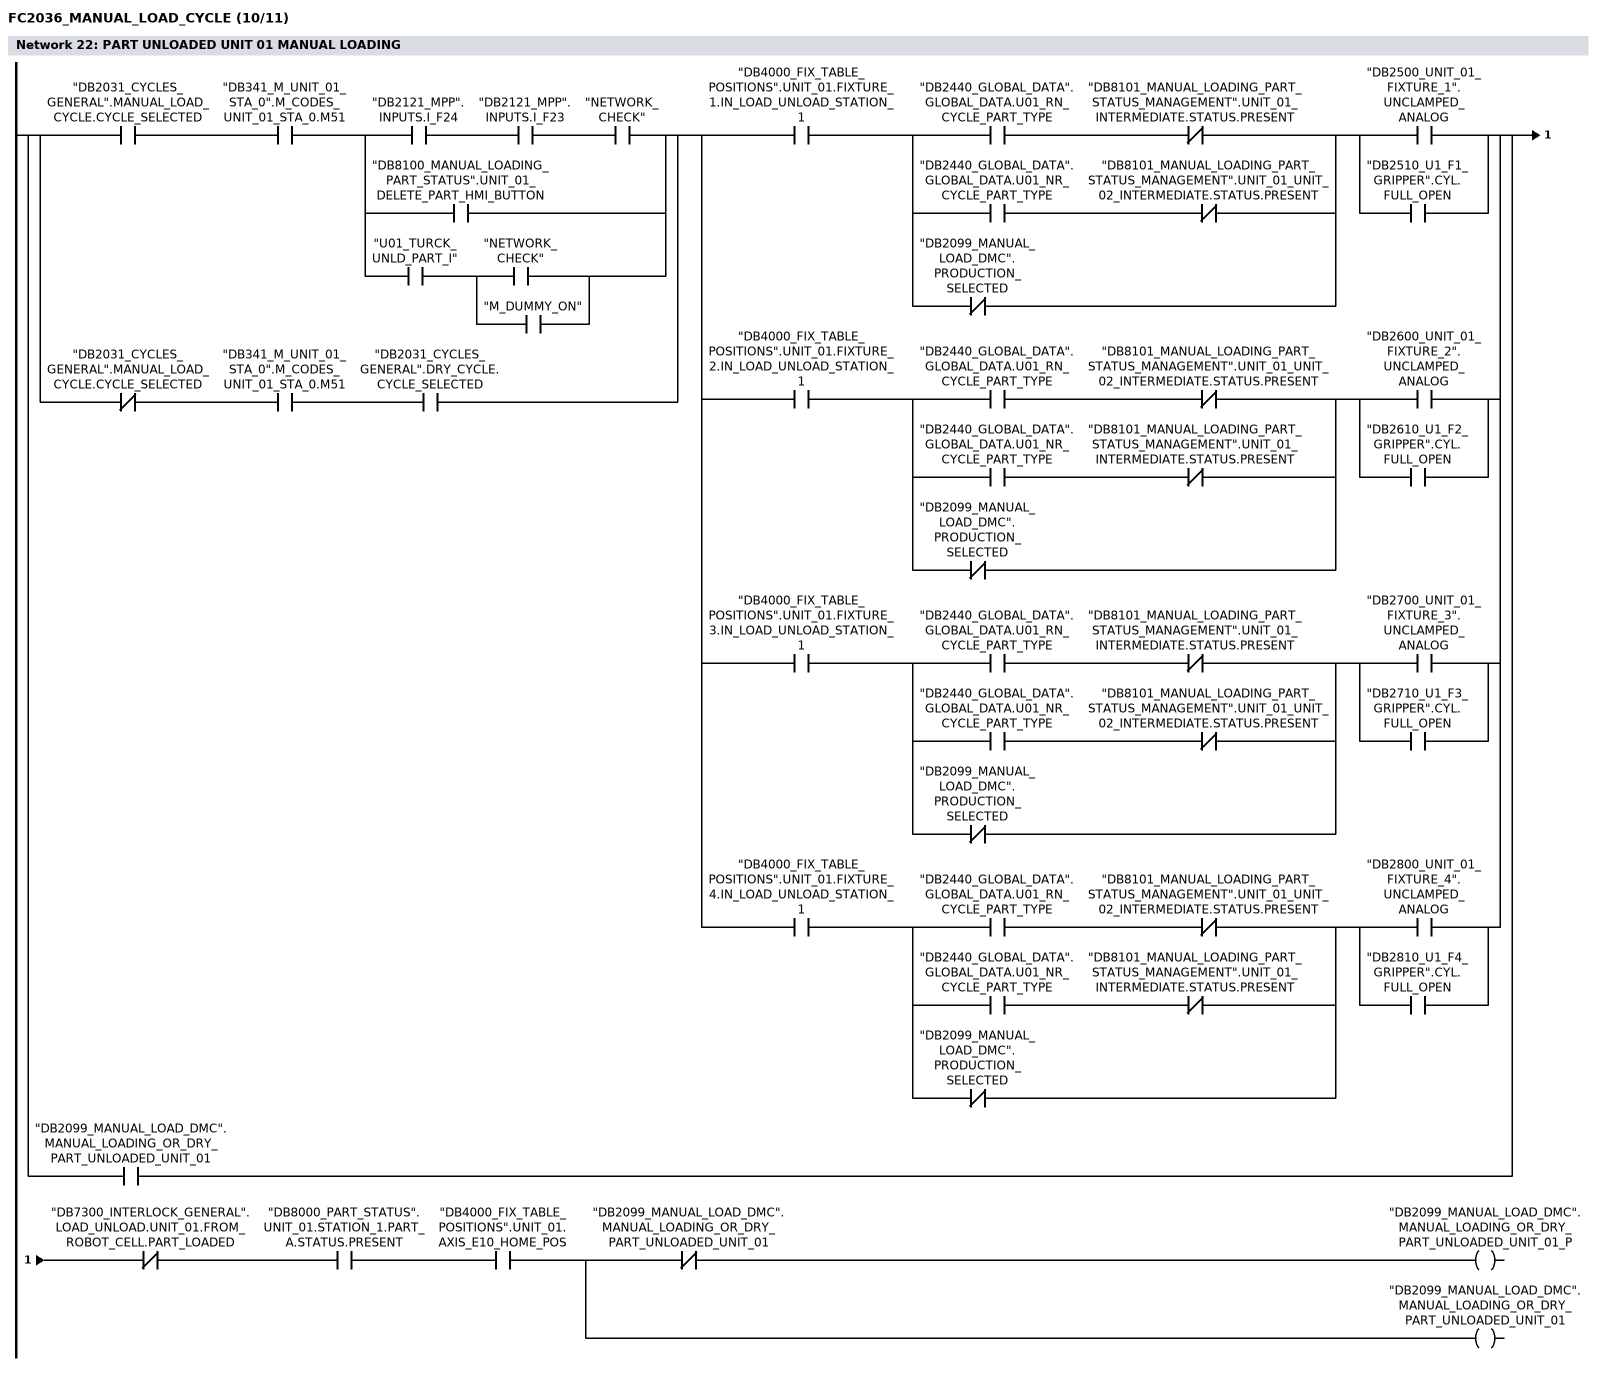
   RUNG wire#powerrail
      Contact( "DB2031_CYCLES_GENERAL".MANUAL_LOAD_CYCLE.CYCLE_SELECTED )
      Contact( "DB341_M_UNIT_01_STA_0".M_CODES_UNIT_01_STA_0.M51 )
      wire#w1
      Contact( "DB2121_MPP".INPUTS.I_F24 )
      Contact( "DB2121_MPP".INPUTS.I_F23 )
      Contact( "NETWORK_CHECK" )
      wire#w2
      Contact( "DB4000_FIX_TABLE_POSITIONS".UNIT_01.FIXTURE_1.IN_LOAD_UNLOAD_STATION_1 )
      wire#w4
      Contact( "DB2440_GLOBAL_DATA".GLOBAL_DATA.U01_RN_CYCLE_PART_TYPE )
      I_Contact( "DB8101_MANUAL_LOADING_PART_STATUS_MANAGEMENT".UNIT_01_INTERMEDIATE.STATUS.PRESENT )
      wire#w5
      Contact( "DB2500_UNIT_01_FIXTURE_1".UNCLAMPED_ANALOG )
      wire#w6
      I_Contact( "DB7300_INTERLOCK_GENERAL".LOAD_UNLOAD.UNIT_01.FROM_ROBOT_CELL.PART_LOADED )
      Contact( "DB8000_PART_STATUS".UNIT_01.STATION_1.PART_A.STATUS.PRESENT )
      Contact( "DB4000_FIX_TABLE_POSITIONS".UNIT_01.AXIS_E10_HOME_POS )
      wire#w13
      I_Contact( "DB2099_MANUAL_LOAD_DMC".MANUAL_LOADING_OR_DRY_PART_UNLOADED_UNIT_01 )
      Coil( "DB2099_MANUAL_LOAD_DMC".MANUAL_LOADING_OR_DRY_PART_UNLOADED_UNIT_01_P )
   END_RUNG
   RUNG wire#w1
      Contact( "DB8100_MANUAL_LOADING_PART_STATUS".UNIT_01_DELETE_PART_HMI_BUTTON )
   END_RUNG wire#w2
   RUNG wire#w1
      Contact( "U01_TURCK_UNLD_PART_I" )
      wire#w3
      Contact( "NETWORK_CHECK" )
   END_RUNG wire#w2
   RUNG wire#w3
      Contact( "M_DUMMY_ON" )
   END_RUNG wire#w2
   RUNG wire#powerrail
      I_Contact( "DB2031_CYCLES_GENERAL".MANUAL_LOAD_CYCLE.CYCLE_SELECTED )
      Contact( "DB341_M_UNIT_01_STA_0".M_CODES_UNIT_01_STA_0.M51 )
      Contact( "DB2031_CYCLES_GENERAL".DRY_CYCLE.CYCLE_SELECTED )
   END_RUNG wire#w2
   RUNG wire#w4
      Contact( "DB2440_GLOBAL_DATA".GLOBAL_DATA.U01_NR_CYCLE_PART_TYPE )
      I_Contact( "DB8101_MANUAL_LOADING_PART_STATUS_MANAGEMENT".UNIT_01_UNIT_02_INTERMEDIATE.STATUS.PRESENT )
   END_RUNG wire#w5
   RUNG wire#w4
      I_Contact( "DB2099_MANUAL_LOAD_DMC".PRODUCTION_SELECTED )
   END_RUNG wire#w5
   RUNG wire#w5
      Contact( "DB2510_U1_F1_GRIPPER".CYL.FULL_OPEN )
   END_RUNG wire#w6
   RUNG wire#w2
      Contact( "DB4000_FIX_TABLE_POSITIONS".UNIT_01.FIXTURE_2.IN_LOAD_UNLOAD_STATION_1 )
      wire#w7
      Contact( "DB2440_GLOBAL_DATA".GLOBAL_DATA.U01_RN_CYCLE_PART_TYPE )
      I_Contact( "DB8101_MANUAL_LOADING_PART_STATUS_MANAGEMENT".UNIT_01_UNIT_02_INTERMEDIATE.STATUS.PRESENT )
      wire#w8
      Contact( "DB2600_UNIT_01_FIXTURE_2".UNCLAMPED_ANALOG )
   END_RUNG wire#w6
   RUNG wire#w7
      Contact( "DB2440_GLOBAL_DATA".GLOBAL_DATA.U01_NR_CYCLE_PART_TYPE )
      I_Contact( "DB8101_MANUAL_LOADING_PART_STATUS_MANAGEMENT".UNIT_01_INTERMEDIATE.STATUS.PRESENT )
   END_RUNG wire#w8
   RUNG wire#w7
      I_Contact( "DB2099_MANUAL_LOAD_DMC".PRODUCTION_SELECTED )
   END_RUNG wire#w8
   RUNG wire#w8
      Contact( "DB2610_U1_F2_GRIPPER".CYL.FULL_OPEN )
   END_RUNG wire#w6
   RUNG wire#w2
      Contact( "DB4000_FIX_TABLE_POSITIONS".UNIT_01.FIXTURE_3.IN_LOAD_UNLOAD_STATION_1 )
      wire#w9
      Contact( "DB2440_GLOBAL_DATA".GLOBAL_DATA.U01_RN_CYCLE_PART_TYPE )
      I_Contact( "DB8101_MANUAL_LOADING_PART_STATUS_MANAGEMENT".UNIT_01_INTERMEDIATE.STATUS.PRESENT )
      wire#w10
      Contact( "DB2700_UNIT_01_FIXTURE_3".UNCLAMPED_ANALOG )
   END_RUNG wire#w6
   RUNG wire#w9
      Contact( "DB2440_GLOBAL_DATA".GLOBAL_DATA.U01_NR_CYCLE_PART_TYPE )
      I_Contact( "DB8101_MANUAL_LOADING_PART_STATUS_MANAGEMENT".UNIT_01_UNIT_02_INTERMEDIATE.STATUS.PRESENT )
   END_RUNG wire#w10
   RUNG wire#w9
      I_Contact( "DB2099_MANUAL_LOAD_DMC".PRODUCTION_SELECTED )
   END_RUNG wire#w10
   RUNG wire#w10
      Contact( "DB2710_U1_F3_GRIPPER".CYL.FULL_OPEN )
   END_RUNG wire#w6
   RUNG wire#w2
      Contact( "DB4000_FIX_TABLE_POSITIONS".UNIT_01.FIXTURE_4.IN_LOAD_UNLOAD_STATION_1 )
      wire#w11
      Contact( "DB2440_GLOBAL_DATA".GLOBAL_DATA.U01_RN_CYCLE_PART_TYPE )
      I_Contact( "DB8101_MANUAL_LOADING_PART_STATUS_MANAGEMENT".UNIT_01_UNIT_02_INTERMEDIATE.STATUS.PRESENT )
      wire#w12
      Contact( "DB2800_UNIT_01_FIXTURE_4".UNCLAMPED_ANALOG )
   END_RUNG wire#w6
   RUNG wire#w11
      Contact( "DB2440_GLOBAL_DATA".GLOBAL_DATA.U01_NR_CYCLE_PART_TYPE )
      I_Contact( "DB8101_MANUAL_LOADING_PART_STATUS_MANAGEMENT".UNIT_01_INTERMEDIATE.STATUS.PRESENT )
   END_RUNG wire#w12
   RUNG wire#w11
      I_Contact( "DB2099_MANUAL_LOAD_DMC".PRODUCTION_SELECTED )
   END_RUNG wire#w12
   RUNG wire#w12
      Contact( "DB2810_U1_F4_GRIPPER".CYL.FULL_OPEN )
   END_RUNG wire#w6
   RUNG wire#powerrail
      Contact( "DB2099_MANUAL_LOAD_DMC".MANUAL_LOADING_OR_DRY_PART_UNLOADED_UNIT_01 )
   END_RUNG wire#w6
   RUNG wire#w13
      Coil( "DB2099_MANUAL_LOAD_DMC".MANUAL_LOADING_OR_DRY_PART_UNLOADED_UNIT_01 )
   END_RUNG
   // the same network as SCL:
   #_w1 := (((("DB2031_CYCLES_GENERAL".MANUAL_LOAD_CYCLE.CYCLE_SELECTED AND "DB341_M_UNIT_01_STA_0".M_CODES_UNIT_01_STA_0.M51 AND (("DB2121_MPP".INPUTS.I_F24 AND "DB2121_MPP".INPUTS.I_F23 AND "NETWORK_CHECK") OR "DB8100_MANUAL_LOADING_PART_STATUS".UNIT_01_DELETE_PART_HMI_BUTTON OR ("U01_TURCK_UNLD_PART_I" AND ("NETWORK_CHECK" OR "M_DUMMY_ON")))) OR (NOT "DB2031_CYCLES_GENERAL".MANUAL_LOAD_CYCLE.CYCLE_SELECTED AND "DB341_M_UNIT_01_STA_0".M_CODES_UNIT_01_STA_0.M51 AND "DB2031_CYCLES_GENERAL".DRY_CYCLE.CYCLE_SELECTED)) AND (("DB4000_FIX_TABLE_POSITIONS".UNIT_01.FIXTURE_1.IN_LOAD_UNLOAD_STATION_1 AND (("DB2440_GLOBAL_DATA".GLOBAL_DATA.U01_RN_CYCLE_PART_TYPE AND NOT "DB8101_MANUAL_LOADING_PART_STATUS_MANAGEMENT".UNIT_01_INTERMEDIATE.STATUS.PRESENT) OR ("DB2440_GLOBAL_DATA".GLOBAL_DATA.U01_NR_CYCLE_PART_TYPE AND NOT "DB8101_MANUAL_LOADING_PART_STATUS_MANAGEMENT".UNIT_01_UNIT_02_INTERMEDIATE.STATUS.PRESENT) OR NOT "DB2099_MANUAL_LOAD_DMC".PRODUCTION_SELECTED) AND ("DB2500_UNIT_01_FIXTURE_1".UNCLAMPED_ANALOG OR "DB2510_U1_F1_GRIPPER".CYL.FULL_OPEN)) OR ("DB4000_FIX_TABLE_POSITIONS".UNIT_01.FIXTURE_2.IN_LOAD_UNLOAD_STATION_1 AND (("DB2440_GLOBAL_DATA".GLOBAL_DATA.U01_RN_CYCLE_PART_TYPE AND NOT "DB8101_MANUAL_LOADING_PART_STATUS_MANAGEMENT".UNIT_01_UNIT_02_INTERMEDIATE.STATUS.PRESENT) OR ("DB2440_GLOBAL_DATA".GLOBAL_DATA.U01_NR_CYCLE_PART_TYPE AND NOT "DB8101_MANUAL_LOADING_PART_STATUS_MANAGEMENT".UNIT_01_INTERMEDIATE.STATUS.PRESENT) OR NOT "DB2099_MANUAL_LOAD_DMC".PRODUCTION_SELECTED) AND ("DB2600_UNIT_01_FIXTURE_2".UNCLAMPED_ANALOG OR "DB2610_U1_F2_GRIPPER".CYL.FULL_OPEN)) OR ("DB4000_FIX_TABLE_POSITIONS".UNIT_01.FIXTURE_3.IN_LOAD_UNLOAD_STATION_1 AND (("DB2440_GLOBAL_DATA".GLOBAL_DATA.U01_RN_CYCLE_PART_TYPE AND NOT "DB8101_MANUAL_LOADING_PART_STATUS_MANAGEMENT".UNIT_01_INTERMEDIATE.STATUS.PRESENT) OR ("DB2440_GLOBAL_DATA".GLOBAL_DATA.U01_NR_CYCLE_PART_TYPE AND NOT "DB8101_MANUAL_LOADING_PART_STATUS_MANAGEMENT".UNIT_01_UNIT_02_INTERMEDIATE.STATUS.PRESENT) OR NOT "DB2099_MANUAL_LOAD_DMC".PRODUCTION_SELECTED) AND ("DB2700_UNIT_01_FIXTURE_3".UNCLAMPED_ANALOG OR "DB2710_U1_F3_GRIPPER".CYL.FULL_OPEN)) OR ("DB4000_FIX_TABLE_POSITIONS".UNIT_01.FIXTURE_4.IN_LOAD_UNLOAD_STATION_1 AND (("DB2440_GLOBAL_DATA".GLOBAL_DATA.U01_RN_CYCLE_PART_TYPE AND NOT "DB8101_MANUAL_LOADING_PART_STATUS_MANAGEMENT".UNIT_01_UNIT_02_INTERMEDIATE.STATUS.PRESENT) OR ("DB2440_GLOBAL_DATA".GLOBAL_DATA.U01_NR_CYCLE_PART_TYPE AND NOT "DB8101_MANUAL_LOADING_PART_STATUS_MANAGEMENT".UNIT_01_INTERMEDIATE.STATUS.PRESENT) OR NOT "DB2099_MANUAL_LOAD_DMC".PRODUCTION_SELECTED) AND ("DB2800_UNIT_01_FIXTURE_4".UNCLAMPED_ANALOG OR "DB2810_U1_F4_GRIPPER".CYL.FULL_OPEN)))) OR "DB2099_MANUAL_LOAD_DMC".MANUAL_LOADING_OR_DRY_PART_UNLOADED_UNIT_01) AND NOT "DB7300_INTERLOCK_GENERAL".LOAD_UNLOAD.UNIT_01.FROM_ROBOT_CELL.PART_LOADED AND "DB8000_PART_STATUS".UNIT_01.STATION_1.PART_A.STATUS.PRESENT AND "DB4000_FIX_TABLE_POSITIONS".UNIT_01.AXIS_E10_HOME_POS;
   "DB2099_MANUAL_LOAD_DMC".MANUAL_LOADING_OR_DRY_PART_UNLOADED_UNIT_01_P := #_w1 AND NOT "DB2099_MANUAL_LOAD_DMC".MANUAL_LOADING_OR_DRY_PART_UNLOADED_UNIT_01;
   "DB2099_MANUAL_LOAD_DMC".MANUAL_LOADING_OR_DRY_PART_UNLOADED_UNIT_01 := #_w1;
END_REGION

REGION Network 23: PART UNLOADED UNIT 02 MANUAL LOADING
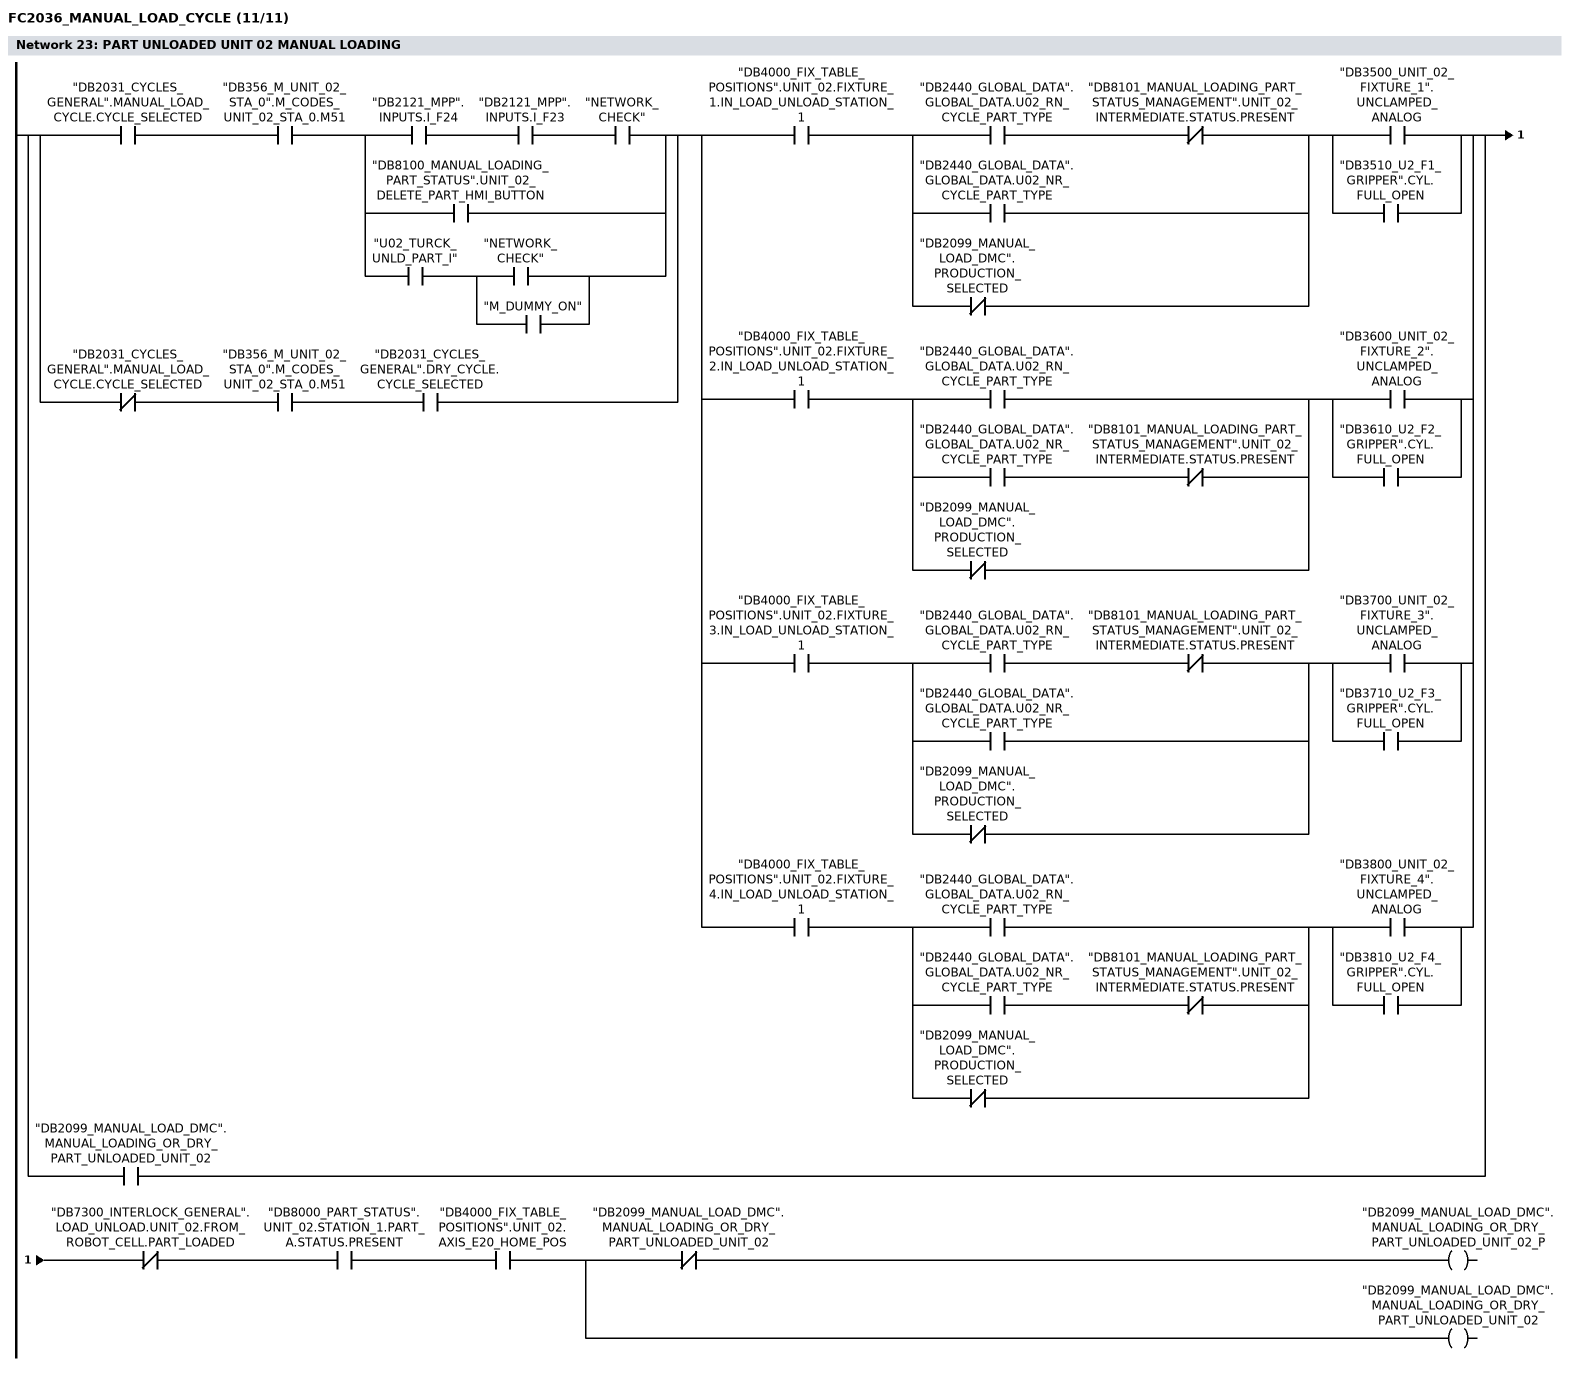
   RUNG wire#powerrail
      Contact( "DB2031_CYCLES_GENERAL".MANUAL_LOAD_CYCLE.CYCLE_SELECTED )
      Contact( "DB356_M_UNIT_02_STA_0".M_CODES_UNIT_02_STA_0.M51 )
      wire#w1
      Contact( "DB2121_MPP".INPUTS.I_F24 )
      Contact( "DB2121_MPP".INPUTS.I_F23 )
      Contact( "NETWORK_CHECK" )
      wire#w2
      Contact( "DB4000_FIX_TABLE_POSITIONS".UNIT_02.FIXTURE_1.IN_LOAD_UNLOAD_STATION_1 )
      wire#w4
      Contact( "DB2440_GLOBAL_DATA".GLOBAL_DATA.U02_RN_CYCLE_PART_TYPE )
      I_Contact( "DB8101_MANUAL_LOADING_PART_STATUS_MANAGEMENT".UNIT_02_INTERMEDIATE.STATUS.PRESENT )
      wire#w5
      Contact( "DB3500_UNIT_02_FIXTURE_1".UNCLAMPED_ANALOG )
      wire#w6
      I_Contact( "DB7300_INTERLOCK_GENERAL".LOAD_UNLOAD.UNIT_02.FROM_ROBOT_CELL.PART_LOADED )
      Contact( "DB8000_PART_STATUS".UNIT_02.STATION_1.PART_A.STATUS.PRESENT )
      Contact( "DB4000_FIX_TABLE_POSITIONS".UNIT_02.AXIS_E20_HOME_POS )
      wire#w13
      I_Contact( "DB2099_MANUAL_LOAD_DMC".MANUAL_LOADING_OR_DRY_PART_UNLOADED_UNIT_02 )
      Coil( "DB2099_MANUAL_LOAD_DMC".MANUAL_LOADING_OR_DRY_PART_UNLOADED_UNIT_02_P )
   END_RUNG
   RUNG wire#w1
      Contact( "DB8100_MANUAL_LOADING_PART_STATUS".UNIT_02_DELETE_PART_HMI_BUTTON )
   END_RUNG wire#w2
   RUNG wire#w1
      Contact( "U02_TURCK_UNLD_PART_I" )
      wire#w3
      Contact( "NETWORK_CHECK" )
   END_RUNG wire#w2
   RUNG wire#w3
      Contact( "M_DUMMY_ON" )
   END_RUNG wire#w2
   RUNG wire#powerrail
      I_Contact( "DB2031_CYCLES_GENERAL".MANUAL_LOAD_CYCLE.CYCLE_SELECTED )
      Contact( "DB356_M_UNIT_02_STA_0".M_CODES_UNIT_02_STA_0.M51 )
      Contact( "DB2031_CYCLES_GENERAL".DRY_CYCLE.CYCLE_SELECTED )
   END_RUNG wire#w2
   RUNG wire#w4
      Contact( "DB2440_GLOBAL_DATA".GLOBAL_DATA.U02_NR_CYCLE_PART_TYPE )
   END_RUNG wire#w5
   RUNG wire#w4
      I_Contact( "DB2099_MANUAL_LOAD_DMC".PRODUCTION_SELECTED )
   END_RUNG wire#w5
   RUNG wire#w5
      Contact( "DB3510_U2_F1_GRIPPER".CYL.FULL_OPEN )
   END_RUNG wire#w6
   RUNG wire#w2
      Contact( "DB4000_FIX_TABLE_POSITIONS".UNIT_02.FIXTURE_2.IN_LOAD_UNLOAD_STATION_1 )
      wire#w7
      Contact( "DB2440_GLOBAL_DATA".GLOBAL_DATA.U02_RN_CYCLE_PART_TYPE )
      wire#w8
      Contact( "DB3600_UNIT_02_FIXTURE_2".UNCLAMPED_ANALOG )
   END_RUNG wire#w6
   RUNG wire#w7
      Contact( "DB2440_GLOBAL_DATA".GLOBAL_DATA.U02_NR_CYCLE_PART_TYPE )
      I_Contact( "DB8101_MANUAL_LOADING_PART_STATUS_MANAGEMENT".UNIT_02_INTERMEDIATE.STATUS.PRESENT )
   END_RUNG wire#w8
   RUNG wire#w7
      I_Contact( "DB2099_MANUAL_LOAD_DMC".PRODUCTION_SELECTED )
   END_RUNG wire#w8
   RUNG wire#w8
      Contact( "DB3610_U2_F2_GRIPPER".CYL.FULL_OPEN )
   END_RUNG wire#w6
   RUNG wire#w2
      Contact( "DB4000_FIX_TABLE_POSITIONS".UNIT_02.FIXTURE_3.IN_LOAD_UNLOAD_STATION_1 )
      wire#w9
      Contact( "DB2440_GLOBAL_DATA".GLOBAL_DATA.U02_RN_CYCLE_PART_TYPE )
      I_Contact( "DB8101_MANUAL_LOADING_PART_STATUS_MANAGEMENT".UNIT_02_INTERMEDIATE.STATUS.PRESENT )
      wire#w10
      Contact( "DB3700_UNIT_02_FIXTURE_3".UNCLAMPED_ANALOG )
   END_RUNG wire#w6
   RUNG wire#w9
      Contact( "DB2440_GLOBAL_DATA".GLOBAL_DATA.U02_NR_CYCLE_PART_TYPE )
   END_RUNG wire#w10
   RUNG wire#w9
      I_Contact( "DB2099_MANUAL_LOAD_DMC".PRODUCTION_SELECTED )
   END_RUNG wire#w10
   RUNG wire#w10
      Contact( "DB3710_U2_F3_GRIPPER".CYL.FULL_OPEN )
   END_RUNG wire#w6
   RUNG wire#w2
      Contact( "DB4000_FIX_TABLE_POSITIONS".UNIT_02.FIXTURE_4.IN_LOAD_UNLOAD_STATION_1 )
      wire#w11
      Contact( "DB2440_GLOBAL_DATA".GLOBAL_DATA.U02_RN_CYCLE_PART_TYPE )
      wire#w12
      Contact( "DB3800_UNIT_02_FIXTURE_4".UNCLAMPED_ANALOG )
   END_RUNG wire#w6
   RUNG wire#w11
      Contact( "DB2440_GLOBAL_DATA".GLOBAL_DATA.U02_NR_CYCLE_PART_TYPE )
      I_Contact( "DB8101_MANUAL_LOADING_PART_STATUS_MANAGEMENT".UNIT_02_INTERMEDIATE.STATUS.PRESENT )
   END_RUNG wire#w12
   RUNG wire#w11
      I_Contact( "DB2099_MANUAL_LOAD_DMC".PRODUCTION_SELECTED )
   END_RUNG wire#w12
   RUNG wire#w12
      Contact( "DB3810_U2_F4_GRIPPER".CYL.FULL_OPEN )
   END_RUNG wire#w6
   RUNG wire#powerrail
      Contact( "DB2099_MANUAL_LOAD_DMC".MANUAL_LOADING_OR_DRY_PART_UNLOADED_UNIT_02 )
   END_RUNG wire#w6
   RUNG wire#w13
      Coil( "DB2099_MANUAL_LOAD_DMC".MANUAL_LOADING_OR_DRY_PART_UNLOADED_UNIT_02 )
   END_RUNG
   // the same network as SCL:
   #_w1 := (((("DB2031_CYCLES_GENERAL".MANUAL_LOAD_CYCLE.CYCLE_SELECTED AND "DB356_M_UNIT_02_STA_0".M_CODES_UNIT_02_STA_0.M51 AND (("DB2121_MPP".INPUTS.I_F24 AND "DB2121_MPP".INPUTS.I_F23 AND "NETWORK_CHECK") OR "DB8100_MANUAL_LOADING_PART_STATUS".UNIT_02_DELETE_PART_HMI_BUTTON OR ("U02_TURCK_UNLD_PART_I" AND ("NETWORK_CHECK" OR "M_DUMMY_ON")))) OR (NOT "DB2031_CYCLES_GENERAL".MANUAL_LOAD_CYCLE.CYCLE_SELECTED AND "DB356_M_UNIT_02_STA_0".M_CODES_UNIT_02_STA_0.M51 AND "DB2031_CYCLES_GENERAL".DRY_CYCLE.CYCLE_SELECTED)) AND (("DB4000_FIX_TABLE_POSITIONS".UNIT_02.FIXTURE_1.IN_LOAD_UNLOAD_STATION_1 AND (("DB2440_GLOBAL_DATA".GLOBAL_DATA.U02_RN_CYCLE_PART_TYPE AND NOT "DB8101_MANUAL_LOADING_PART_STATUS_MANAGEMENT".UNIT_02_INTERMEDIATE.STATUS.PRESENT) OR "DB2440_GLOBAL_DATA".GLOBAL_DATA.U02_NR_CYCLE_PART_TYPE OR NOT "DB2099_MANUAL_LOAD_DMC".PRODUCTION_SELECTED) AND ("DB3500_UNIT_02_FIXTURE_1".UNCLAMPED_ANALOG OR "DB3510_U2_F1_GRIPPER".CYL.FULL_OPEN)) OR ("DB4000_FIX_TABLE_POSITIONS".UNIT_02.FIXTURE_2.IN_LOAD_UNLOAD_STATION_1 AND ("DB2440_GLOBAL_DATA".GLOBAL_DATA.U02_RN_CYCLE_PART_TYPE OR ("DB2440_GLOBAL_DATA".GLOBAL_DATA.U02_NR_CYCLE_PART_TYPE AND NOT "DB8101_MANUAL_LOADING_PART_STATUS_MANAGEMENT".UNIT_02_INTERMEDIATE.STATUS.PRESENT) OR NOT "DB2099_MANUAL_LOAD_DMC".PRODUCTION_SELECTED) AND ("DB3600_UNIT_02_FIXTURE_2".UNCLAMPED_ANALOG OR "DB3610_U2_F2_GRIPPER".CYL.FULL_OPEN)) OR ("DB4000_FIX_TABLE_POSITIONS".UNIT_02.FIXTURE_3.IN_LOAD_UNLOAD_STATION_1 AND (("DB2440_GLOBAL_DATA".GLOBAL_DATA.U02_RN_CYCLE_PART_TYPE AND NOT "DB8101_MANUAL_LOADING_PART_STATUS_MANAGEMENT".UNIT_02_INTERMEDIATE.STATUS.PRESENT) OR "DB2440_GLOBAL_DATA".GLOBAL_DATA.U02_NR_CYCLE_PART_TYPE OR NOT "DB2099_MANUAL_LOAD_DMC".PRODUCTION_SELECTED) AND ("DB3700_UNIT_02_FIXTURE_3".UNCLAMPED_ANALOG OR "DB3710_U2_F3_GRIPPER".CYL.FULL_OPEN)) OR ("DB4000_FIX_TABLE_POSITIONS".UNIT_02.FIXTURE_4.IN_LOAD_UNLOAD_STATION_1 AND ("DB2440_GLOBAL_DATA".GLOBAL_DATA.U02_RN_CYCLE_PART_TYPE OR ("DB2440_GLOBAL_DATA".GLOBAL_DATA.U02_NR_CYCLE_PART_TYPE AND NOT "DB8101_MANUAL_LOADING_PART_STATUS_MANAGEMENT".UNIT_02_INTERMEDIATE.STATUS.PRESENT) OR NOT "DB2099_MANUAL_LOAD_DMC".PRODUCTION_SELECTED) AND ("DB3800_UNIT_02_FIXTURE_4".UNCLAMPED_ANALOG OR "DB3810_U2_F4_GRIPPER".CYL.FULL_OPEN)))) OR "DB2099_MANUAL_LOAD_DMC".MANUAL_LOADING_OR_DRY_PART_UNLOADED_UNIT_02) AND NOT "DB7300_INTERLOCK_GENERAL".LOAD_UNLOAD.UNIT_02.FROM_ROBOT_CELL.PART_LOADED AND "DB8000_PART_STATUS".UNIT_02.STATION_1.PART_A.STATUS.PRESENT AND "DB4000_FIX_TABLE_POSITIONS".UNIT_02.AXIS_E20_HOME_POS;
   "DB2099_MANUAL_LOAD_DMC".MANUAL_LOADING_OR_DRY_PART_UNLOADED_UNIT_02_P := #_w1 AND NOT "DB2099_MANUAL_LOAD_DMC".MANUAL_LOADING_OR_DRY_PART_UNLOADED_UNIT_02;
   "DB2099_MANUAL_LOAD_DMC".MANUAL_LOADING_OR_DRY_PART_UNLOADED_UNIT_02 := #_w1;
END_REGION
END_FUNCTION
